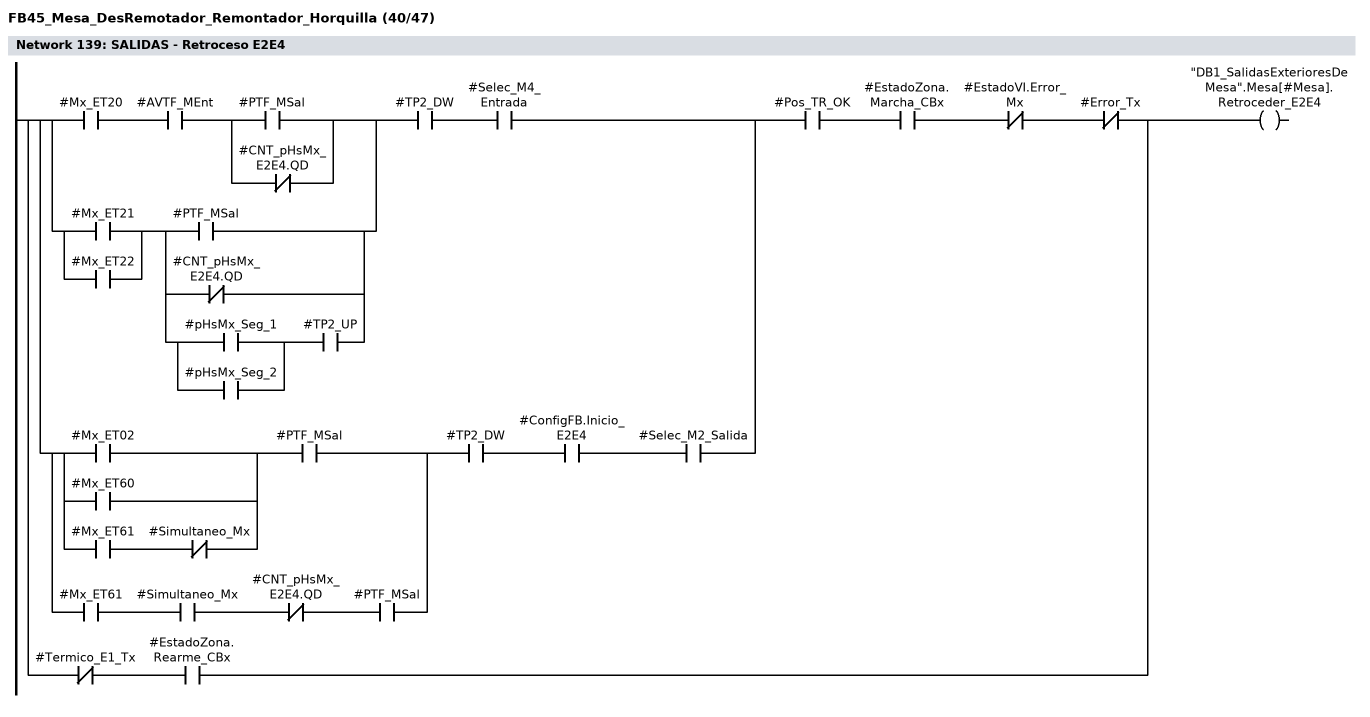
   RUNG wire#powerrail
      Contact( #Mx_ET20 )
      Contact( #AVTF_MEnt )
      wire#w1
      Contact( #PTF_MSal )
      wire#w2
      Contact( #TP2_DW )
      Contact( #Selec_M4_Entrada )
      wire#w5
      Contact( #Pos_TR_OK )
      Contact( #EstadoZona.Marcha_CBx )
      I_Contact( #EstadoVI.Error_Mx )
      I_Contact( #Error_Tx )
      wire#w8
      Coil( "DB1_SalidasExterioresDeMesa".Mesa[#Mesa].Retroceder_E2E4 )
   END_RUNG
   RUNG wire#w1
      I_Contact( #CNT_pHsMx_E2E4.QD )
   END_RUNG wire#w2
   RUNG wire#powerrail
      Contact( #Mx_ET21 )
      wire#w3
      Contact( #PTF_MSal )
   END_RUNG wire#w2
   RUNG wire#powerrail
      Contact( #Mx_ET22 )
   END_RUNG wire#w3
   RUNG wire#w3
      I_Contact( #CNT_pHsMx_E2E4.QD )
   END_RUNG wire#w2
   RUNG wire#w3
      Contact( #pHsMx_Seg_1 )
      wire#w4
      Contact( #TP2_UP )
   END_RUNG wire#w2
   RUNG wire#w3
      Contact( #pHsMx_Seg_2 )
   END_RUNG wire#w4
   RUNG wire#powerrail
      Contact( #Mx_ET02 )
      wire#w6
      Contact( #PTF_MSal )
      wire#w7
      Contact( #TP2_DW )
      Contact( #ConfigFB.Inicio_E2E4 )
      Contact( #Selec_M2_Salida )
   END_RUNG wire#w5
   RUNG wire#powerrail
      Contact( #Mx_ET60 )
   END_RUNG wire#w6
   RUNG wire#powerrail
      Contact( #Mx_ET61 )
      I_Contact( #Simultaneo_Mx )
   END_RUNG wire#w6
   RUNG wire#powerrail
      Contact( #Mx_ET61 )
      Contact( #Simultaneo_Mx )
      I_Contact( #CNT_pHsMx_E2E4.QD )
      Contact( #PTF_MSal )
   END_RUNG wire#w7
   RUNG wire#powerrail
      I_Contact( #Termico_E1_Tx )
      Contact( #EstadoZona.Rearme_CBx )
   END_RUNG wire#w8
   // the same network as SCL:
   "DB1_SalidasExterioresDeMesa".Mesa[#Mesa].Retroceder_E2E4 := (((((#Mx_ET20 AND #AVTF_MEnt AND (#PTF_MSal OR NOT #CNT_pHsMx_E2E4.QD)) OR ((#Mx_ET21 OR #Mx_ET22) AND (#PTF_MSal OR NOT #CNT_pHsMx_E2E4.QD OR ((#pHsMx_Seg_1 OR #pHsMx_Seg_2) AND #TP2_UP)))) AND #TP2_DW AND #Selec_M4_Entrada) OR ((((#Mx_ET02 OR #Mx_ET60 OR (#Mx_ET61 AND NOT #Simultaneo_Mx)) AND #PTF_MSal) OR (#Mx_ET61 AND #Simultaneo_Mx AND NOT #CNT_pHsMx_E2E4.QD AND #PTF_MSal)) AND #TP2_DW AND #ConfigFB.Inicio_E2E4 AND #Selec_M2_Salida)) AND #Pos_TR_OK AND #EstadoZona.Marcha_CBx AND NOT #EstadoVI.Error_Mx AND NOT #Error_Tx) OR (NOT #Termico_E1_Tx AND #EstadoZona.Rearme_CBx);
END_REGION

REGION Network 140: SALIDAS - Parar E2E4
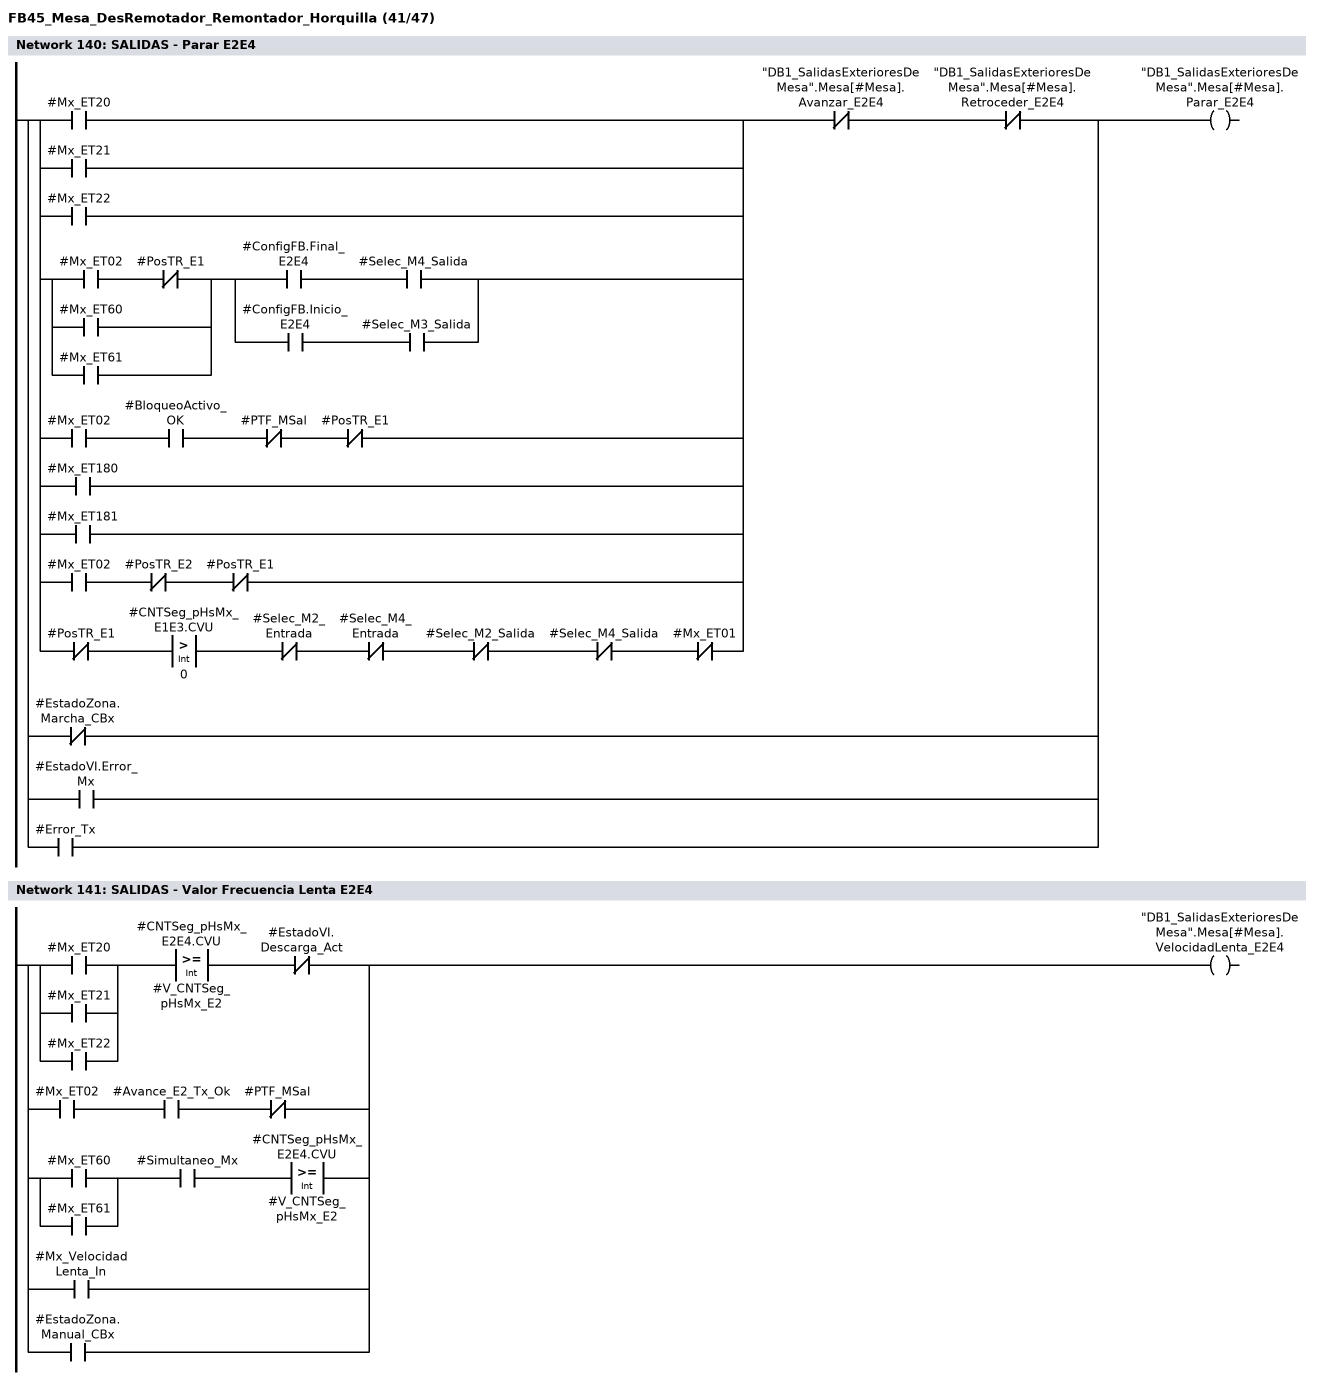
   RUNG wire#powerrail
      Contact( #Mx_ET20 )
      wire#w1
      I_Contact( "DB1_SalidasExterioresDeMesa".Mesa[#Mesa].Avanzar_E2E4 )
      I_Contact( "DB1_SalidasExterioresDeMesa".Mesa[#Mesa].Retroceder_E2E4 )
      wire#w3
      Coil( "DB1_SalidasExterioresDeMesa".Mesa[#Mesa].Parar_E2E4 )
   END_RUNG
   RUNG wire#powerrail
      Contact( #Mx_ET21 )
   END_RUNG wire#w1
   RUNG wire#powerrail
      Contact( #Mx_ET22 )
   END_RUNG wire#w1
   RUNG wire#powerrail
      Contact( #Mx_ET02 )
      I_Contact( #PosTR_E1 )
      wire#w2
      Contact( #ConfigFB.Final_E2E4 )
      Contact( #Selec_M4_Salida )
   END_RUNG wire#w1
   RUNG wire#powerrail
      Contact( #Mx_ET60 )
   END_RUNG wire#w2
   RUNG wire#powerrail
      Contact( #Mx_ET61 )
   END_RUNG wire#w2
   RUNG wire#w2
      Contact( #ConfigFB.Inicio_E2E4 )
      Contact( #Selec_M3_Salida )
   END_RUNG wire#w1
   RUNG wire#powerrail
      Contact( #Mx_ET02 )
      Contact( #BloqueoActivo_OK )
      I_Contact( #PTF_MSal )
      I_Contact( #PosTR_E1 )
   END_RUNG wire#w1
   RUNG wire#powerrail
      Contact( #Mx_ET180 )
   END_RUNG wire#w1
   RUNG wire#powerrail
      Contact( #Mx_ET181 )
   END_RUNG wire#w1
   RUNG wire#powerrail
      Contact( #Mx_ET02 )
      I_Contact( #PosTR_E2 )
      I_Contact( #PosTR_E1 )
   END_RUNG wire#w1
   RUNG wire#powerrail
      I_Contact( #PosTR_E1 )
      { S7_Templates := "SrcType := Int" } GT_Contact(in1 := #CNTSeg_pHsMx_E1E3.CVU, in2 := 0)
      I_Contact( #Selec_M2_Entrada )
      I_Contact( #Selec_M4_Entrada )
      I_Contact( #Selec_M2_Salida )
      I_Contact( #Selec_M4_Salida )
      I_Contact( #Mx_ET01 )
   END_RUNG wire#w1
   RUNG wire#powerrail
      I_Contact( #EstadoZona.Marcha_CBx )
   END_RUNG wire#w3
   RUNG wire#powerrail
      Contact( #EstadoVI.Error_Mx )
   END_RUNG wire#w3
   RUNG wire#powerrail
      Contact( #Error_Tx )
   END_RUNG wire#w3
   // the same network as SCL:
   "DB1_SalidasExterioresDeMesa".Mesa[#Mesa].Parar_E2E4 := ((#Mx_ET20 OR #Mx_ET21 OR #Mx_ET22 OR (((#Mx_ET02 AND NOT #PosTR_E1) OR #Mx_ET60 OR #Mx_ET61) AND ((#ConfigFB.Final_E2E4 AND #Selec_M4_Salida) OR (#ConfigFB.Inicio_E2E4 AND #Selec_M3_Salida))) OR (#Mx_ET02 AND #BloqueoActivo_OK AND NOT #PTF_MSal AND NOT #PosTR_E1) OR #Mx_ET180 OR #Mx_ET181 OR (#Mx_ET02 AND NOT #PosTR_E2 AND NOT #PosTR_E1) OR (NOT #PosTR_E1 AND (#CNTSeg_pHsMx_E1E3.CVU > 0) AND NOT #Selec_M2_Entrada AND NOT #Selec_M4_Entrada AND NOT #Selec_M2_Salida AND NOT #Selec_M4_Salida AND NOT #Mx_ET01)) AND NOT "DB1_SalidasExterioresDeMesa".Mesa[#Mesa].Avanzar_E2E4 AND NOT "DB1_SalidasExterioresDeMesa".Mesa[#Mesa].Retroceder_E2E4) OR NOT #EstadoZona.Marcha_CBx OR #EstadoVI.Error_Mx OR #Error_Tx;
END_REGION

REGION Network 141: SALIDAS - Valor Frecuencia Lenta E2E4
   RUNG wire#powerrail
      Contact( #Mx_ET20 )
      wire#w1
      { S7_Templates := "SrcType := Int" } GE_Contact(in1 := #CNTSeg_pHsMx_E2E4.CVU, in2 := #V_CNTSeg_pHsMx_E2)
      I_Contact( #EstadoVI.Descarga_Act )
      wire#w2
      Coil( "DB1_SalidasExterioresDeMesa".Mesa[#Mesa].VelocidadLenta_E2E4 )
   END_RUNG
   RUNG wire#powerrail
      Contact( #Mx_ET21 )
   END_RUNG wire#w1
   RUNG wire#powerrail
      Contact( #Mx_ET22 )
   END_RUNG wire#w1
   RUNG wire#powerrail
      Contact( #Mx_ET02 )
      Contact( #Avance_E2_Tx_Ok )
      I_Contact( #PTF_MSal )
   END_RUNG wire#w2
   RUNG wire#powerrail
      Contact( #Mx_ET60 )
      wire#w3
      Contact( #Simultaneo_Mx )
      { S7_Templates := "SrcType := Int" } GE_Contact(in1 := #CNTSeg_pHsMx_E2E4.CVU, in2 := #V_CNTSeg_pHsMx_E2)
   END_RUNG wire#w2
   RUNG wire#powerrail
      Contact( #Mx_ET61 )
   END_RUNG wire#w3
   RUNG wire#powerrail
      Contact( #Mx_VelocidadLenta_In )
   END_RUNG wire#w2
   RUNG wire#powerrail
      Contact( #EstadoZona.Manual_CBx )
   END_RUNG wire#w2
   // the same network as SCL:
   "DB1_SalidasExterioresDeMesa".Mesa[#Mesa].VelocidadLenta_E2E4 := ((#Mx_ET20 OR #Mx_ET21 OR #Mx_ET22) AND (#CNTSeg_pHsMx_E2E4.CVU >= #V_CNTSeg_pHsMx_E2) AND NOT #EstadoVI.Descarga_Act) OR (#Mx_ET02 AND #Avance_E2_Tx_Ok AND NOT #PTF_MSal) OR ((#Mx_ET60 OR #Mx_ET61) AND #Simultaneo_Mx AND (#CNTSeg_pHsMx_E2E4.CVU >= #V_CNTSeg_pHsMx_E2)) OR #Mx_VelocidadLenta_In OR #EstadoZona.Manual_CBx;
END_REGION

REGION Network 142: SALIDAS - Ir a posicion E1E3
   // DANI: 2021/06/28. BAJAR EL TOPE DE CADENAS SI HAY S2 O S4 EN ETAPA2 Y TR POS RODILLOS
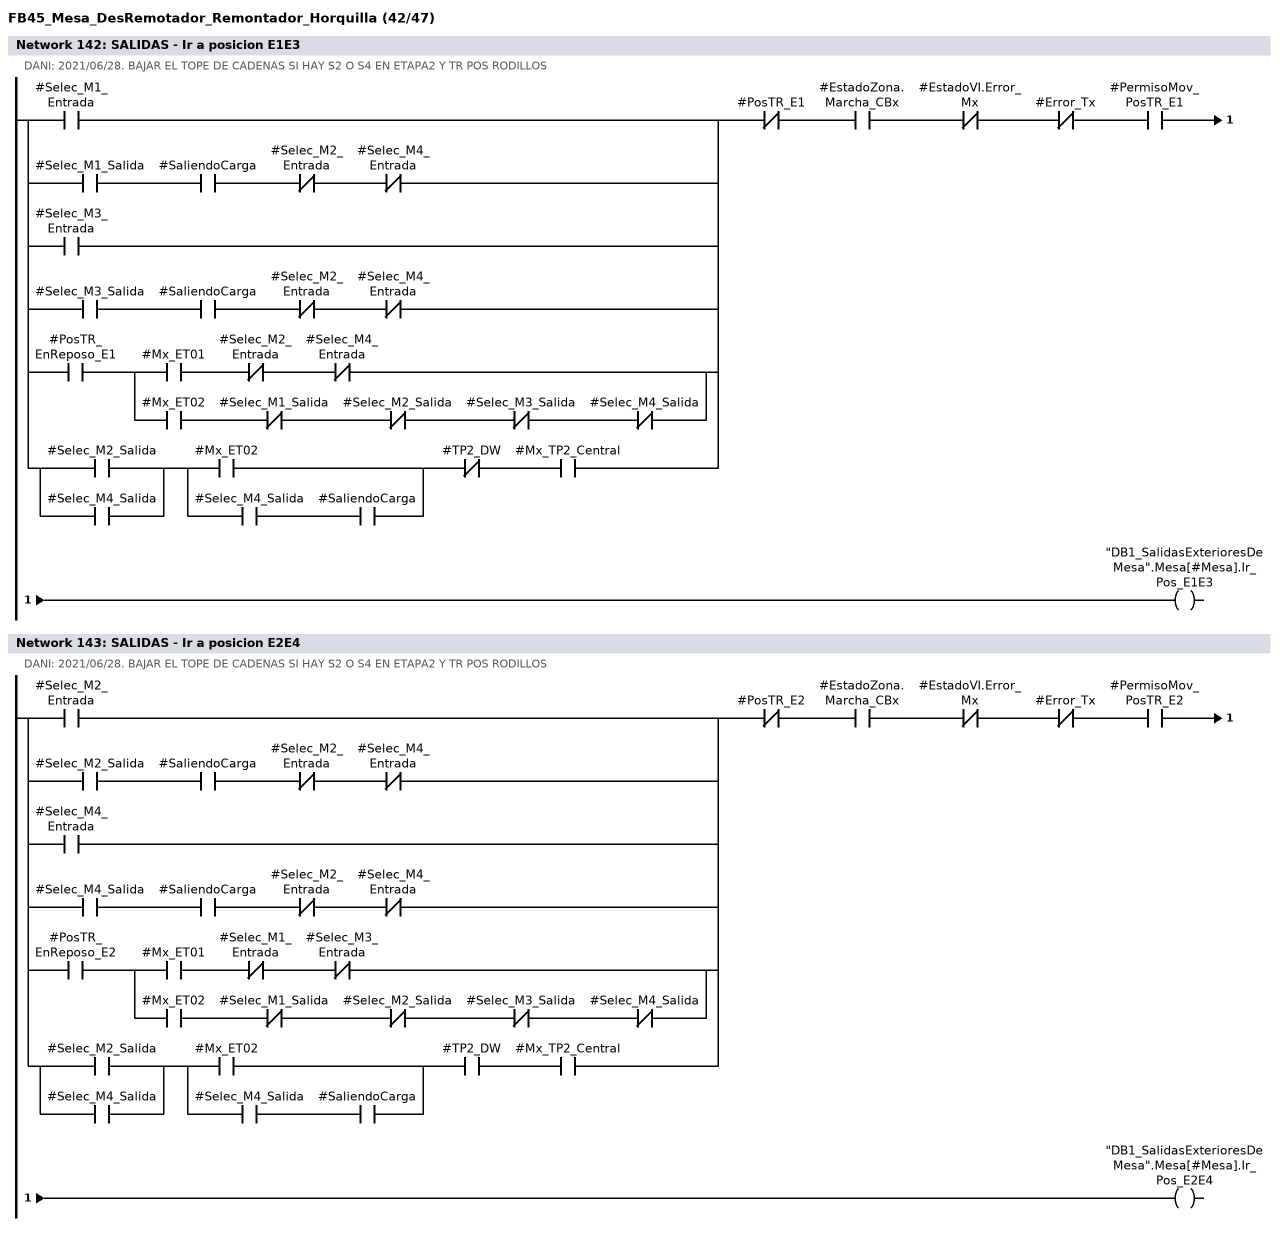
   RUNG wire#powerrail
      Contact( #Selec_M1_Entrada )
      wire#w1
      I_Contact( #PosTR_E1 )
      Contact( #EstadoZona.Marcha_CBx )
      I_Contact( #EstadoVI.Error_Mx )
      I_Contact( #Error_Tx )
      Contact( #PermisoMov_PosTR_E1 )
      Coil( "DB1_SalidasExterioresDeMesa".Mesa[#Mesa].Ir_Pos_E1E3 )
   END_RUNG
   RUNG wire#powerrail
      Contact( #Selec_M1_Salida )
      Contact( #SaliendoCarga )
      I_Contact( #Selec_M2_Entrada )
      I_Contact( #Selec_M4_Entrada )
   END_RUNG wire#w1
   RUNG wire#powerrail
      Contact( #Selec_M3_Entrada )
   END_RUNG wire#w1
   RUNG wire#powerrail
      Contact( #Selec_M3_Salida )
      Contact( #SaliendoCarga )
      I_Contact( #Selec_M2_Entrada )
      I_Contact( #Selec_M4_Entrada )
   END_RUNG wire#w1
   RUNG wire#powerrail
      Contact( #PosTR_EnReposo_E1 )
      wire#w2
      Contact( #Mx_ET01 )
      I_Contact( #Selec_M2_Entrada )
      I_Contact( #Selec_M4_Entrada )
   END_RUNG wire#w1
   RUNG wire#w2
      Contact( #Mx_ET02 )
      I_Contact( #Selec_M1_Salida )
      I_Contact( #Selec_M2_Salida )
      I_Contact( #Selec_M3_Salida )
      I_Contact( #Selec_M4_Salida )
   END_RUNG wire#w1
   RUNG wire#powerrail
      Contact( #Selec_M2_Salida )
      wire#w3
      Contact( #Mx_ET02 )
      wire#w4
      I_Contact( #TP2_DW )
      Contact( #Mx_TP2_Central )
   END_RUNG wire#w1
   RUNG wire#powerrail
      Contact( #Selec_M4_Salida )
   END_RUNG wire#w3
   RUNG wire#w3
      Contact( #Selec_M4_Salida )
      Contact( #SaliendoCarga )
   END_RUNG wire#w4
   // the same network as SCL:
   "DB1_SalidasExterioresDeMesa".Mesa[#Mesa].Ir_Pos_E1E3 := (#Selec_M1_Entrada OR (#Selec_M1_Salida AND #SaliendoCarga AND NOT #Selec_M2_Entrada AND NOT #Selec_M4_Entrada) OR #Selec_M3_Entrada OR (#Selec_M3_Salida AND #SaliendoCarga AND NOT #Selec_M2_Entrada AND NOT #Selec_M4_Entrada) OR (#PosTR_EnReposo_E1 AND ((#Mx_ET01 AND NOT #Selec_M2_Entrada AND NOT #Selec_M4_Entrada) OR (#Mx_ET02 AND NOT #Selec_M1_Salida AND NOT #Selec_M2_Salida AND NOT #Selec_M3_Salida AND NOT #Selec_M4_Salida))) OR ((#Selec_M2_Salida OR #Selec_M4_Salida) AND (#Mx_ET02 OR (#Selec_M4_Salida AND #SaliendoCarga)) AND NOT #TP2_DW AND #Mx_TP2_Central)) AND NOT #PosTR_E1 AND #EstadoZona.Marcha_CBx AND NOT #EstadoVI.Error_Mx AND NOT #Error_Tx AND #PermisoMov_PosTR_E1;
END_REGION

REGION Network 143: SALIDAS - Ir a posicion E2E4
   // DANI: 2021/06/28. BAJAR EL TOPE DE CADENAS SI HAY S2 O S4 EN ETAPA2 Y TR POS RODILLOS
   RUNG wire#powerrail
      Contact( #Selec_M2_Entrada )
      wire#w1
      I_Contact( #PosTR_E2 )
      Contact( #EstadoZona.Marcha_CBx )
      I_Contact( #EstadoVI.Error_Mx )
      I_Contact( #Error_Tx )
      Contact( #PermisoMov_PosTR_E2 )
      Coil( "DB1_SalidasExterioresDeMesa".Mesa[#Mesa].Ir_Pos_E2E4 )
   END_RUNG
   RUNG wire#powerrail
      Contact( #Selec_M2_Salida )
      Contact( #SaliendoCarga )
      I_Contact( #Selec_M2_Entrada )
      I_Contact( #Selec_M4_Entrada )
   END_RUNG wire#w1
   RUNG wire#powerrail
      Contact( #Selec_M4_Entrada )
   END_RUNG wire#w1
   RUNG wire#powerrail
      Contact( #Selec_M4_Salida )
      Contact( #SaliendoCarga )
      I_Contact( #Selec_M2_Entrada )
      I_Contact( #Selec_M4_Entrada )
   END_RUNG wire#w1
   RUNG wire#powerrail
      Contact( #PosTR_EnReposo_E2 )
      wire#w2
      Contact( #Mx_ET01 )
      I_Contact( #Selec_M1_Entrada )
      I_Contact( #Selec_M3_Entrada )
   END_RUNG wire#w1
   RUNG wire#w2
      Contact( #Mx_ET02 )
      I_Contact( #Selec_M1_Salida )
      I_Contact( #Selec_M2_Salida )
      I_Contact( #Selec_M3_Salida )
      I_Contact( #Selec_M4_Salida )
   END_RUNG wire#w1
   RUNG wire#powerrail
      Contact( #Selec_M2_Salida )
      wire#w3
      Contact( #Mx_ET02 )
      wire#w4
      Contact( #TP2_DW )
      Contact( #Mx_TP2_Central )
   END_RUNG wire#w1
   RUNG wire#powerrail
      Contact( #Selec_M4_Salida )
   END_RUNG wire#w3
   RUNG wire#w3
      Contact( #Selec_M4_Salida )
      Contact( #SaliendoCarga )
   END_RUNG wire#w4
   // the same network as SCL:
   "DB1_SalidasExterioresDeMesa".Mesa[#Mesa].Ir_Pos_E2E4 := (#Selec_M2_Entrada OR (#Selec_M2_Salida AND #SaliendoCarga AND NOT #Selec_M2_Entrada AND NOT #Selec_M4_Entrada) OR #Selec_M4_Entrada OR (#Selec_M4_Salida AND #SaliendoCarga AND NOT #Selec_M2_Entrada AND NOT #Selec_M4_Entrada) OR (#PosTR_EnReposo_E2 AND ((#Mx_ET01 AND NOT #Selec_M1_Entrada AND NOT #Selec_M3_Entrada) OR (#Mx_ET02 AND NOT #Selec_M1_Salida AND NOT #Selec_M2_Salida AND NOT #Selec_M3_Salida AND NOT #Selec_M4_Salida))) OR ((#Selec_M2_Salida OR #Selec_M4_Salida) AND (#Mx_ET02 OR (#Selec_M4_Salida AND #SaliendoCarga)) AND #TP2_DW AND #Mx_TP2_Central)) AND NOT #PosTR_E2 AND #EstadoZona.Marcha_CBx AND NOT #EstadoVI.Error_Mx AND NOT #Error_Tx AND #PermisoMov_PosTR_E2;
END_REGION

REGION Network 144: SALIDAS - Bajar TP1
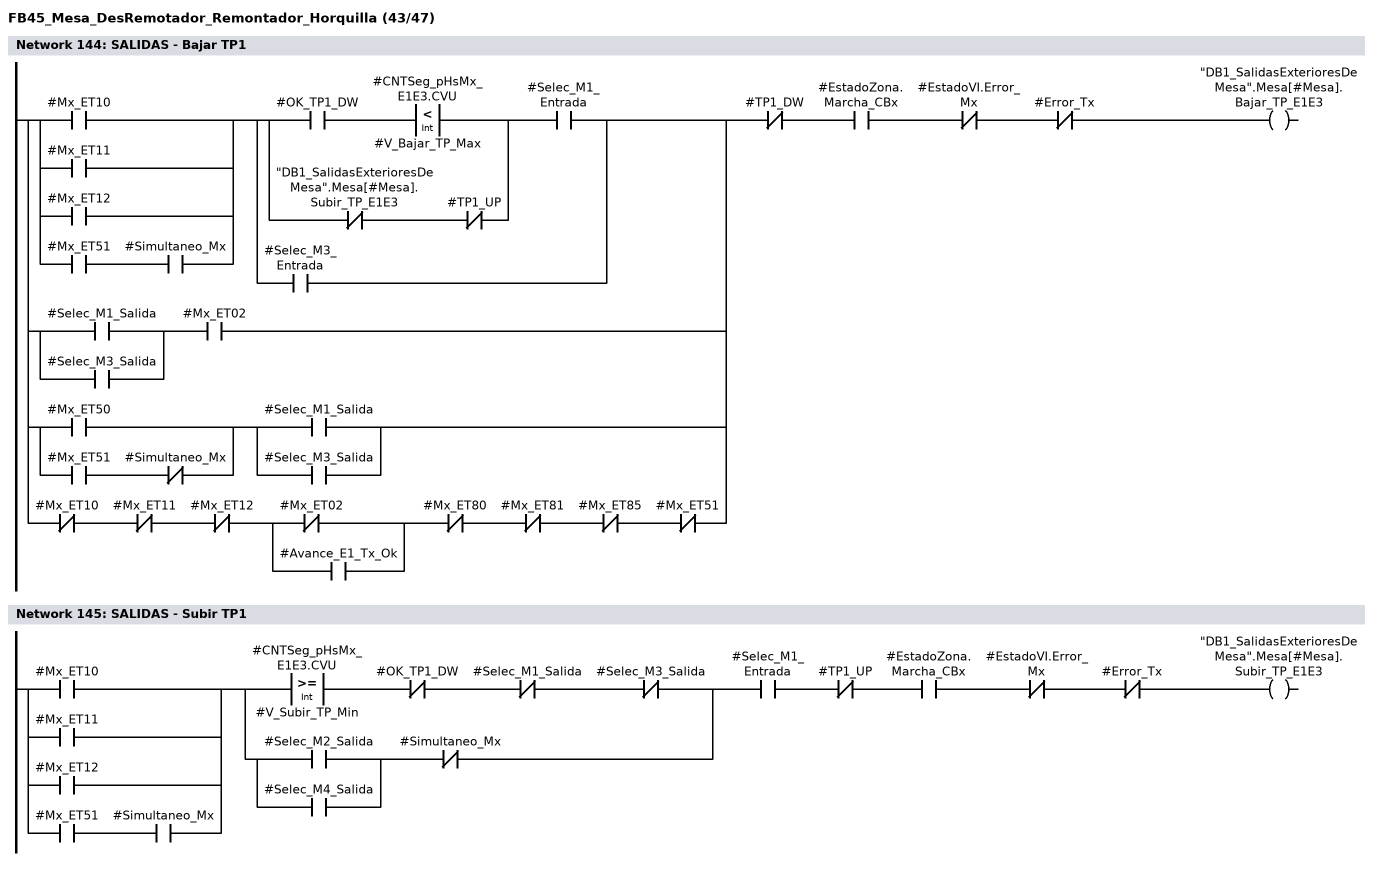
   RUNG wire#powerrail
      Contact( #Mx_ET10 )
      wire#w1
      Contact( #OK_TP1_DW )
      { S7_Templates := "SrcType := Int" } LT_Contact(in1 := #CNTSeg_pHsMx_E1E3.CVU, in2 := #V_Bajar_TP_Max)
      wire#w2
      Contact( #Selec_M1_Entrada )
      wire#w3
      I_Contact( #TP1_DW )
      Contact( #EstadoZona.Marcha_CBx )
      I_Contact( #EstadoVI.Error_Mx )
      I_Contact( #Error_Tx )
      Coil( "DB1_SalidasExterioresDeMesa".Mesa[#Mesa].Bajar_TP_E1E3 )
   END_RUNG
   RUNG wire#powerrail
      Contact( #Mx_ET11 )
   END_RUNG wire#w1
   RUNG wire#powerrail
      Contact( #Mx_ET12 )
   END_RUNG wire#w1
   RUNG wire#powerrail
      Contact( #Mx_ET51 )
      Contact( #Simultaneo_Mx )
   END_RUNG wire#w1
   RUNG wire#w1
      I_Contact( "DB1_SalidasExterioresDeMesa".Mesa[#Mesa].Subir_TP_E1E3 )
      I_Contact( #TP1_UP )
   END_RUNG wire#w2
   RUNG wire#w1
      Contact( #Selec_M3_Entrada )
   END_RUNG wire#w3
   RUNG wire#powerrail
      Contact( #Selec_M1_Salida )
      wire#w4
      Contact( #Mx_ET02 )
   END_RUNG wire#w3
   RUNG wire#powerrail
      Contact( #Selec_M3_Salida )
   END_RUNG wire#w4
   RUNG wire#powerrail
      Contact( #Mx_ET50 )
      wire#w5
      Contact( #Selec_M1_Salida )
   END_RUNG wire#w3
   RUNG wire#powerrail
      Contact( #Mx_ET51 )
      I_Contact( #Simultaneo_Mx )
   END_RUNG wire#w5
   RUNG wire#w5
      Contact( #Selec_M3_Salida )
   END_RUNG wire#w3
   RUNG wire#powerrail
      I_Contact( #Mx_ET10 )
      I_Contact( #Mx_ET11 )
      I_Contact( #Mx_ET12 )
      wire#w6
      I_Contact( #Mx_ET02 )
      wire#w7
      I_Contact( #Mx_ET80 )
      I_Contact( #Mx_ET81 )
      I_Contact( #Mx_ET85 )
      I_Contact( #Mx_ET51 )
   END_RUNG wire#w3
   RUNG wire#w6
      Contact( #Avance_E1_Tx_Ok )
   END_RUNG wire#w7
   // the same network as SCL:
   "DB1_SalidasExterioresDeMesa".Mesa[#Mesa].Bajar_TP_E1E3 := (((#Mx_ET10 OR #Mx_ET11 OR #Mx_ET12 OR (#Mx_ET51 AND #Simultaneo_Mx)) AND ((((#OK_TP1_DW AND (#CNTSeg_pHsMx_E1E3.CVU < #V_Bajar_TP_Max)) OR (NOT "DB1_SalidasExterioresDeMesa".Mesa[#Mesa].Subir_TP_E1E3 AND NOT #TP1_UP)) AND #Selec_M1_Entrada) OR #Selec_M3_Entrada)) OR ((#Selec_M1_Salida OR #Selec_M3_Salida) AND #Mx_ET02) OR ((#Mx_ET50 OR (#Mx_ET51 AND NOT #Simultaneo_Mx)) AND (#Selec_M1_Salida OR #Selec_M3_Salida)) OR (NOT #Mx_ET10 AND NOT #Mx_ET11 AND NOT #Mx_ET12 AND (NOT #Mx_ET02 OR #Avance_E1_Tx_Ok) AND NOT #Mx_ET80 AND NOT #Mx_ET81 AND NOT #Mx_ET85 AND NOT #Mx_ET51)) AND NOT #TP1_DW AND #EstadoZona.Marcha_CBx AND NOT #EstadoVI.Error_Mx AND NOT #Error_Tx;
END_REGION

REGION Network 145: SALIDAS - Subir TP1
   RUNG wire#powerrail
      Contact( #Mx_ET10 )
      wire#w1
      { S7_Templates := "SrcType := Int" } GE_Contact(in1 := #CNTSeg_pHsMx_E1E3.CVU, in2 := #V_Subir_TP_Min)
      I_Contact( #OK_TP1_DW )
      I_Contact( #Selec_M1_Salida )
      I_Contact( #Selec_M3_Salida )
      wire#w2
      Contact( #Selec_M1_Entrada )
      I_Contact( #TP1_UP )
      Contact( #EstadoZona.Marcha_CBx )
      I_Contact( #EstadoVI.Error_Mx )
      I_Contact( #Error_Tx )
      Coil( "DB1_SalidasExterioresDeMesa".Mesa[#Mesa].Subir_TP_E1E3 )
   END_RUNG
   RUNG wire#powerrail
      Contact( #Mx_ET11 )
   END_RUNG wire#w1
   RUNG wire#powerrail
      Contact( #Mx_ET12 )
   END_RUNG wire#w1
   RUNG wire#powerrail
      Contact( #Mx_ET51 )
      Contact( #Simultaneo_Mx )
   END_RUNG wire#w1
   RUNG wire#w1
      Contact( #Selec_M2_Salida )
      wire#w3
      I_Contact( #Simultaneo_Mx )
   END_RUNG wire#w2
   RUNG wire#w1
      Contact( #Selec_M4_Salida )
   END_RUNG wire#w3
   // the same network as SCL:
   "DB1_SalidasExterioresDeMesa".Mesa[#Mesa].Subir_TP_E1E3 := (#Mx_ET10 OR #Mx_ET11 OR #Mx_ET12 OR (#Mx_ET51 AND #Simultaneo_Mx)) AND (((#CNTSeg_pHsMx_E1E3.CVU >= #V_Subir_TP_Min) AND NOT #OK_TP1_DW AND NOT #Selec_M1_Salida AND NOT #Selec_M3_Salida) OR ((#Selec_M2_Salida OR #Selec_M4_Salida) AND NOT #Simultaneo_Mx)) AND #Selec_M1_Entrada AND NOT #TP1_UP AND #EstadoZona.Marcha_CBx AND NOT #EstadoVI.Error_Mx AND NOT #Error_Tx;
END_REGION

REGION Network 146: SALIDAS - Bajar TP2
   // DANI: 2021/06/28. BAJAR EL TOPE DE CADENAS SI HAY S2 O S4 EN ETAPA2 Y TR POS RODILLOS
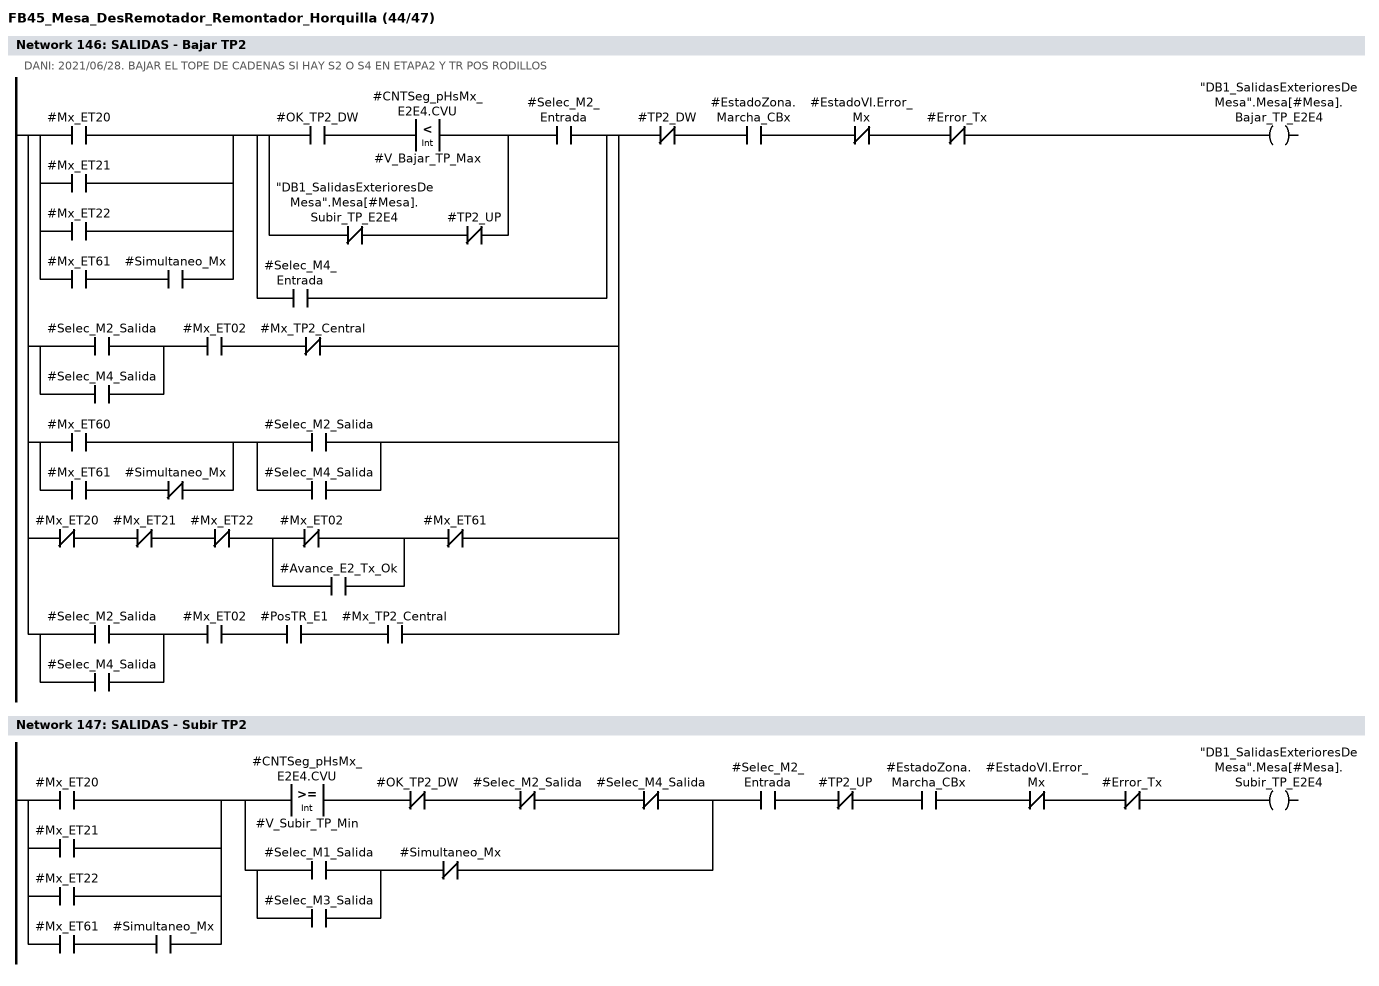
   RUNG wire#powerrail
      Contact( #Mx_ET20 )
      wire#w1
      Contact( #OK_TP2_DW )
      { S7_Templates := "SrcType := Int" } LT_Contact(in1 := #CNTSeg_pHsMx_E2E4.CVU, in2 := #V_Bajar_TP_Max)
      wire#w2
      Contact( #Selec_M2_Entrada )
      wire#w3
      I_Contact( #TP2_DW )
      Contact( #EstadoZona.Marcha_CBx )
      I_Contact( #EstadoVI.Error_Mx )
      I_Contact( #Error_Tx )
      Coil( "DB1_SalidasExterioresDeMesa".Mesa[#Mesa].Bajar_TP_E2E4 )
   END_RUNG
   RUNG wire#powerrail
      Contact( #Mx_ET21 )
   END_RUNG wire#w1
   RUNG wire#powerrail
      Contact( #Mx_ET22 )
   END_RUNG wire#w1
   RUNG wire#powerrail
      Contact( #Mx_ET61 )
      Contact( #Simultaneo_Mx )
   END_RUNG wire#w1
   RUNG wire#w1
      I_Contact( "DB1_SalidasExterioresDeMesa".Mesa[#Mesa].Subir_TP_E2E4 )
      I_Contact( #TP2_UP )
   END_RUNG wire#w2
   RUNG wire#w1
      Contact( #Selec_M4_Entrada )
   END_RUNG wire#w3
   RUNG wire#powerrail
      Contact( #Selec_M2_Salida )
      wire#w4
      Contact( #Mx_ET02 )
      I_Contact( #Mx_TP2_Central )
   END_RUNG wire#w3
   RUNG wire#powerrail
      Contact( #Selec_M4_Salida )
   END_RUNG wire#w4
   RUNG wire#powerrail
      Contact( #Mx_ET60 )
      wire#w5
      Contact( #Selec_M2_Salida )
   END_RUNG wire#w3
   RUNG wire#powerrail
      Contact( #Mx_ET61 )
      I_Contact( #Simultaneo_Mx )
   END_RUNG wire#w5
   RUNG wire#w5
      Contact( #Selec_M4_Salida )
   END_RUNG wire#w3
   RUNG wire#powerrail
      I_Contact( #Mx_ET20 )
      I_Contact( #Mx_ET21 )
      I_Contact( #Mx_ET22 )
      wire#w6
      I_Contact( #Mx_ET02 )
      wire#w7
      I_Contact( #Mx_ET61 )
   END_RUNG wire#w3
   RUNG wire#w6
      Contact( #Avance_E2_Tx_Ok )
   END_RUNG wire#w7
   RUNG wire#powerrail
      Contact( #Selec_M2_Salida )
      wire#w8
      Contact( #Mx_ET02 )
      Contact( #PosTR_E1 )
      Contact( #Mx_TP2_Central )
   END_RUNG wire#w3
   RUNG wire#powerrail
      Contact( #Selec_M4_Salida )
   END_RUNG wire#w8
   // the same network as SCL:
   "DB1_SalidasExterioresDeMesa".Mesa[#Mesa].Bajar_TP_E2E4 := (((#Mx_ET20 OR #Mx_ET21 OR #Mx_ET22 OR (#Mx_ET61 AND #Simultaneo_Mx)) AND ((((#OK_TP2_DW AND (#CNTSeg_pHsMx_E2E4.CVU < #V_Bajar_TP_Max)) OR (NOT "DB1_SalidasExterioresDeMesa".Mesa[#Mesa].Subir_TP_E2E4 AND NOT #TP2_UP)) AND #Selec_M2_Entrada) OR #Selec_M4_Entrada)) OR ((#Selec_M2_Salida OR #Selec_M4_Salida) AND #Mx_ET02 AND NOT #Mx_TP2_Central) OR ((#Mx_ET60 OR (#Mx_ET61 AND NOT #Simultaneo_Mx)) AND (#Selec_M2_Salida OR #Selec_M4_Salida)) OR (NOT #Mx_ET20 AND NOT #Mx_ET21 AND NOT #Mx_ET22 AND (NOT #Mx_ET02 OR #Avance_E2_Tx_Ok) AND NOT #Mx_ET61) OR ((#Selec_M2_Salida OR #Selec_M4_Salida) AND #Mx_ET02 AND #PosTR_E1 AND #Mx_TP2_Central)) AND NOT #TP2_DW AND #EstadoZona.Marcha_CBx AND NOT #EstadoVI.Error_Mx AND NOT #Error_Tx;
END_REGION

REGION Network 147: SALIDAS - Subir TP2
   RUNG wire#powerrail
      Contact( #Mx_ET20 )
      wire#w1
      { S7_Templates := "SrcType := Int" } GE_Contact(in1 := #CNTSeg_pHsMx_E2E4.CVU, in2 := #V_Subir_TP_Min)
      I_Contact( #OK_TP2_DW )
      I_Contact( #Selec_M2_Salida )
      I_Contact( #Selec_M4_Salida )
      wire#w2
      Contact( #Selec_M2_Entrada )
      I_Contact( #TP2_UP )
      Contact( #EstadoZona.Marcha_CBx )
      I_Contact( #EstadoVI.Error_Mx )
      I_Contact( #Error_Tx )
      Coil( "DB1_SalidasExterioresDeMesa".Mesa[#Mesa].Subir_TP_E2E4 )
   END_RUNG
   RUNG wire#powerrail
      Contact( #Mx_ET21 )
   END_RUNG wire#w1
   RUNG wire#powerrail
      Contact( #Mx_ET22 )
   END_RUNG wire#w1
   RUNG wire#powerrail
      Contact( #Mx_ET61 )
      Contact( #Simultaneo_Mx )
   END_RUNG wire#w1
   RUNG wire#w1
      Contact( #Selec_M1_Salida )
      wire#w3
      I_Contact( #Simultaneo_Mx )
   END_RUNG wire#w2
   RUNG wire#w1
      Contact( #Selec_M3_Salida )
   END_RUNG wire#w3
   // the same network as SCL:
   "DB1_SalidasExterioresDeMesa".Mesa[#Mesa].Subir_TP_E2E4 := (#Mx_ET20 OR #Mx_ET21 OR #Mx_ET22 OR (#Mx_ET61 AND #Simultaneo_Mx)) AND (((#CNTSeg_pHsMx_E2E4.CVU >= #V_Subir_TP_Min) AND NOT #OK_TP2_DW AND NOT #Selec_M2_Salida AND NOT #Selec_M4_Salida) OR ((#Selec_M1_Salida OR #Selec_M3_Salida) AND NOT #Simultaneo_Mx)) AND #Selec_M2_Entrada AND NOT #TP2_UP AND #EstadoZona.Marcha_CBx AND NOT #EstadoVI.Error_Mx AND NOT #Error_Tx;
END_REGION

REGION Network 148: ESTADOS DE LA MESA
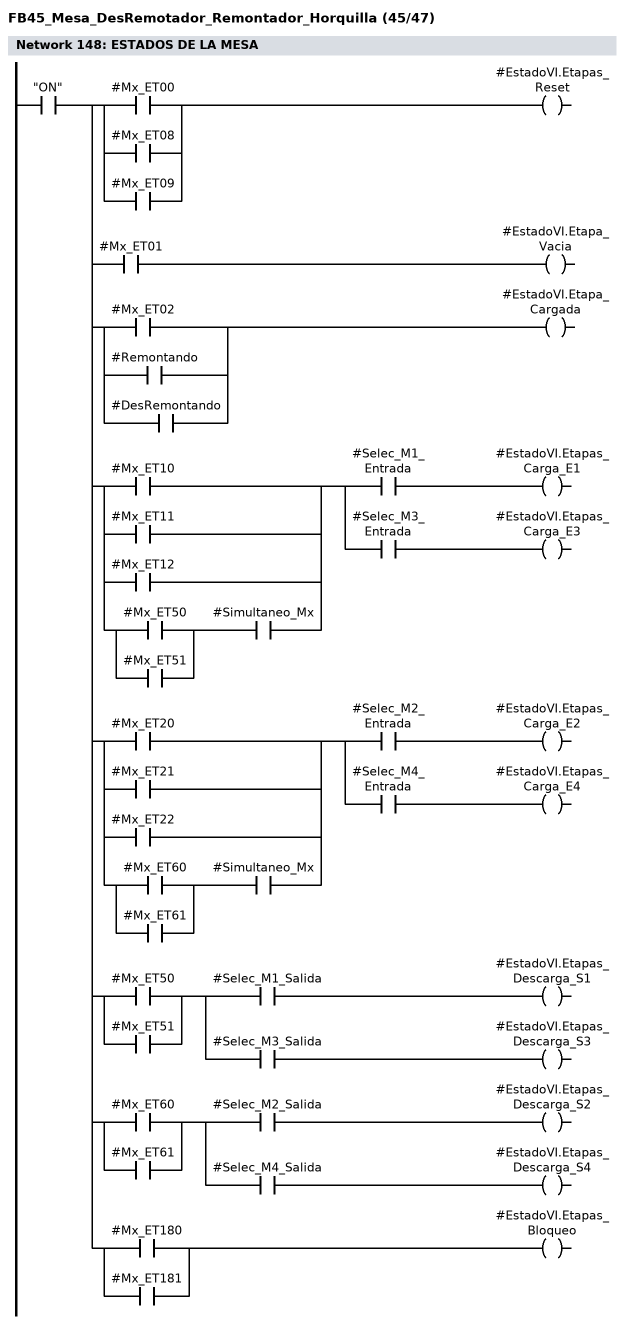
   RUNG wire#powerrail
      Contact( "ON" )
      wire#w1
      Contact( #Mx_ET00 )
      wire#w2
      Coil( #EstadoVI.Etapas_Reset )
   END_RUNG
   RUNG wire#w1
      Contact( #Mx_ET08 )
   END_RUNG wire#w2
   RUNG wire#w1
      Contact( #Mx_ET09 )
   END_RUNG wire#w2
   RUNG wire#w1
      Contact( #Mx_ET01 )
      Coil( #EstadoVI.Etapa_Vacia )
   END_RUNG
   RUNG wire#w1
      Contact( #Mx_ET02 )
      wire#w3
      Coil( #EstadoVI.Etapa_Cargada )
   END_RUNG
   RUNG wire#w1
      Contact( #Remontando )
   END_RUNG wire#w3
   RUNG wire#w1
      Contact( #DesRemontando )
   END_RUNG wire#w3
   RUNG wire#w1
      Contact( #Mx_ET10 )
      wire#w4
      Contact( #Selec_M1_Entrada )
      Coil( #EstadoVI.Etapas_Carga_E1 )
   END_RUNG
   RUNG wire#w1
      Contact( #Mx_ET11 )
   END_RUNG wire#w4
   RUNG wire#w1
      Contact( #Mx_ET12 )
   END_RUNG wire#w4
   RUNG wire#w1
      Contact( #Mx_ET50 )
      wire#w5
      Contact( #Simultaneo_Mx )
   END_RUNG wire#w4
   RUNG wire#w1
      Contact( #Mx_ET51 )
   END_RUNG wire#w5
   RUNG wire#w4
      Contact( #Selec_M3_Entrada )
      Coil( #EstadoVI.Etapas_Carga_E3 )
   END_RUNG
   RUNG wire#w1
      Contact( #Mx_ET20 )
      wire#w6
      Contact( #Selec_M2_Entrada )
      Coil( #EstadoVI.Etapas_Carga_E2 )
   END_RUNG
   RUNG wire#w1
      Contact( #Mx_ET21 )
   END_RUNG wire#w6
   RUNG wire#w1
      Contact( #Mx_ET22 )
   END_RUNG wire#w6
   RUNG wire#w1
      Contact( #Mx_ET60 )
      wire#w7
      Contact( #Simultaneo_Mx )
   END_RUNG wire#w6
   RUNG wire#w1
      Contact( #Mx_ET61 )
   END_RUNG wire#w7
   RUNG wire#w6
      Contact( #Selec_M4_Entrada )
      Coil( #EstadoVI.Etapas_Carga_E4 )
   END_RUNG
   RUNG wire#w1
      Contact( #Mx_ET50 )
      wire#w8
      Contact( #Selec_M1_Salida )
      Coil( #EstadoVI.Etapas_Descarga_S1 )
   END_RUNG
   RUNG wire#w1
      Contact( #Mx_ET51 )
   END_RUNG wire#w8
   RUNG wire#w8
      Contact( #Selec_M3_Salida )
      Coil( #EstadoVI.Etapas_Descarga_S3 )
   END_RUNG
   RUNG wire#w1
      Contact( #Mx_ET60 )
      wire#w9
      Contact( #Selec_M2_Salida )
      Coil( #EstadoVI.Etapas_Descarga_S2 )
   END_RUNG
   RUNG wire#w1
      Contact( #Mx_ET61 )
   END_RUNG wire#w9
   RUNG wire#w9
      Contact( #Selec_M4_Salida )
      Coil( #EstadoVI.Etapas_Descarga_S4 )
   END_RUNG
   RUNG wire#w1
      Contact( #Mx_ET180 )
      wire#w10
      Coil( #EstadoVI.Etapas_Bloqueo )
   END_RUNG
   RUNG wire#w1
      Contact( #Mx_ET181 )
   END_RUNG wire#w10
   // the same network as SCL:
   #EstadoVI.Etapas_Reset := "ON" AND (#Mx_ET00 OR #Mx_ET08 OR #Mx_ET09);
   #EstadoVI.Etapa_Vacia := "ON" AND #Mx_ET01;
   #EstadoVI.Etapa_Cargada := "ON" AND (#Mx_ET02 OR #Remontando OR #DesRemontando);
   #_w1 := "ON" AND (#Mx_ET10 OR #Mx_ET11 OR #Mx_ET12 OR ((#Mx_ET50 OR #Mx_ET51) AND #Simultaneo_Mx));
   #EstadoVI.Etapas_Carga_E1 := #_w1 AND #Selec_M1_Entrada;
   #EstadoVI.Etapas_Carga_E3 := #_w1 AND #Selec_M3_Entrada;
   #_w2 := "ON" AND (#Mx_ET20 OR #Mx_ET21 OR #Mx_ET22 OR ((#Mx_ET60 OR #Mx_ET61) AND #Simultaneo_Mx));
   #EstadoVI.Etapas_Carga_E2 := #_w2 AND #Selec_M2_Entrada;
   #EstadoVI.Etapas_Carga_E4 := #_w2 AND #Selec_M4_Entrada;
   #_w3 := "ON" AND (#Mx_ET50 OR #Mx_ET51);
   #EstadoVI.Etapas_Descarga_S1 := #_w3 AND #Selec_M1_Salida;
   #EstadoVI.Etapas_Descarga_S3 := #_w3 AND #Selec_M3_Salida;
   #_w4 := "ON" AND (#Mx_ET60 OR #Mx_ET61);
   #EstadoVI.Etapas_Descarga_S2 := #_w4 AND #Selec_M2_Salida;
   #EstadoVI.Etapas_Descarga_S4 := #_w4 AND #Selec_M4_Salida;
   #EstadoVI.Etapas_Bloqueo := "ON" AND (#Mx_ET180 OR #Mx_ET181);
END_REGION

REGION Network 149: ESTADO ENTRADAS DE LA MESA
   // MODIF: TRANSFER UP, TRANSFER_DW, TOPE_UP_2, TOPE_DW_2
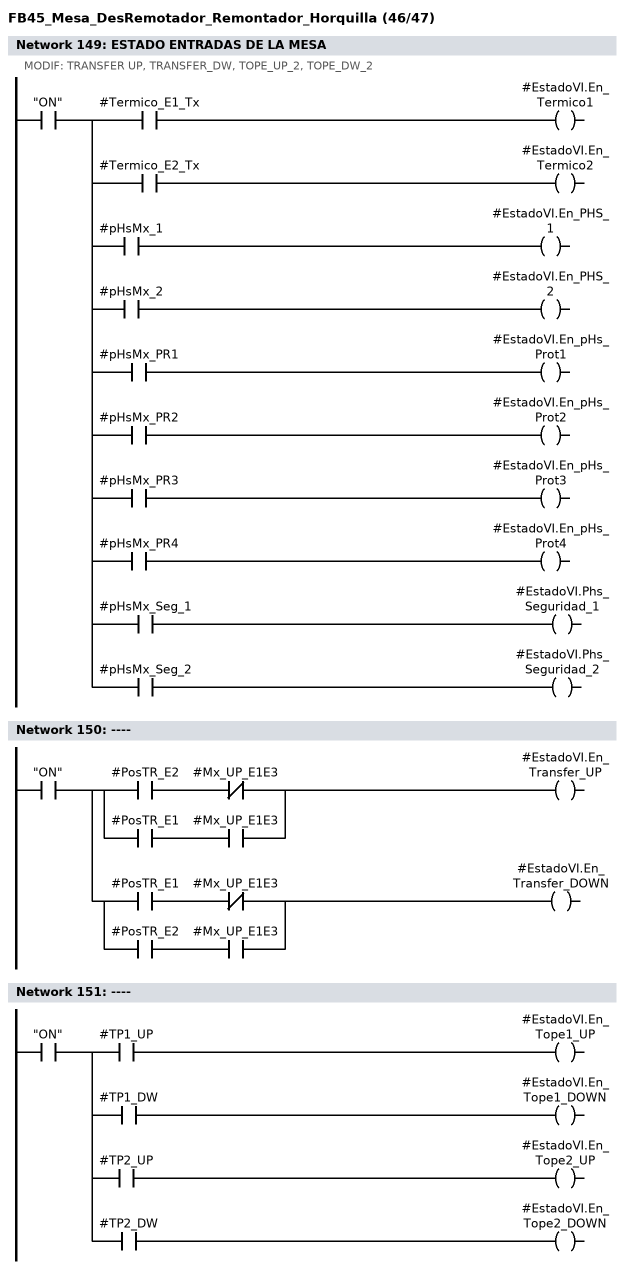
   RUNG wire#powerrail
      Contact( "ON" )
      wire#w1
      Contact( #Termico_E1_Tx )
      Coil( #EstadoVI.En_Termico1 )
   END_RUNG
   RUNG wire#w1
      Contact( #Termico_E2_Tx )
      Coil( #EstadoVI.En_Termico2 )
   END_RUNG
   RUNG wire#w1
      Contact( #pHsMx_1 )
      Coil( #EstadoVI.En_PHS_1 )
   END_RUNG
   RUNG wire#w1
      Contact( #pHsMx_2 )
      Coil( #EstadoVI.En_PHS_2 )
   END_RUNG
   RUNG wire#w1
      Contact( #pHsMx_PR1 )
      Coil( #EstadoVI.En_pHs_Prot1 )
   END_RUNG
   RUNG wire#w1
      Contact( #pHsMx_PR2 )
      Coil( #EstadoVI.En_pHs_Prot2 )
   END_RUNG
   RUNG wire#w1
      Contact( #pHsMx_PR3 )
      Coil( #EstadoVI.En_pHs_Prot3 )
   END_RUNG
   RUNG wire#w1
      Contact( #pHsMx_PR4 )
      Coil( #EstadoVI.En_pHs_Prot4 )
   END_RUNG
   RUNG wire#w1
      Contact( #pHsMx_Seg_1 )
      Coil( #EstadoVI.Phs_Seguridad_1 )
   END_RUNG
   RUNG wire#w1
      Contact( #pHsMx_Seg_2 )
      Coil( #EstadoVI.Phs_Seguridad_2 )
   END_RUNG
   // the same network as SCL:
   #EstadoVI.En_Termico1 := "ON" AND #Termico_E1_Tx;
   #EstadoVI.En_Termico2 := "ON" AND #Termico_E2_Tx;
   #EstadoVI.En_PHS_1 := "ON" AND #pHsMx_1;
   #EstadoVI.En_PHS_2 := "ON" AND #pHsMx_2;
   #EstadoVI.En_pHs_Prot1 := "ON" AND #pHsMx_PR1;
   #EstadoVI.En_pHs_Prot2 := "ON" AND #pHsMx_PR2;
   #EstadoVI.En_pHs_Prot3 := "ON" AND #pHsMx_PR3;
   #EstadoVI.En_pHs_Prot4 := "ON" AND #pHsMx_PR4;
   #EstadoVI.Phs_Seguridad_1 := "ON" AND #pHsMx_Seg_1;
   #EstadoVI.Phs_Seguridad_2 := "ON" AND #pHsMx_Seg_2;
END_REGION

REGION Network 150: ----
   RUNG wire#powerrail
      Contact( "ON" )
      wire#w1
      Contact( #PosTR_E2 )
      I_Contact( #Mx_UP_E1E3 )
      wire#w2
      Coil( #EstadoVI.En_Transfer_UP )
   END_RUNG
   RUNG wire#w1
      Contact( #PosTR_E1 )
      Contact( #Mx_UP_E1E3 )
   END_RUNG wire#w2
   RUNG wire#w1
      Contact( #PosTR_E1 )
      I_Contact( #Mx_UP_E1E3 )
      wire#w3
      Coil( #EstadoVI.En_Transfer_DOWN )
   END_RUNG
   RUNG wire#w1
      Contact( #PosTR_E2 )
      Contact( #Mx_UP_E1E3 )
   END_RUNG wire#w3
   // the same network as SCL:
   #EstadoVI.En_Transfer_UP := "ON" AND ((#PosTR_E2 AND NOT #Mx_UP_E1E3) OR (#PosTR_E1 AND #Mx_UP_E1E3));
   #EstadoVI.En_Transfer_DOWN := "ON" AND ((#PosTR_E1 AND NOT #Mx_UP_E1E3) OR (#PosTR_E2 AND #Mx_UP_E1E3));
END_REGION

REGION Network 151: ----
   RUNG wire#powerrail
      Contact( "ON" )
      wire#w1
      Contact( #TP1_UP )
      Coil( #EstadoVI.En_Tope1_UP )
   END_RUNG
   RUNG wire#w1
      Contact( #TP1_DW )
      Coil( #EstadoVI.En_Tope1_DOWN )
   END_RUNG
   RUNG wire#w1
      Contact( #TP2_UP )
      Coil( #EstadoVI.En_Tope2_UP )
   END_RUNG
   RUNG wire#w1
      Contact( #TP2_DW )
      Coil( #EstadoVI.En_Tope2_DOWN )
   END_RUNG
   // the same network as SCL:
   #EstadoVI.En_Tope1_UP := "ON" AND #TP1_UP;
   #EstadoVI.En_Tope1_DOWN := "ON" AND #TP1_DW;
   #EstadoVI.En_Tope2_UP := "ON" AND #TP2_UP;
   #EstadoVI.En_Tope2_DOWN := "ON" AND #TP2_DW;
END_REGION

REGION Network 152: SALIDAS DE LA MESA
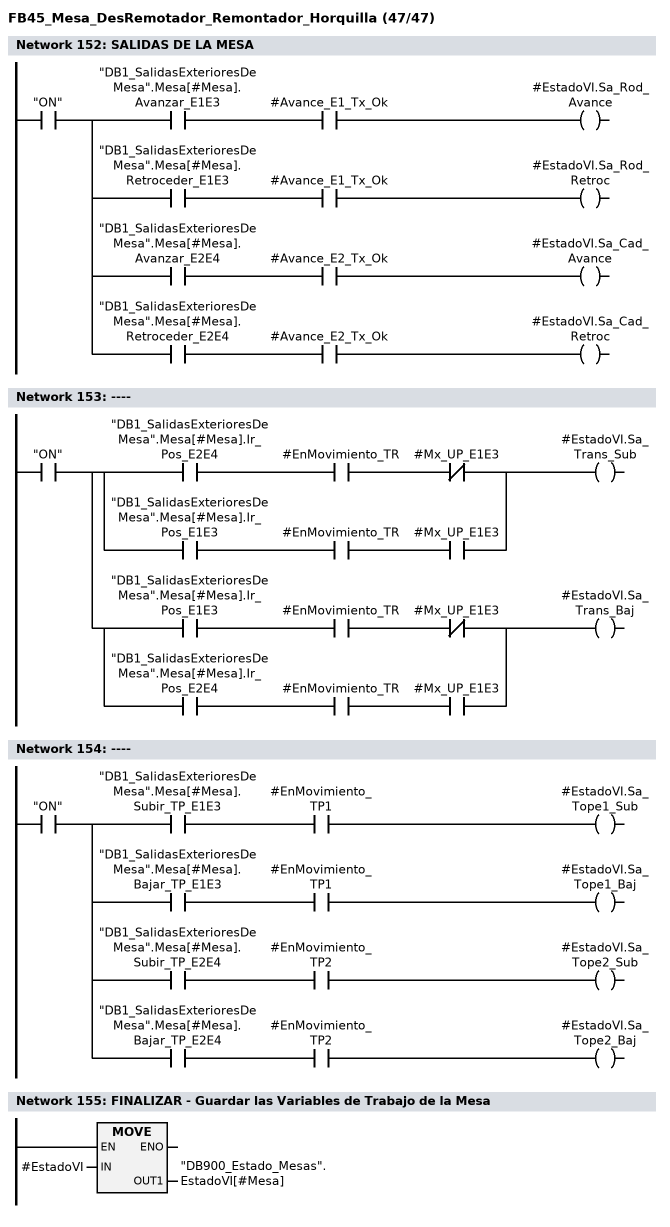
   RUNG wire#powerrail
      Contact( "ON" )
      wire#w1
      Contact( "DB1_SalidasExterioresDeMesa".Mesa[#Mesa].Avanzar_E1E3 )
      Contact( #Avance_E1_Tx_Ok )
      Coil( #EstadoVI.Sa_Rod_Avance )
   END_RUNG
   RUNG wire#w1
      Contact( "DB1_SalidasExterioresDeMesa".Mesa[#Mesa].Retroceder_E1E3 )
      Contact( #Avance_E1_Tx_Ok )
      Coil( #EstadoVI.Sa_Rod_Retroc )
   END_RUNG
   RUNG wire#w1
      Contact( "DB1_SalidasExterioresDeMesa".Mesa[#Mesa].Avanzar_E2E4 )
      Contact( #Avance_E2_Tx_Ok )
      Coil( #EstadoVI.Sa_Cad_Avance )
   END_RUNG
   RUNG wire#w1
      Contact( "DB1_SalidasExterioresDeMesa".Mesa[#Mesa].Retroceder_E2E4 )
      Contact( #Avance_E2_Tx_Ok )
      Coil( #EstadoVI.Sa_Cad_Retroc )
   END_RUNG
   // the same network as SCL:
   #EstadoVI.Sa_Rod_Avance := "ON" AND "DB1_SalidasExterioresDeMesa".Mesa[#Mesa].Avanzar_E1E3 AND #Avance_E1_Tx_Ok;
   #EstadoVI.Sa_Rod_Retroc := "ON" AND "DB1_SalidasExterioresDeMesa".Mesa[#Mesa].Retroceder_E1E3 AND #Avance_E1_Tx_Ok;
   #EstadoVI.Sa_Cad_Avance := "ON" AND "DB1_SalidasExterioresDeMesa".Mesa[#Mesa].Avanzar_E2E4 AND #Avance_E2_Tx_Ok;
   #EstadoVI.Sa_Cad_Retroc := "ON" AND "DB1_SalidasExterioresDeMesa".Mesa[#Mesa].Retroceder_E2E4 AND #Avance_E2_Tx_Ok;
END_REGION

REGION Network 153: ----
   RUNG wire#powerrail
      Contact( "ON" )
      wire#w1
      Contact( "DB1_SalidasExterioresDeMesa".Mesa[#Mesa].Ir_Pos_E2E4 )
      Contact( #EnMovimiento_TR )
      I_Contact( #Mx_UP_E1E3 )
      wire#w2
      Coil( #EstadoVI.Sa_Trans_Sub )
   END_RUNG
   RUNG wire#w1
      Contact( "DB1_SalidasExterioresDeMesa".Mesa[#Mesa].Ir_Pos_E1E3 )
      Contact( #EnMovimiento_TR )
      Contact( #Mx_UP_E1E3 )
   END_RUNG wire#w2
   RUNG wire#w1
      Contact( "DB1_SalidasExterioresDeMesa".Mesa[#Mesa].Ir_Pos_E1E3 )
      Contact( #EnMovimiento_TR )
      I_Contact( #Mx_UP_E1E3 )
      wire#w3
      Coil( #EstadoVI.Sa_Trans_Baj )
   END_RUNG
   RUNG wire#w1
      Contact( "DB1_SalidasExterioresDeMesa".Mesa[#Mesa].Ir_Pos_E2E4 )
      Contact( #EnMovimiento_TR )
      Contact( #Mx_UP_E1E3 )
   END_RUNG wire#w3
   // the same network as SCL:
   #EstadoVI.Sa_Trans_Sub := "ON" AND (("DB1_SalidasExterioresDeMesa".Mesa[#Mesa].Ir_Pos_E2E4 AND #EnMovimiento_TR AND NOT #Mx_UP_E1E3) OR ("DB1_SalidasExterioresDeMesa".Mesa[#Mesa].Ir_Pos_E1E3 AND #EnMovimiento_TR AND #Mx_UP_E1E3));
   #EstadoVI.Sa_Trans_Baj := "ON" AND (("DB1_SalidasExterioresDeMesa".Mesa[#Mesa].Ir_Pos_E1E3 AND #EnMovimiento_TR AND NOT #Mx_UP_E1E3) OR ("DB1_SalidasExterioresDeMesa".Mesa[#Mesa].Ir_Pos_E2E4 AND #EnMovimiento_TR AND #Mx_UP_E1E3));
END_REGION

REGION Network 154: ----
   RUNG wire#powerrail
      Contact( "ON" )
      wire#w1
      Contact( "DB1_SalidasExterioresDeMesa".Mesa[#Mesa].Subir_TP_E1E3 )
      Contact( #EnMovimiento_TP1 )
      Coil( #EstadoVI.Sa_Tope1_Sub )
   END_RUNG
   RUNG wire#w1
      Contact( "DB1_SalidasExterioresDeMesa".Mesa[#Mesa].Bajar_TP_E1E3 )
      Contact( #EnMovimiento_TP1 )
      Coil( #EstadoVI.Sa_Tope1_Baj )
   END_RUNG
   RUNG wire#w1
      Contact( "DB1_SalidasExterioresDeMesa".Mesa[#Mesa].Subir_TP_E2E4 )
      Contact( #EnMovimiento_TP2 )
      Coil( #EstadoVI.Sa_Tope2_Sub )
   END_RUNG
   RUNG wire#w1
      Contact( "DB1_SalidasExterioresDeMesa".Mesa[#Mesa].Bajar_TP_E2E4 )
      Contact( #EnMovimiento_TP2 )
      Coil( #EstadoVI.Sa_Tope2_Baj )
   END_RUNG
   // the same network as SCL:
   #EstadoVI.Sa_Tope1_Sub := "ON" AND "DB1_SalidasExterioresDeMesa".Mesa[#Mesa].Subir_TP_E1E3 AND #EnMovimiento_TP1;
   #EstadoVI.Sa_Tope1_Baj := "ON" AND "DB1_SalidasExterioresDeMesa".Mesa[#Mesa].Bajar_TP_E1E3 AND #EnMovimiento_TP1;
   #EstadoVI.Sa_Tope2_Sub := "ON" AND "DB1_SalidasExterioresDeMesa".Mesa[#Mesa].Subir_TP_E2E4 AND #EnMovimiento_TP2;
   #EstadoVI.Sa_Tope2_Baj := "ON" AND "DB1_SalidasExterioresDeMesa".Mesa[#Mesa].Bajar_TP_E2E4 AND #EnMovimiento_TP2;
END_REGION

REGION Network 155: FINALIZAR - Guardar las Variables de Trabajo de la Mesa
   RUNG wire#powerrail
      Move(in := #EstadoVI, out1 => "DB900_Estado_Mesas".EstadoVI[#Mesa])
   END_RUNG
   // the same network as SCL:
   "DB900_Estado_Mesas".EstadoVI[#Mesa] := #EstadoVI;
END_REGION
END_FUNCTION_BLOCK

FUNCTION_BLOCK "FB461_CRTL_TR_TP_E1E2_S34_Pres"   // FB461, LAD
TITLE = Control del Ramal de Salidas
{ S7_Optimized_Access := 'FALSE' }
AUTHOR : TLigero
NAME : 20180827
VERSION : 3.3
// stored: AutoNumber false, SetENOAutomatically false
   VAR_INPUT
      Mesa : UInt;   // Número de mesa
      En_Tension : Bool;
      pHsMx : Bool;   // pHs de presencia de la Mesa
      TP1_Up : Bool;   // TP1 Arriba. E1 >> S3. si no hay tope poner ON
      TP1_Down : Bool;   // TP1 Abajo. E1 >> S3. si no hay tope poner ON
      TP2_Up : Bool;   // TP1 Arriba. E2 >> S4. si no hay tope poner ON
      TP2_Down : Bool;   // TP1 Abajo. E2 >> S4. si no hay tope poner ON
      PosTR_E1 : Bool;   // Posicion del TR en E1E3
      PosTR_E2 : Bool;   // Posicion del TR en E2E4
      Termico_13 : Bool;   // Proteccion del Tx en E1E3
      Termico_24 : Bool;   // Proteccion del Tx en E2E4
      Avance_13 : Bool;   // Avance del Tx en E1E3
      Avance_24 : Bool;   // Avance del Tx en E2E4
      PTF_Sal_M3 : Bool;   // S3 >> Mesa Siguiente PTF
      NXT_Avance_S3 : Bool;   // S3 >> Mesa Siguiente avanzando
      PTF_Sal_M4 : Bool;   // S4 >> Mesa Siguiente PTF
      NXT_Avance_S4 : Bool;   // S4 >> Mesa Siguiente avanzando
      F_EnvMens_Mx : Bool;   // Fin de Envio de Mensaje
      Mx_Bloq_Activo_S4 : Bool;   // Bloqueo Activo de la Mesa
      Mx_FlujoPrin_S4 : Bool;   // El flujo principal es Saliendo por S4
      AVTF_Ent_M1 : Bool;   // E1 >> Mesa Anterior AVTF
      AVTF_Ent_M2 : Bool;   // E2 >> Mesa Anterior AVTF
      Num_Cruce : UInt;   // Número de cruce.
      DB_FIFO_Cruce : UInt := 213;   // DB de la FIFO de ordenes del cruce
      Long_FIFO_Cruce : UInt := 1;   // Longitut de la FIFO de ordenes del cruce
      ValorOrden_S4 : Word := 16#81;   // Con que orden entra por S4
      MesaS3 : UInt;   // Número de mesa por S3
      MesaS4 : UInt;   // Número de mesa por S4
      V_CNT_pHsMx_E1 : UDInt := 500;   // Valor de presencia por E1 en ms
      V_CNT_pHsMx_E2 : UDInt := 500;   // Valor de presencia por E2 en ms
      V_CNT_ApHsMx_S3 : UDInt := 500;   // Valor de Ausencia por S3 en ms
      V_CNT_ApHsMx_S4 : UDInt := 500;   // Valor de Ausencia por S4 en ms
      V_TOut_Tx_Mx : UDInt := 3000;   // TimeOut de Atasco en ms
      V_Vaciado : UDInt := 3000;   // Valor de vaciado en ms
      V_Paro : UDInt := 5000;   // tiempo que avanza el transportador sin aviso hasta que se para (ms)
      V_TOut_TP : UDInt;   // TimeOut de Tope en ms
      V_TOut_TR : UDInt;   // TimeOut de Transfer en ms
   END_VAR
   VAR_OUTPUT
      P_EnvMens_PMx : Bool;   // Permiso de Enviar Mensaje de Presencia
      Etiqueta_Jdt : UDInt;   // Etiqueta que ha sido leida
      Orden_Ejecutada_Jdt : UInt;   // Orden que se ha ejecutado
      PTF_Ent_M1 : Bool;   // E1 >> Mesa Anterior PTF
      PTF_Ent_M2 : Bool;   // E2 >> Mesa Anterior PTF
      AVTF_Sal_M3 : Bool;   // S3 >> Mesa Siguiente AVTF
      NXT_Descarga_Act_S3 : Bool;   // S3 >> Mesa Siguiente descarga activa
      AVTF_Sal_M4 : Bool;   // S4 >> Mesa Siguiente AVTF
      NXT_Descarga_Act_S4 : Bool;   // S4 >> Mesa Siguiente descarga activa
   END_VAR
   VAR
      T1_ET00 : Bool;
      T1_ET01 : Bool;
      T1_ET02 : Bool;
      T1_ET03 : Bool;
      T1_ET10 : Bool;
      T1_ET11 : Bool;
      T1_ET20 : Bool;
      T1_ET21 : Bool;
      T1_ET50 : Bool;
      T1_ET60 : Bool;
      T1_ET61 : Bool;
      T1_ET70 : Bool;
      T1_ET110 : Bool;
      T1_ET111 : Bool;
      T1_ET112 : Bool;
      Simul_Mx : Bool;
      maux_fp_disparo_e1 : Bool;
      maux_fp_disparo_e2 : Bool;
      FIFO_OK : Bool;
      TRANS_OK : Bool;
      O_Bloqueo : Bool;
      Ultima_entra_de_E2 : Bool;
      Ultima_entra_de_E1 : Bool;
      Err_Detec_PHS : Bool;
      FN_ET02 : Bool;
      TIM_Vaciado_Q : Bool;
      TMP_Paro_Q : Bool;
      TMP_Presencia_E1 : UDInt;
      TMP_Aus_S4 : UDInt;
      TMP_Aus_S3 : UDInt;
      CNT_pHs_E2 : UDInt;
      TIM_Vaciado : UDInt;
      TMP_Paro : UDInt;
      TMP_tout_Tope_S3 : UDInt;
      TMP_tout_Tope_S4 : UDInt;
      TMP_tout_transfer : UDInt;
      TMP_Err_Tout : UDInt;
      TMP_En_Tension : UDInt;
      Datos_Scanner { S7_SetPoint := 'True'} : "ROUT_Orden_Fifo_Scanner";
   END_VAR
   VAR_TEMP
      EstadoZona : "EstadoZona";   // Estado de Zona de la Mesa
      EstadoVI : "EstadosMesa";   // Estado del Vehiculo Inteliguente de la Mesa
      ConfigFB : "UDT_ConfigFB";   // Configuracion de la FB de la Mesa
      MA_SubirTP : Bool;
      O_Sal_S3 : Bool;
      O_Sal_S4 : Bool;
      O_Vaciar : Bool;
      Moti_ERRO : Bool;
      Moti_NENC : Bool;
      Moti_NORM : Bool;
      Moti_INIC : Bool;
      Parar_E1 : Bool;
      tmp_Aus_S4_Q : Bool;
      tmp_pHs_E2_Q : Bool;
      tmp_pHs_E1_Q : Bool;
      tmp_pHs_S3_Q : Bool;
      TMP_Err_Tout_Q : Bool;
      timeout_tope_s3 : Bool;
      timeout_tope_s4 : Bool;
      timeout_transfer : Bool;
      ok_tension : Bool;
      Aux_W_Moti : Word;
      Libre : UInt;
      INT_ORDEN : UInt;
      Aux_W_Orden : Word;
      I_Ord_Filtrada : UInt;
      I_V_Ord_S4 : UInt;
   END_VAR
   VAR_TEMP   // added for the SCL form of the ladder/FBD networks
      _w1 : Bool;
      _w2 : Bool;
      _w3 : Bool;
      _w4 : Bool;
      _w5 : Bool;
      _w6 : Bool;
   END_VAR
BEGIN

REGION Network 1: INICIALIZAR - Recoger las Variables de Estado de la Mesa
   // Se recoge - Estado_CBx
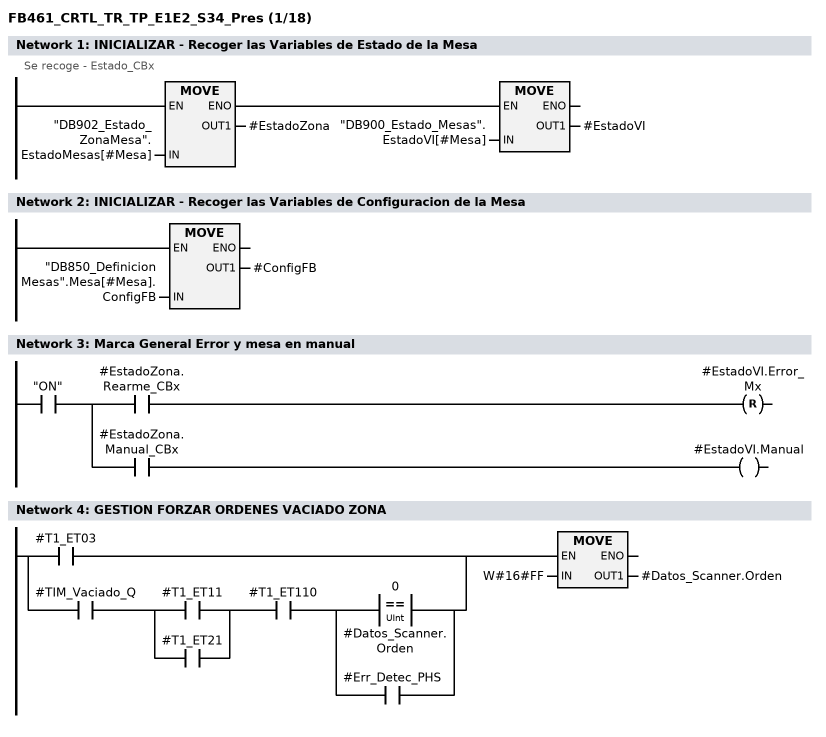
   RUNG wire#powerrail
      Move(in := "DB902_Estado_ZonaMesa".EstadoMesas[#Mesa], out1 => #EstadoZona)
      Move(in := "DB900_Estado_Mesas".EstadoVI[#Mesa], out1 => #EstadoVI)
   END_RUNG
   // the same network as SCL:
   #EstadoZona := "DB902_Estado_ZonaMesa".EstadoMesas[#Mesa];
   #EstadoVI := "DB900_Estado_Mesas".EstadoVI[#Mesa];
END_REGION

REGION Network 2: INICIALIZAR - Recoger las Variables de Configuracion de la Mesa
   RUNG wire#powerrail
      Move(in := "DB850_DefinicionMesas".Mesa[#Mesa].ConfigFB, out1 => #ConfigFB)
   END_RUNG
   // the same network as SCL:
   #ConfigFB := "DB850_DefinicionMesas".Mesa[#Mesa].ConfigFB;
END_REGION

REGION Network 3: Marca General Error y mesa en manual
   RUNG wire#powerrail
      Contact( "ON" )
      wire#w1
      Contact( #EstadoZona.Rearme_CBx )
      R_Coil( #EstadoVI.Error_Mx )
   END_RUNG
   RUNG wire#w1
      Contact( #EstadoZona.Manual_CBx )
      Coil( #EstadoVI.Manual )
   END_RUNG
   // the same network as SCL:
   IF "ON" AND #EstadoZona.Rearme_CBx THEN #EstadoVI.Error_Mx := FALSE; END_IF;
   #EstadoVI.Manual := "ON" AND #EstadoZona.Manual_CBx;
END_REGION

REGION Network 4: GESTION FORZAR ORDENES VACIADO ZONA
   RUNG wire#powerrail
      Contact( #T1_ET03 )
      wire#w1
      { S7_GenerateENO := "TRUE" } Move(in := W#16#FF, out1 => #Datos_Scanner.Orden)
   END_RUNG
   RUNG wire#powerrail
      Contact( #TIM_Vaciado_Q )
      wire#w2
      Contact( #T1_ET11 )
      wire#w3
      Contact( #T1_ET110 )
      wire#w4
      { S7_Templates := "SrcType := UInt" } EQ_Contact(in1 := 0, in2 := #Datos_Scanner.Orden)
   END_RUNG wire#w1
   RUNG wire#w2
      Contact( #T1_ET21 )
   END_RUNG wire#w3
   RUNG wire#w4
      Contact( #Err_Detec_PHS )
   END_RUNG wire#w1
   // the same network as SCL:
   IF #T1_ET03 OR (#TIM_Vaciado_Q AND (#T1_ET11 OR #T1_ET21) AND #T1_ET110 AND ((0 = #Datos_Scanner.Orden) OR #Err_Detec_PHS)) THEN
       #Datos_Scanner.Orden := W#16#FF;
   END_IF;
END_REGION

REGION Network 5: Extraccion de orden
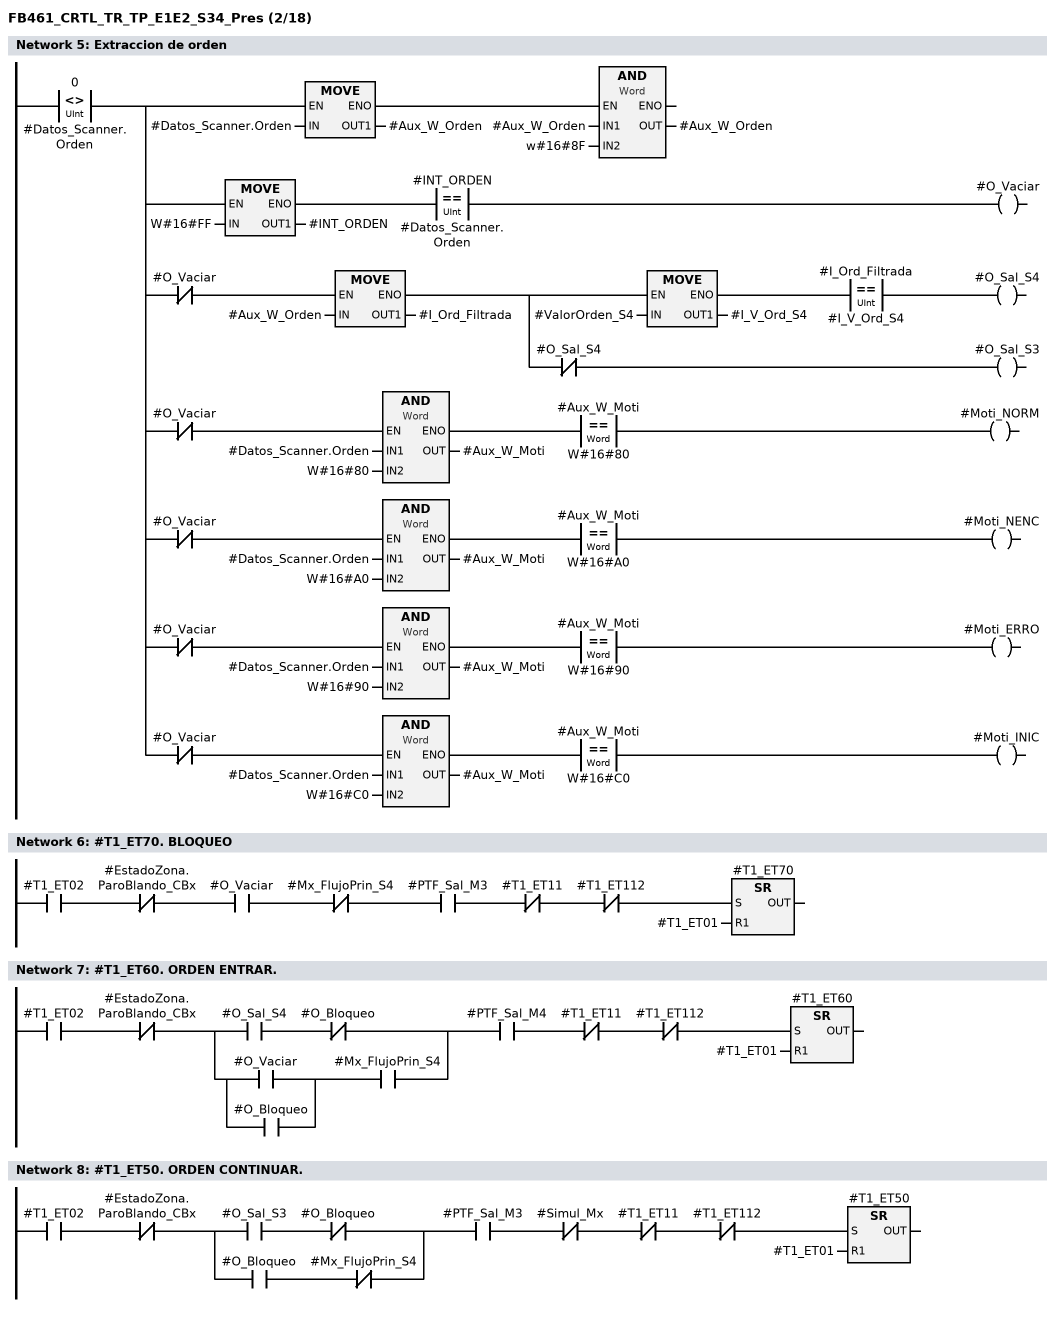
   RUNG wire#powerrail
      { S7_Templates := "SrcType := UInt" } NE_Contact(in1 := 0, in2 := #Datos_Scanner.Orden)
      wire#w1
      { S7_GenerateENO := "TRUE" } Move(in := #Datos_Scanner.Orden, out1 => #Aux_W_Orden)
      { S7_Templates := "SrcType := Word"; S7_GenerateENO := "TRUE" } And(in1 := #Aux_W_Orden, in2 := w#16#8F, out => #Aux_W_Orden)
   END_RUNG
   RUNG wire#w1
      { S7_GenerateENO := "TRUE" } Move(in := W#16#FF, out1 => #INT_ORDEN)
      { S7_Templates := "SrcType := UInt" } EQ_Contact(in1 := #INT_ORDEN, in2 := #Datos_Scanner.Orden)
      Coil( #O_Vaciar )
   END_RUNG
   RUNG wire#w1
      I_Contact( #O_Vaciar )
      { S7_GenerateENO := "TRUE" } Move(in := #Aux_W_Orden, out1 => #I_Ord_Filtrada)
      wire#w2
      { S7_GenerateENO := "TRUE" } Move(in := #ValorOrden_S4, out1 => #I_V_Ord_S4)
      { S7_Templates := "SrcType := UInt" } EQ_Contact(in1 := #I_Ord_Filtrada, in2 := #I_V_Ord_S4)
      Coil( #O_Sal_S4 )
   END_RUNG
   RUNG wire#w2
      I_Contact( #O_Sal_S4 )
      Coil( #O_Sal_S3 )
   END_RUNG
   RUNG wire#w1
      I_Contact( #O_Vaciar )
      { S7_Templates := "SrcType := Word"; S7_GenerateENO := "TRUE" } And(in1 := #Datos_Scanner.Orden, in2 := W#16#80, out => #Aux_W_Moti)
      { S7_Templates := "SrcType := Word" } EQ_Contact(in1 := #Aux_W_Moti, in2 := W#16#80)
      Coil( #Moti_NORM )
   END_RUNG
   RUNG wire#w1
      I_Contact( #O_Vaciar )
      { S7_Templates := "SrcType := Word"; S7_GenerateENO := "TRUE" } And(in1 := #Datos_Scanner.Orden, in2 := W#16#A0, out => #Aux_W_Moti)
      { S7_Templates := "SrcType := Word" } EQ_Contact(in1 := #Aux_W_Moti, in2 := W#16#A0)
      Coil( #Moti_NENC )
   END_RUNG
   RUNG wire#w1
      I_Contact( #O_Vaciar )
      { S7_Templates := "SrcType := Word"; S7_GenerateENO := "TRUE" } And(in1 := #Datos_Scanner.Orden, in2 := W#16#90, out => #Aux_W_Moti)
      { S7_Templates := "SrcType := Word" } EQ_Contact(in1 := #Aux_W_Moti, in2 := W#16#90)
      Coil( #Moti_ERRO )
   END_RUNG
   RUNG wire#w1
      I_Contact( #O_Vaciar )
      { S7_Templates := "SrcType := Word"; S7_GenerateENO := "TRUE" } And(in1 := #Datos_Scanner.Orden, in2 := W#16#C0, out => #Aux_W_Moti)
      { S7_Templates := "SrcType := Word" } EQ_Contact(in1 := #Aux_W_Moti, in2 := W#16#C0)
      Coil( #Moti_INIC )
   END_RUNG
   // the same network as SCL:
   // ENO of a box is taken as its EN; it also drops when the box reports an error
   #_w1 := 0 <> #Datos_Scanner.Orden;
   IF #_w1 THEN
       #Aux_W_Orden := #Datos_Scanner.Orden;
       #Aux_W_Orden := #Aux_W_Orden AND w#16#8F;
       #INT_ORDEN := W#16#FF;
   END_IF;
   #O_Vaciar := #_w1 AND (#INT_ORDEN = #Datos_Scanner.Orden);
   #_w2 := #_w1 AND NOT #O_Vaciar;
   IF #_w2 THEN
       #I_Ord_Filtrada := #Aux_W_Orden;
       #I_V_Ord_S4 := #ValorOrden_S4;
   END_IF;
   #O_Sal_S4 := #_w2 AND (#I_Ord_Filtrada = #I_V_Ord_S4);
   #O_Sal_S3 := #_w2 AND NOT #O_Sal_S4;
   #_w3 := #_w1 AND NOT #O_Vaciar;
   IF #_w3 THEN #Aux_W_Moti := #Datos_Scanner.Orden AND W#16#80; END_IF;
   #Moti_NORM := #_w3 AND (#Aux_W_Moti = W#16#80);
   #_w4 := #_w1 AND NOT #O_Vaciar;
   IF #_w4 THEN #Aux_W_Moti := #Datos_Scanner.Orden AND W#16#A0; END_IF;
   #Moti_NENC := #_w4 AND (#Aux_W_Moti = W#16#A0);
   #_w5 := #_w1 AND NOT #O_Vaciar;
   IF #_w5 THEN #Aux_W_Moti := #Datos_Scanner.Orden AND W#16#90; END_IF;
   #Moti_ERRO := #_w5 AND (#Aux_W_Moti = W#16#90);
   #_w6 := #_w1 AND NOT #O_Vaciar;
   IF #_w6 THEN #Aux_W_Moti := #Datos_Scanner.Orden AND W#16#C0; END_IF;
   #Moti_INIC := #_w6 AND (#Aux_W_Moti = W#16#C0);
END_REGION

REGION Network 6: #T1_ET70. BLOQUEO
   RUNG wire#powerrail
      Contact( #T1_ET02 )
      I_Contact( #EstadoZona.ParoBlando_CBx )
      Contact( #O_Vaciar )
      I_Contact( #Mx_FlujoPrin_S4 )
      Contact( #PTF_Sal_M3 )
      I_Contact( #T1_ET11 )
      I_Contact( #T1_ET112 )
      S_SR(operand := #T1_ET70, r1 := #T1_ET01)
   END_RUNG
   // the same network as SCL:
   IF #T1_ET02 AND NOT #EstadoZona.ParoBlando_CBx AND #O_Vaciar AND NOT #Mx_FlujoPrin_S4 AND #PTF_Sal_M3 AND NOT #T1_ET11 AND NOT #T1_ET112 THEN
       #T1_ET70 := TRUE;   // SR flip-flop
   END_IF;
   IF #T1_ET01 THEN #T1_ET70 := FALSE; END_IF;
END_REGION

REGION Network 7: #T1_ET60. ORDEN ENTRAR.
   RUNG wire#powerrail
      Contact( #T1_ET02 )
      I_Contact( #EstadoZona.ParoBlando_CBx )
      wire#w1
      Contact( #O_Sal_S4 )
      I_Contact( #O_Bloqueo )
      wire#w2
      Contact( #PTF_Sal_M4 )
      I_Contact( #T1_ET11 )
      I_Contact( #T1_ET112 )
      S_SR(operand := #T1_ET60, r1 := #T1_ET01)
   END_RUNG
   RUNG wire#w1
      Contact( #O_Vaciar )
      wire#w3
      Contact( #Mx_FlujoPrin_S4 )
   END_RUNG wire#w2
   RUNG wire#w1
      Contact( #O_Bloqueo )
   END_RUNG wire#w3
   // the same network as SCL:
   IF #T1_ET02 AND NOT #EstadoZona.ParoBlando_CBx AND ((#O_Sal_S4 AND NOT #O_Bloqueo) OR ((#O_Vaciar OR #O_Bloqueo) AND #Mx_FlujoPrin_S4)) AND #PTF_Sal_M4 AND NOT #T1_ET11 AND NOT #T1_ET112 THEN
       #T1_ET60 := TRUE;   // SR flip-flop
   END_IF;
   IF #T1_ET01 THEN #T1_ET60 := FALSE; END_IF;
END_REGION

REGION Network 8: #T1_ET50. ORDEN CONTINUAR.
   RUNG wire#powerrail
      Contact( #T1_ET02 )
      I_Contact( #EstadoZona.ParoBlando_CBx )
      wire#w1
      Contact( #O_Sal_S3 )
      I_Contact( #O_Bloqueo )
      wire#w2
      Contact( #PTF_Sal_M3 )
      I_Contact( #Simul_Mx )
      I_Contact( #T1_ET11 )
      I_Contact( #T1_ET112 )
      S_SR(operand := #T1_ET50, r1 := #T1_ET01)
   END_RUNG
   RUNG wire#w1
      Contact( #O_Bloqueo )
      I_Contact( #Mx_FlujoPrin_S4 )
   END_RUNG wire#w2
   // the same network as SCL:
   IF #T1_ET02 AND NOT #EstadoZona.ParoBlando_CBx AND ((#O_Sal_S3 AND NOT #O_Bloqueo) OR (#O_Bloqueo AND NOT #Mx_FlujoPrin_S4)) AND #PTF_Sal_M3 AND NOT #Simul_Mx AND NOT #T1_ET11 AND NOT #T1_ET112 THEN
       #T1_ET50 := TRUE;   // SR flip-flop
   END_IF;
   IF #T1_ET01 THEN #T1_ET50 := FALSE; END_IF;
END_REGION

REGION Network 9: #T1_ET02. ESTADO REPOSO CARGADA.
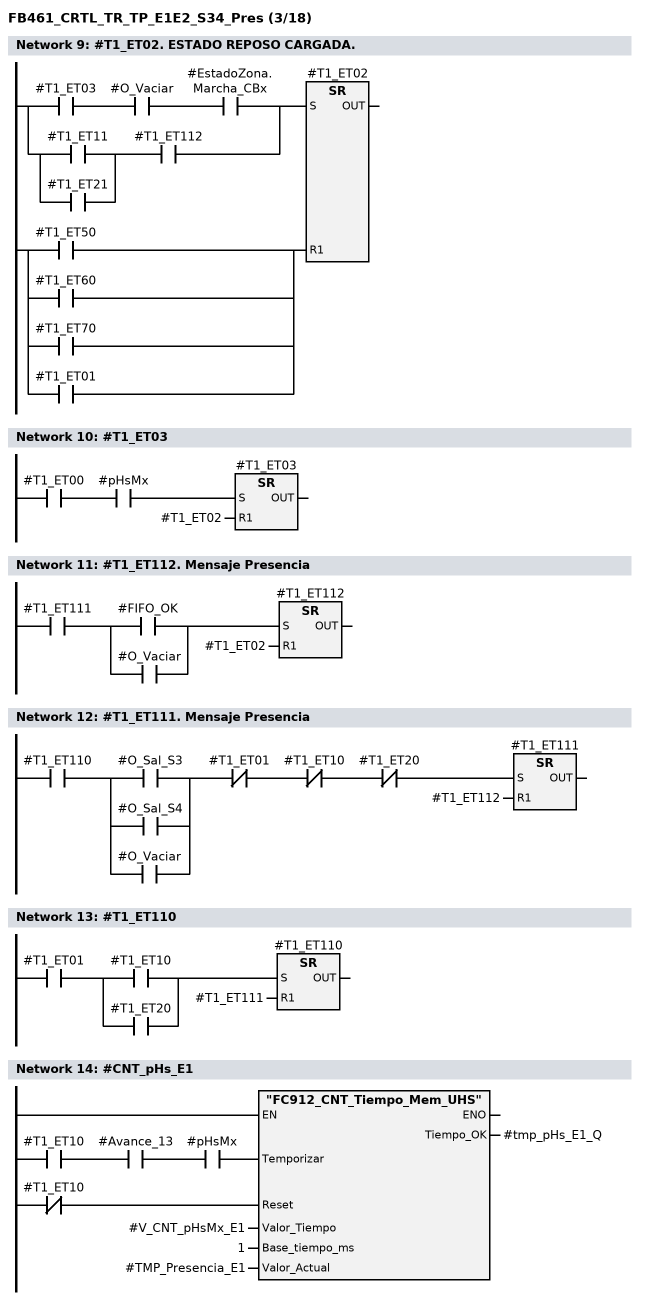
   RUNG wire#powerrail
      Contact( #T1_ET03 )
      Contact( #O_Vaciar )
      Contact( #EstadoZona.Marcha_CBx )
      wire#w1
      S_SR(operand := #T1_ET02, r1 := wire#w3)
   END_RUNG
   RUNG wire#powerrail
      Contact( #T1_ET11 )
      wire#w2
      Contact( #T1_ET112 )
   END_RUNG wire#w1
   RUNG wire#powerrail
      Contact( #T1_ET21 )
   END_RUNG wire#w2
   RUNG wire#powerrail
      Contact( #T1_ET50 )
   END_RUNG wire#w3
   RUNG wire#powerrail
      Contact( #T1_ET60 )
   END_RUNG wire#w3
   RUNG wire#powerrail
      Contact( #T1_ET70 )
   END_RUNG wire#w3
   RUNG wire#powerrail
      Contact( #T1_ET01 )
   END_RUNG wire#w3
   // the same network as SCL:
   IF (#T1_ET03 AND #O_Vaciar AND #EstadoZona.Marcha_CBx) OR ((#T1_ET11 OR #T1_ET21) AND #T1_ET112) THEN
       #T1_ET02 := TRUE;   // SR flip-flop
   END_IF;
   IF #T1_ET50 OR #T1_ET60 OR #T1_ET70 OR #T1_ET01 THEN #T1_ET02 := FALSE; END_IF;
END_REGION

REGION Network 10: #T1_ET03
   RUNG wire#powerrail
      Contact( #T1_ET00 )
      Contact( #pHsMx )
      S_SR(operand := #T1_ET03, r1 := #T1_ET02)
   END_RUNG
   // the same network as SCL:
   IF #T1_ET00 AND #pHsMx THEN
       #T1_ET03 := TRUE;   // SR flip-flop
   END_IF;
   IF #T1_ET02 THEN #T1_ET03 := FALSE; END_IF;
END_REGION

REGION Network 11: #T1_ET112. Mensaje Presencia
   RUNG wire#powerrail
      Contact( #T1_ET111 )
      wire#w1
      Contact( #FIFO_OK )
      wire#w2
      S_SR(operand := #T1_ET112, r1 := #T1_ET02)
   END_RUNG
   RUNG wire#w1
      Contact( #O_Vaciar )
   END_RUNG wire#w2
   // the same network as SCL:
   IF #T1_ET111 AND (#FIFO_OK OR #O_Vaciar) THEN
       #T1_ET112 := TRUE;   // SR flip-flop
   END_IF;
   IF #T1_ET02 THEN #T1_ET112 := FALSE; END_IF;
END_REGION

REGION Network 12: #T1_ET111. Mensaje Presencia
   RUNG wire#powerrail
      Contact( #T1_ET110 )
      wire#w1
      Contact( #O_Sal_S3 )
      wire#w2
      I_Contact( #T1_ET01 )
      I_Contact( #T1_ET10 )
      I_Contact( #T1_ET20 )
      S_SR(operand := #T1_ET111, r1 := #T1_ET112)
   END_RUNG
   RUNG wire#w1
      Contact( #O_Sal_S4 )
   END_RUNG wire#w2
   RUNG wire#w1
      Contact( #O_Vaciar )
   END_RUNG wire#w2
   // the same network as SCL:
   IF #T1_ET110 AND (#O_Sal_S3 OR #O_Sal_S4 OR #O_Vaciar) AND NOT #T1_ET01 AND NOT #T1_ET10 AND NOT #T1_ET20 THEN
       #T1_ET111 := TRUE;   // SR flip-flop
   END_IF;
   IF #T1_ET112 THEN #T1_ET111 := FALSE; END_IF;
END_REGION

REGION Network 13: #T1_ET110
   RUNG wire#powerrail
      Contact( #T1_ET01 )
      wire#w1
      Contact( #T1_ET10 )
      wire#w2
      S_SR(operand := #T1_ET110, r1 := #T1_ET111)
   END_RUNG
   RUNG wire#w1
      Contact( #T1_ET20 )
   END_RUNG wire#w2
   // the same network as SCL:
   IF #T1_ET01 AND (#T1_ET10 OR #T1_ET20) THEN
       #T1_ET110 := TRUE;   // SR flip-flop
   END_IF;
   IF #T1_ET111 THEN #T1_ET110 := FALSE; END_IF;
END_REGION

REGION Network 14: #CNT_pHs_E1
   RUNG wire#powerrail
      "FC912_CNT_Tiempo_Mem_UHS"(Temporizar := wire#w1, Reset := wire#w2, Valor_Tiempo := #V_CNT_pHsMx_E1, Base_tiempo_ms := 1, Valor_Actual := #TMP_Presencia_E1, Tiempo_OK => #tmp_pHs_E1_Q)
   END_RUNG
   RUNG wire#powerrail
      Contact( #T1_ET10 )
      Contact( #Avance_13 )
      Contact( #pHsMx )
   END_RUNG wire#w1
   RUNG wire#powerrail
      I_Contact( #T1_ET10 )
   END_RUNG wire#w2
   // the same network as SCL:
   "FC912_CNT_Tiempo_Mem_UHS"(Temporizar := #T1_ET10 AND #Avance_13 AND #pHsMx,
                           Reset := NOT #T1_ET10,
                           Valor_Tiempo := #V_CNT_pHsMx_E1,
                           Base_tiempo_ms := 1,
                           Valor_Actual := #TMP_Presencia_E1,
                           Tiempo_OK => #tmp_pHs_E1_Q);
END_REGION

REGION Network 15: #CNT_pHs_E2
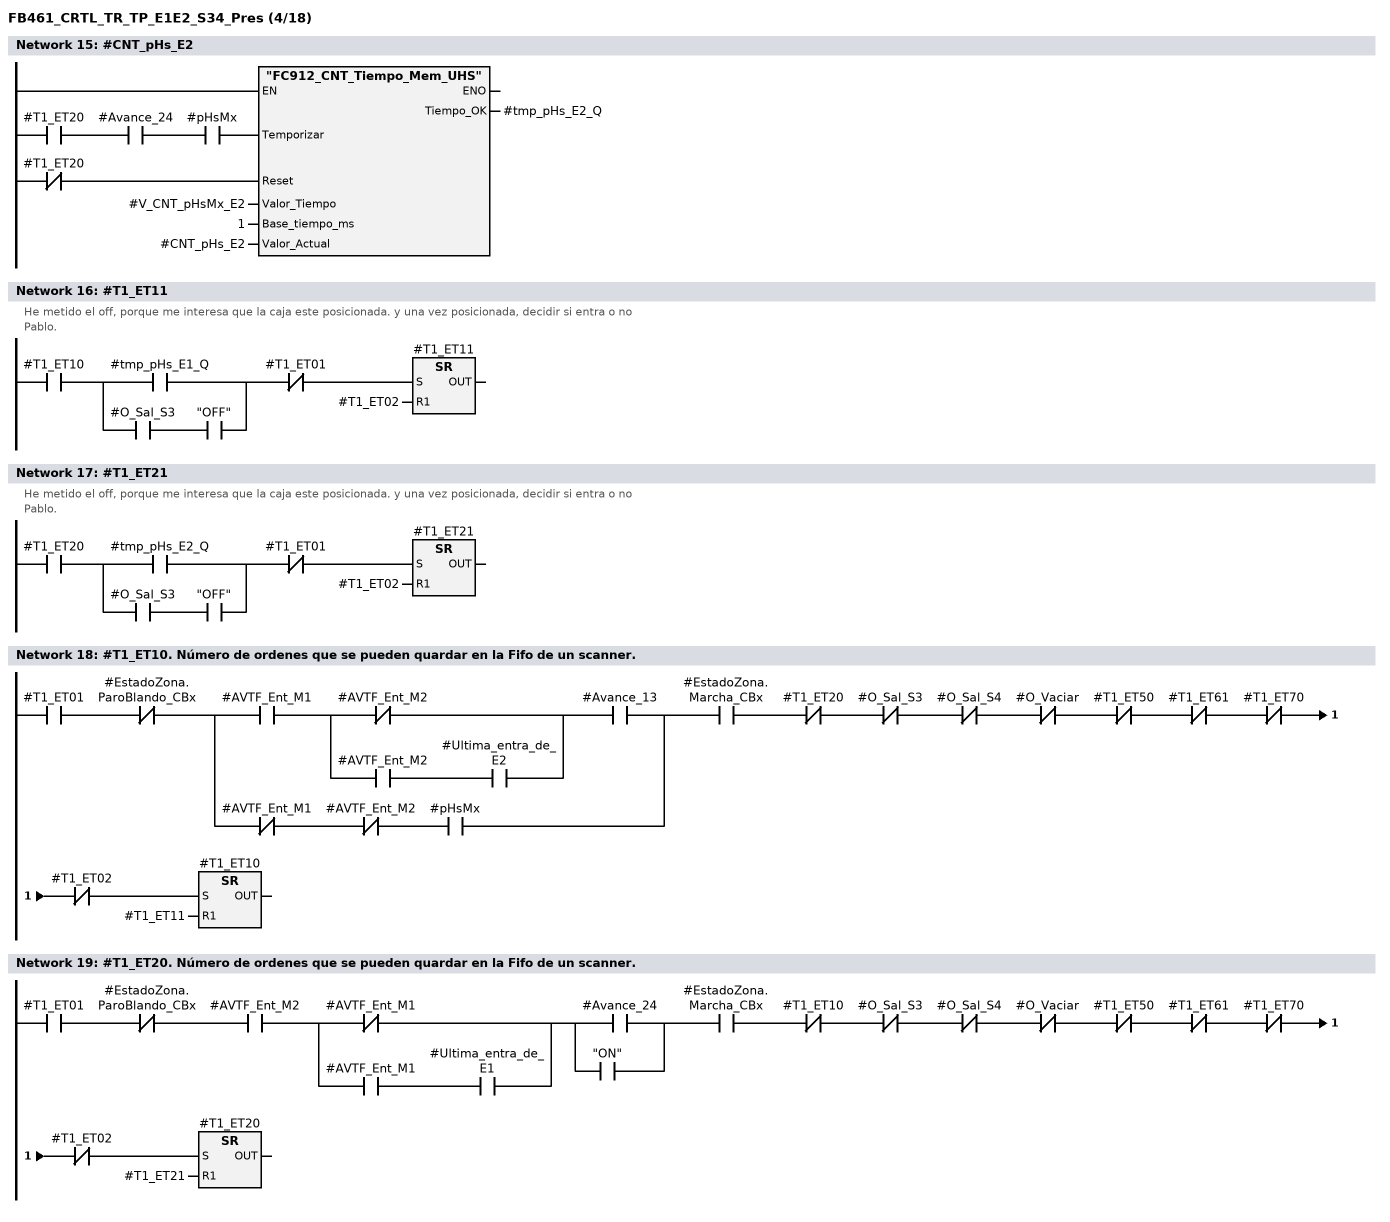
   RUNG wire#powerrail
      "FC912_CNT_Tiempo_Mem_UHS"(Temporizar := wire#w1, Reset := wire#w2, Valor_Tiempo := #V_CNT_pHsMx_E2, Base_tiempo_ms := 1, Valor_Actual := #CNT_pHs_E2, Tiempo_OK => #tmp_pHs_E2_Q)
   END_RUNG
   RUNG wire#powerrail
      Contact( #T1_ET20 )
      Contact( #Avance_24 )
      Contact( #pHsMx )
   END_RUNG wire#w1
   RUNG wire#powerrail
      I_Contact( #T1_ET20 )
   END_RUNG wire#w2
   // the same network as SCL:
   "FC912_CNT_Tiempo_Mem_UHS"(Temporizar := #T1_ET20 AND #Avance_24 AND #pHsMx,
                           Reset := NOT #T1_ET20,
                           Valor_Tiempo := #V_CNT_pHsMx_E2,
                           Base_tiempo_ms := 1,
                           Valor_Actual := #CNT_pHs_E2,
                           Tiempo_OK => #tmp_pHs_E2_Q);
END_REGION

REGION Network 16: #T1_ET11
   // He metido el off, porque me interesa que la caja este posicionada. y una vez posicionada, decidir si entra o no
   // Pablo.
   RUNG wire#powerrail
      Contact( #T1_ET10 )
      wire#w1
      Contact( #tmp_pHs_E1_Q )
      wire#w2
      I_Contact( #T1_ET01 )
      S_SR(operand := #T1_ET11, r1 := #T1_ET02)
   END_RUNG
   RUNG wire#w1
      Contact( #O_Sal_S3 )
      Contact( "OFF" )
   END_RUNG wire#w2
   // the same network as SCL:
   IF #T1_ET10 AND (#tmp_pHs_E1_Q OR (#O_Sal_S3 AND "OFF")) AND NOT #T1_ET01 THEN
       #T1_ET11 := TRUE;   // SR flip-flop
   END_IF;
   IF #T1_ET02 THEN #T1_ET11 := FALSE; END_IF;
END_REGION

REGION Network 17: #T1_ET21
   // He metido el off, porque me interesa que la caja este posicionada. y una vez posicionada, decidir si entra o no
   // Pablo.
   RUNG wire#powerrail
      Contact( #T1_ET20 )
      wire#w1
      Contact( #tmp_pHs_E2_Q )
      wire#w2
      I_Contact( #T1_ET01 )
      S_SR(operand := #T1_ET21, r1 := #T1_ET02)
   END_RUNG
   RUNG wire#w1
      Contact( #O_Sal_S3 )
      Contact( "OFF" )
   END_RUNG wire#w2
   // the same network as SCL:
   IF #T1_ET20 AND (#tmp_pHs_E2_Q OR (#O_Sal_S3 AND "OFF")) AND NOT #T1_ET01 THEN
       #T1_ET21 := TRUE;   // SR flip-flop
   END_IF;
   IF #T1_ET02 THEN #T1_ET21 := FALSE; END_IF;
END_REGION

REGION Network 18: #T1_ET10. Número de ordenes que se pueden quardar en la Fifo de un scanner.
   RUNG wire#powerrail
      Contact( #T1_ET01 )
      I_Contact( #EstadoZona.ParoBlando_CBx )
      wire#w1
      Contact( #AVTF_Ent_M1 )
      wire#w2
      I_Contact( #AVTF_Ent_M2 )
      wire#w3
      Contact( #Avance_13 )
      wire#w4
      Contact( #EstadoZona.Marcha_CBx )
      I_Contact( #T1_ET20 )
      I_Contact( #O_Sal_S3 )
      I_Contact( #O_Sal_S4 )
      I_Contact( #O_Vaciar )
      I_Contact( #T1_ET50 )
      I_Contact( #T1_ET61 )
      I_Contact( #T1_ET70 )
      I_Contact( #T1_ET02 )
      S_SR(operand := #T1_ET10, r1 := #T1_ET11)
   END_RUNG
   RUNG wire#w2
      Contact( #AVTF_Ent_M2 )
      Contact( #Ultima_entra_de_E2 )
   END_RUNG wire#w3
   RUNG wire#w1
      I_Contact( #AVTF_Ent_M1 )
      I_Contact( #AVTF_Ent_M2 )
      Contact( #pHsMx )
   END_RUNG wire#w4
   // the same network as SCL:
   IF #T1_ET01 AND NOT #EstadoZona.ParoBlando_CBx AND ((#AVTF_Ent_M1 AND (NOT #AVTF_Ent_M2 OR (#AVTF_Ent_M2 AND #Ultima_entra_de_E2)) AND #Avance_13) OR (NOT #AVTF_Ent_M1 AND NOT #AVTF_Ent_M2 AND #pHsMx)) AND #EstadoZona.Marcha_CBx AND NOT #T1_ET20 AND NOT #O_Sal_S3 AND NOT #O_Sal_S4 AND NOT #O_Vaciar AND NOT #T1_ET50 AND NOT #T1_ET61 AND NOT #T1_ET70 AND NOT #T1_ET02 THEN
       #T1_ET10 := TRUE;   // SR flip-flop
   END_IF;
   IF #T1_ET11 THEN #T1_ET10 := FALSE; END_IF;
END_REGION

REGION Network 19: #T1_ET20. Número de ordenes que se pueden quardar en la Fifo de un scanner.
   RUNG wire#powerrail
      Contact( #T1_ET01 )
      I_Contact( #EstadoZona.ParoBlando_CBx )
      Contact( #AVTF_Ent_M2 )
      wire#w1
      I_Contact( #AVTF_Ent_M1 )
      wire#w2
      Contact( #Avance_24 )
      wire#w3
      Contact( #EstadoZona.Marcha_CBx )
      I_Contact( #T1_ET10 )
      I_Contact( #O_Sal_S3 )
      I_Contact( #O_Sal_S4 )
      I_Contact( #O_Vaciar )
      I_Contact( #T1_ET50 )
      I_Contact( #T1_ET61 )
      I_Contact( #T1_ET70 )
      I_Contact( #T1_ET02 )
      S_SR(operand := #T1_ET20, r1 := #T1_ET21)
   END_RUNG
   RUNG wire#w1
      Contact( #AVTF_Ent_M1 )
      Contact( #Ultima_entra_de_E1 )
   END_RUNG wire#w2
   RUNG wire#w2
      Contact( "ON" )
   END_RUNG wire#w3
   // the same network as SCL:
   IF #T1_ET01 AND NOT #EstadoZona.ParoBlando_CBx AND #AVTF_Ent_M2 AND (NOT #AVTF_Ent_M1 OR (#AVTF_Ent_M1 AND #Ultima_entra_de_E1)) AND (#Avance_24 OR "ON") AND #EstadoZona.Marcha_CBx AND NOT #T1_ET10 AND NOT #O_Sal_S3 AND NOT #O_Sal_S4 AND NOT #O_Vaciar AND NOT #T1_ET50 AND NOT #T1_ET61 AND NOT #T1_ET70 AND NOT #T1_ET02 THEN
       #T1_ET20 := TRUE;   // SR flip-flop
   END_IF;
   IF #T1_ET21 THEN #T1_ET20 := FALSE; END_IF;
END_REGION

REGION Network 20: #CNT_Aus_S4
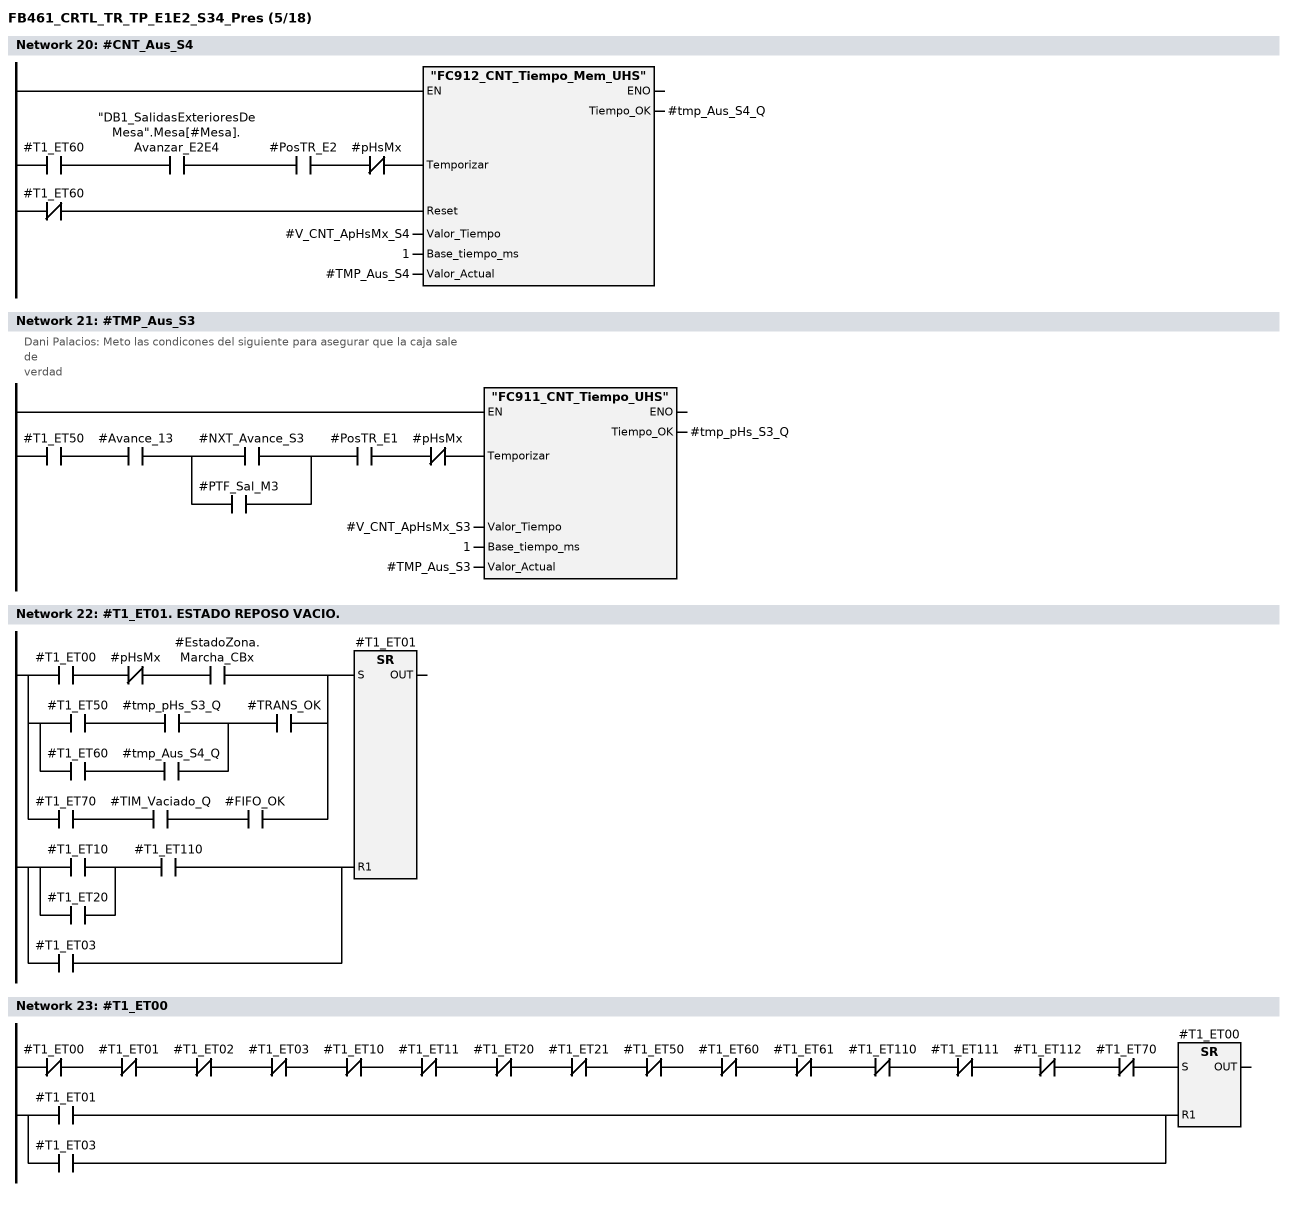
   RUNG wire#powerrail
      "FC912_CNT_Tiempo_Mem_UHS"(Temporizar := wire#w1, Reset := wire#w2, Valor_Tiempo := #V_CNT_ApHsMx_S4, Base_tiempo_ms := 1, Valor_Actual := #TMP_Aus_S4, Tiempo_OK => #tmp_Aus_S4_Q)
   END_RUNG
   RUNG wire#powerrail
      Contact( #T1_ET60 )
      Contact( "DB1_SalidasExterioresDeMesa".Mesa[#Mesa].Avanzar_E2E4 )
      Contact( #PosTR_E2 )
      I_Contact( #pHsMx )
   END_RUNG wire#w1
   RUNG wire#powerrail
      I_Contact( #T1_ET60 )
   END_RUNG wire#w2
   // the same network as SCL:
   "FC912_CNT_Tiempo_Mem_UHS"(Temporizar := #T1_ET60 AND "DB1_SalidasExterioresDeMesa".Mesa[#Mesa].Avanzar_E2E4 AND #PosTR_E2 AND NOT #pHsMx,
                           Reset := NOT #T1_ET60,
                           Valor_Tiempo := #V_CNT_ApHsMx_S4,
                           Base_tiempo_ms := 1,
                           Valor_Actual := #TMP_Aus_S4,
                           Tiempo_OK => #tmp_Aus_S4_Q);
END_REGION

REGION Network 21: #TMP_Aus_S3
   // Dani Palacios: Meto las condicones del siguiente para asegurar que la caja sale 
   // de 
   // verdad
   RUNG wire#powerrail
      "FC911_CNT_Tiempo_UHS"(Temporizar := wire#w3, Valor_Tiempo := #V_CNT_ApHsMx_S3, Base_tiempo_ms := 1, Valor_Actual := #TMP_Aus_S3, Tiempo_OK => #tmp_pHs_S3_Q)
   END_RUNG
   RUNG wire#powerrail
      Contact( #T1_ET50 )
      Contact( #Avance_13 )
      wire#w1
      Contact( #NXT_Avance_S3 )
      wire#w2
      Contact( #PosTR_E1 )
      I_Contact( #pHsMx )
   END_RUNG wire#w3
   RUNG wire#w1
      Contact( #PTF_Sal_M3 )
   END_RUNG wire#w2
   // the same network as SCL:
   "FC911_CNT_Tiempo_UHS"(Temporizar := #T1_ET50 AND #Avance_13 AND (#NXT_Avance_S3 OR #PTF_Sal_M3) AND #PosTR_E1 AND NOT #pHsMx,
                          Valor_Tiempo := #V_CNT_ApHsMx_S3,
                          Base_tiempo_ms := 1,
                          Valor_Actual := #TMP_Aus_S3,
                          Tiempo_OK => #tmp_pHs_S3_Q);
END_REGION

REGION Network 22: #T1_ET01. ESTADO REPOSO VACIO.
   RUNG wire#powerrail
      Contact( #T1_ET00 )
      I_Contact( #pHsMx )
      Contact( #EstadoZona.Marcha_CBx )
      wire#w1
      S_SR(operand := #T1_ET01, r1 := wire#w4)
   END_RUNG
   RUNG wire#powerrail
      Contact( #T1_ET50 )
      Contact( #tmp_pHs_S3_Q )
      wire#w2
      Contact( #TRANS_OK )
   END_RUNG wire#w1
   RUNG wire#powerrail
      Contact( #T1_ET60 )
      Contact( #tmp_Aus_S4_Q )
   END_RUNG wire#w2
   RUNG wire#powerrail
      Contact( #T1_ET70 )
      Contact( #TIM_Vaciado_Q )
      Contact( #FIFO_OK )
   END_RUNG wire#w1
   RUNG wire#powerrail
      Contact( #T1_ET10 )
      wire#w3
      Contact( #T1_ET110 )
   END_RUNG wire#w4
   RUNG wire#powerrail
      Contact( #T1_ET20 )
   END_RUNG wire#w3
   RUNG wire#powerrail
      Contact( #T1_ET03 )
   END_RUNG wire#w4
   // the same network as SCL:
   IF (#T1_ET00 AND NOT #pHsMx AND #EstadoZona.Marcha_CBx) OR (((#T1_ET50 AND #tmp_pHs_S3_Q) OR (#T1_ET60 AND #tmp_Aus_S4_Q)) AND #TRANS_OK) OR (#T1_ET70 AND #TIM_Vaciado_Q AND #FIFO_OK) THEN
       #T1_ET01 := TRUE;   // SR flip-flop
   END_IF;
   IF ((#T1_ET10 OR #T1_ET20) AND #T1_ET110) OR #T1_ET03 THEN #T1_ET01 := FALSE; END_IF;
END_REGION

REGION Network 23: #T1_ET00
   RUNG wire#powerrail
      I_Contact( #T1_ET00 )
      I_Contact( #T1_ET01 )
      I_Contact( #T1_ET02 )
      I_Contact( #T1_ET03 )
      I_Contact( #T1_ET10 )
      I_Contact( #T1_ET11 )
      I_Contact( #T1_ET20 )
      I_Contact( #T1_ET21 )
      I_Contact( #T1_ET50 )
      I_Contact( #T1_ET60 )
      I_Contact( #T1_ET61 )
      I_Contact( #T1_ET110 )
      I_Contact( #T1_ET111 )
      I_Contact( #T1_ET112 )
      I_Contact( #T1_ET70 )
      S_SR(operand := #T1_ET00, r1 := wire#w1)
   END_RUNG
   RUNG wire#powerrail
      Contact( #T1_ET01 )
   END_RUNG wire#w1
   RUNG wire#powerrail
      Contact( #T1_ET03 )
   END_RUNG wire#w1
   // the same network as SCL:
   IF NOT #T1_ET00 AND NOT #T1_ET01 AND NOT #T1_ET02 AND NOT #T1_ET03 AND NOT #T1_ET10 AND NOT #T1_ET11 AND NOT #T1_ET20 AND NOT #T1_ET21 AND NOT #T1_ET50 AND NOT #T1_ET60 AND NOT #T1_ET61 AND NOT #T1_ET110 AND NOT #T1_ET111 AND NOT #T1_ET112 AND NOT #T1_ET70 THEN
       #T1_ET00 := TRUE;   // SR flip-flop
   END_IF;
   IF #T1_ET01 OR #T1_ET03 THEN #T1_ET00 := FALSE; END_IF;
END_REGION

REGION Network 24: timeout tope S3
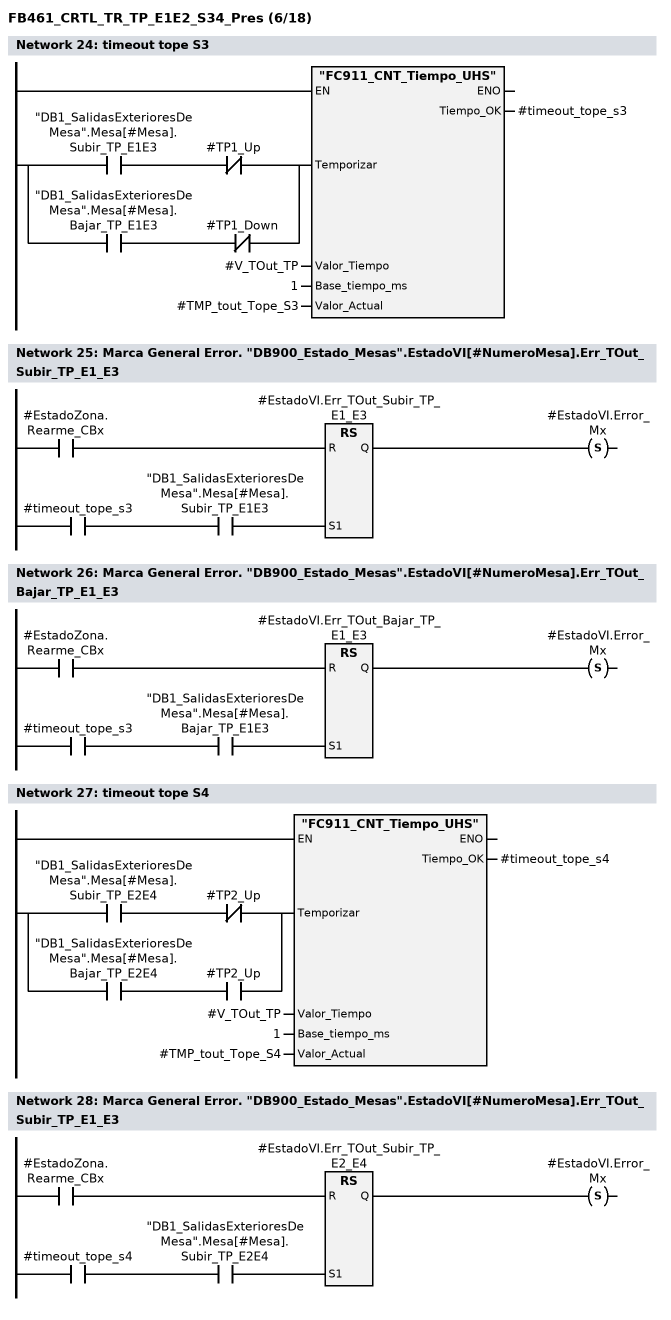
   RUNG wire#powerrail
      "FC911_CNT_Tiempo_UHS"(Temporizar := wire#w1, Valor_Tiempo := #V_TOut_TP, Base_tiempo_ms := 1, Valor_Actual := #TMP_tout_Tope_S3, Tiempo_OK => #timeout_tope_s3)
   END_RUNG
   RUNG wire#powerrail
      Contact( "DB1_SalidasExterioresDeMesa".Mesa[#Mesa].Subir_TP_E1E3 )
      I_Contact( #TP1_Up )
   END_RUNG wire#w1
   RUNG wire#powerrail
      Contact( "DB1_SalidasExterioresDeMesa".Mesa[#Mesa].Bajar_TP_E1E3 )
      I_Contact( #TP1_Down )
   END_RUNG wire#w1
   // the same network as SCL:
   "FC911_CNT_Tiempo_UHS"(Temporizar := ("DB1_SalidasExterioresDeMesa".Mesa[#Mesa].Subir_TP_E1E3 AND NOT #TP1_Up) OR ("DB1_SalidasExterioresDeMesa".Mesa[#Mesa].Bajar_TP_E1E3 AND NOT #TP1_Down),
                          Valor_Tiempo := #V_TOut_TP,
                          Base_tiempo_ms := 1,
                          Valor_Actual := #TMP_tout_Tope_S3,
                          Tiempo_OK => #timeout_tope_s3);
END_REGION

REGION Network 25: Marca General Error. "DB900_Estado_Mesas".EstadoVI[#NumeroMesa].Err_TOut_Subir_TP_E1_E3
   RUNG wire#powerrail
      Contact( #EstadoZona.Rearme_CBx )
      S_RS(operand := #EstadoVI.Err_TOut_Subir_TP_E1_E3, s1 := wire#w1)
      S_Coil( #EstadoVI.Error_Mx )
   END_RUNG
   RUNG wire#powerrail
      Contact( #timeout_tope_s3 )
      Contact( "DB1_SalidasExterioresDeMesa".Mesa[#Mesa].Subir_TP_E1E3 )
   END_RUNG wire#w1
   // the same network as SCL:
   IF #EstadoZona.Rearme_CBx THEN
       #EstadoVI.Err_TOut_Subir_TP_E1_E3 := FALSE;   // RS flip-flop
   END_IF;
   IF #timeout_tope_s3 AND "DB1_SalidasExterioresDeMesa".Mesa[#Mesa].Subir_TP_E1E3 THEN
       #EstadoVI.Err_TOut_Subir_TP_E1_E3 := TRUE;
   END_IF;
   IF #EstadoVI.Err_TOut_Subir_TP_E1_E3 THEN #EstadoVI.Error_Mx := TRUE; END_IF;
END_REGION

REGION Network 26: Marca General Error. "DB900_Estado_Mesas".EstadoVI[#NumeroMesa].Err_TOut_Bajar_TP_E1_E3
   RUNG wire#powerrail
      Contact( #EstadoZona.Rearme_CBx )
      S_RS(operand := #EstadoVI.Err_TOut_Bajar_TP_E1_E3, s1 := wire#w1)
      S_Coil( #EstadoVI.Error_Mx )
   END_RUNG
   RUNG wire#powerrail
      Contact( #timeout_tope_s3 )
      Contact( "DB1_SalidasExterioresDeMesa".Mesa[#Mesa].Bajar_TP_E1E3 )
   END_RUNG wire#w1
   // the same network as SCL:
   IF #EstadoZona.Rearme_CBx THEN
       #EstadoVI.Err_TOut_Bajar_TP_E1_E3 := FALSE;   // RS flip-flop
   END_IF;
   IF #timeout_tope_s3 AND "DB1_SalidasExterioresDeMesa".Mesa[#Mesa].Bajar_TP_E1E3 THEN
       #EstadoVI.Err_TOut_Bajar_TP_E1_E3 := TRUE;
   END_IF;
   IF #EstadoVI.Err_TOut_Bajar_TP_E1_E3 THEN #EstadoVI.Error_Mx := TRUE; END_IF;
END_REGION

REGION Network 27: timeout tope S4
   RUNG wire#powerrail
      "FC911_CNT_Tiempo_UHS"(Temporizar := wire#w1, Valor_Tiempo := #V_TOut_TP, Base_tiempo_ms := 1, Valor_Actual := #TMP_tout_Tope_S4, Tiempo_OK => #timeout_tope_s4)
   END_RUNG
   RUNG wire#powerrail
      Contact( "DB1_SalidasExterioresDeMesa".Mesa[#Mesa].Subir_TP_E2E4 )
      I_Contact( #TP2_Up )
   END_RUNG wire#w1
   RUNG wire#powerrail
      Contact( "DB1_SalidasExterioresDeMesa".Mesa[#Mesa].Bajar_TP_E2E4 )
      Contact( #TP2_Up )
   END_RUNG wire#w1
   // the same network as SCL:
   "FC911_CNT_Tiempo_UHS"(Temporizar := ("DB1_SalidasExterioresDeMesa".Mesa[#Mesa].Subir_TP_E2E4 AND NOT #TP2_Up) OR ("DB1_SalidasExterioresDeMesa".Mesa[#Mesa].Bajar_TP_E2E4 AND #TP2_Up),
                          Valor_Tiempo := #V_TOut_TP,
                          Base_tiempo_ms := 1,
                          Valor_Actual := #TMP_tout_Tope_S4,
                          Tiempo_OK => #timeout_tope_s4);
END_REGION

REGION Network 28: Marca General Error. "DB900_Estado_Mesas".EstadoVI[#NumeroMesa].Err_TOut_Subir_TP_E1_E3
   RUNG wire#powerrail
      Contact( #EstadoZona.Rearme_CBx )
      S_RS(operand := #EstadoVI.Err_TOut_Subir_TP_E2_E4, s1 := wire#w1)
      S_Coil( #EstadoVI.Error_Mx )
   END_RUNG
   RUNG wire#powerrail
      Contact( #timeout_tope_s4 )
      Contact( "DB1_SalidasExterioresDeMesa".Mesa[#Mesa].Subir_TP_E2E4 )
   END_RUNG wire#w1
   // the same network as SCL:
   IF #EstadoZona.Rearme_CBx THEN
       #EstadoVI.Err_TOut_Subir_TP_E2_E4 := FALSE;   // RS flip-flop
   END_IF;
   IF #timeout_tope_s4 AND "DB1_SalidasExterioresDeMesa".Mesa[#Mesa].Subir_TP_E2E4 THEN
       #EstadoVI.Err_TOut_Subir_TP_E2_E4 := TRUE;
   END_IF;
   IF #EstadoVI.Err_TOut_Subir_TP_E2_E4 THEN #EstadoVI.Error_Mx := TRUE; END_IF;
END_REGION

REGION Network 29: Marca General Error. "DB900_Estado_Mesas".EstadoVI[#NumeroMesa].Err_TOut_Bajar_TP_E1_E3
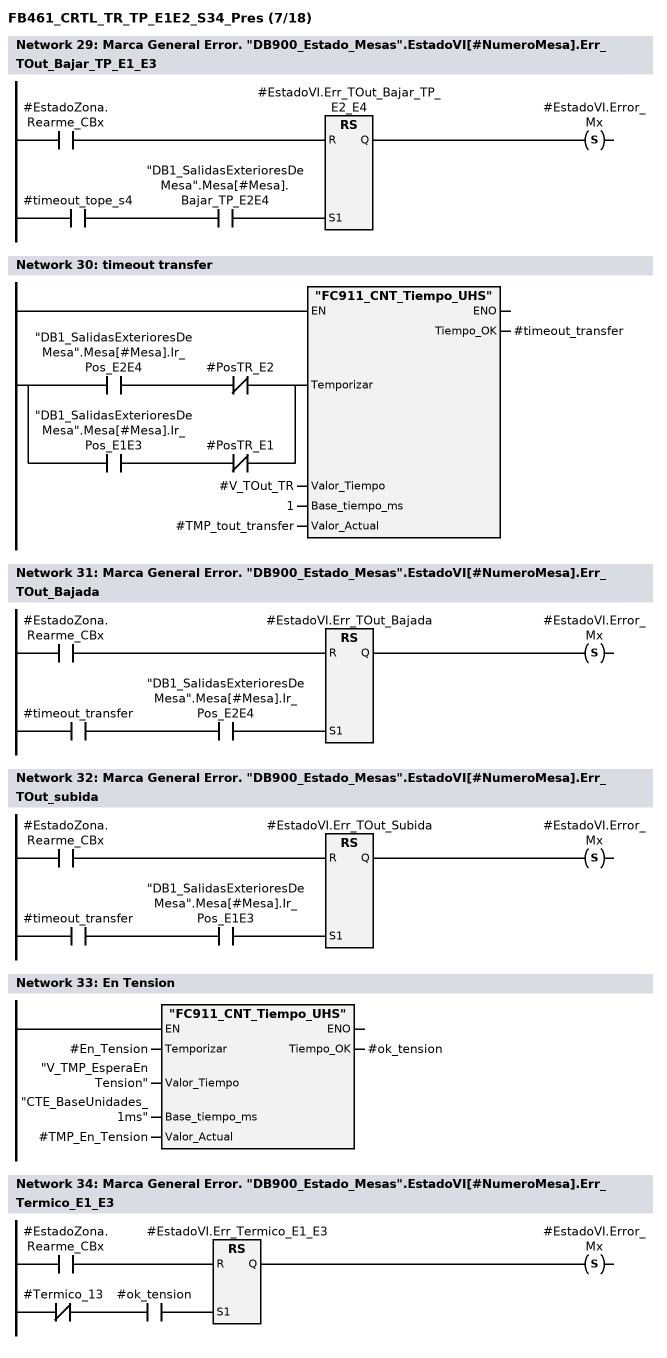
   RUNG wire#powerrail
      Contact( #EstadoZona.Rearme_CBx )
      S_RS(operand := #EstadoVI.Err_TOut_Bajar_TP_E2_E4, s1 := wire#w1)
      S_Coil( #EstadoVI.Error_Mx )
   END_RUNG
   RUNG wire#powerrail
      Contact( #timeout_tope_s4 )
      Contact( "DB1_SalidasExterioresDeMesa".Mesa[#Mesa].Bajar_TP_E2E4 )
   END_RUNG wire#w1
   // the same network as SCL:
   IF #EstadoZona.Rearme_CBx THEN
       #EstadoVI.Err_TOut_Bajar_TP_E2_E4 := FALSE;   // RS flip-flop
   END_IF;
   IF #timeout_tope_s4 AND "DB1_SalidasExterioresDeMesa".Mesa[#Mesa].Bajar_TP_E2E4 THEN
       #EstadoVI.Err_TOut_Bajar_TP_E2_E4 := TRUE;
   END_IF;
   IF #EstadoVI.Err_TOut_Bajar_TP_E2_E4 THEN #EstadoVI.Error_Mx := TRUE; END_IF;
END_REGION

REGION Network 30: timeout transfer
   RUNG wire#powerrail
      "FC911_CNT_Tiempo_UHS"(Temporizar := wire#w1, Valor_Tiempo := #V_TOut_TR, Base_tiempo_ms := 1, Valor_Actual := #TMP_tout_transfer, Tiempo_OK => #timeout_transfer)
   END_RUNG
   RUNG wire#powerrail
      Contact( "DB1_SalidasExterioresDeMesa".Mesa[#Mesa].Ir_Pos_E2E4 )
      I_Contact( #PosTR_E2 )
   END_RUNG wire#w1
   RUNG wire#powerrail
      Contact( "DB1_SalidasExterioresDeMesa".Mesa[#Mesa].Ir_Pos_E1E3 )
      I_Contact( #PosTR_E1 )
   END_RUNG wire#w1
   // the same network as SCL:
   "FC911_CNT_Tiempo_UHS"(Temporizar := ("DB1_SalidasExterioresDeMesa".Mesa[#Mesa].Ir_Pos_E2E4 AND NOT #PosTR_E2) OR ("DB1_SalidasExterioresDeMesa".Mesa[#Mesa].Ir_Pos_E1E3 AND NOT #PosTR_E1),
                          Valor_Tiempo := #V_TOut_TR,
                          Base_tiempo_ms := 1,
                          Valor_Actual := #TMP_tout_transfer,
                          Tiempo_OK => #timeout_transfer);
END_REGION

REGION Network 31: Marca General Error. "DB900_Estado_Mesas".EstadoVI[#NumeroMesa].Err_TOut_Bajada
   RUNG wire#powerrail
      Contact( #EstadoZona.Rearme_CBx )
      S_RS(operand := #EstadoVI.Err_TOut_Bajada, s1 := wire#w1)
      S_Coil( #EstadoVI.Error_Mx )
   END_RUNG
   RUNG wire#powerrail
      Contact( #timeout_transfer )
      Contact( "DB1_SalidasExterioresDeMesa".Mesa[#Mesa].Ir_Pos_E2E4 )
   END_RUNG wire#w1
   // the same network as SCL:
   IF #EstadoZona.Rearme_CBx THEN
       #EstadoVI.Err_TOut_Bajada := FALSE;   // RS flip-flop
   END_IF;
   IF #timeout_transfer AND "DB1_SalidasExterioresDeMesa".Mesa[#Mesa].Ir_Pos_E2E4 THEN
       #EstadoVI.Err_TOut_Bajada := TRUE;
   END_IF;
   IF #EstadoVI.Err_TOut_Bajada THEN #EstadoVI.Error_Mx := TRUE; END_IF;
END_REGION

REGION Network 32: Marca General Error. "DB900_Estado_Mesas".EstadoVI[#NumeroMesa].Err_TOut_subida
   RUNG wire#powerrail
      Contact( #EstadoZona.Rearme_CBx )
      S_RS(operand := #EstadoVI.Err_TOut_Subida, s1 := wire#w1)
      S_Coil( #EstadoVI.Error_Mx )
   END_RUNG
   RUNG wire#powerrail
      Contact( #timeout_transfer )
      Contact( "DB1_SalidasExterioresDeMesa".Mesa[#Mesa].Ir_Pos_E1E3 )
   END_RUNG wire#w1
   // the same network as SCL:
   IF #EstadoZona.Rearme_CBx THEN
       #EstadoVI.Err_TOut_Subida := FALSE;   // RS flip-flop
   END_IF;
   IF #timeout_transfer AND "DB1_SalidasExterioresDeMesa".Mesa[#Mesa].Ir_Pos_E1E3 THEN
       #EstadoVI.Err_TOut_Subida := TRUE;
   END_IF;
   IF #EstadoVI.Err_TOut_Subida THEN #EstadoVI.Error_Mx := TRUE; END_IF;
END_REGION

REGION Network 33: En Tension
   RUNG wire#powerrail
      "FC911_CNT_Tiempo_UHS"(Temporizar := #En_Tension, Valor_Tiempo := "V_TMP_EsperaEnTension", Base_tiempo_ms := "CTE_BaseUnidades_1ms", Valor_Actual := #TMP_En_Tension, Tiempo_OK => #ok_tension)
   END_RUNG
   // the same network as SCL:
   "FC911_CNT_Tiempo_UHS"(Temporizar := #En_Tension,
                          Valor_Tiempo := "V_TMP_EsperaEnTension",
                          Base_tiempo_ms := "CTE_BaseUnidades_1ms",
                          Valor_Actual := #TMP_En_Tension,
                          Tiempo_OK => #ok_tension);
END_REGION

REGION Network 34: Marca General Error. "DB900_Estado_Mesas".EstadoVI[#NumeroMesa].Err_Termico_E1_E3
   RUNG wire#powerrail
      Contact( #EstadoZona.Rearme_CBx )
      S_RS(operand := #EstadoVI.Err_Termico_E1_E3, s1 := wire#w1)
      S_Coil( #EstadoVI.Error_Mx )
   END_RUNG
   RUNG wire#powerrail
      I_Contact( #Termico_13 )
      Contact( #ok_tension )
   END_RUNG wire#w1
   // the same network as SCL:
   IF #EstadoZona.Rearme_CBx THEN
       #EstadoVI.Err_Termico_E1_E3 := FALSE;   // RS flip-flop
   END_IF;
   IF NOT #Termico_13 AND #ok_tension THEN #EstadoVI.Err_Termico_E1_E3 := TRUE; END_IF;
   IF #EstadoVI.Err_Termico_E1_E3 THEN #EstadoVI.Error_Mx := TRUE; END_IF;
END_REGION

REGION Network 35: Marca General Error. "DB900_Estado_Mesas".EstadoVI[#NumeroMesa].Err_Termico_E2_E4
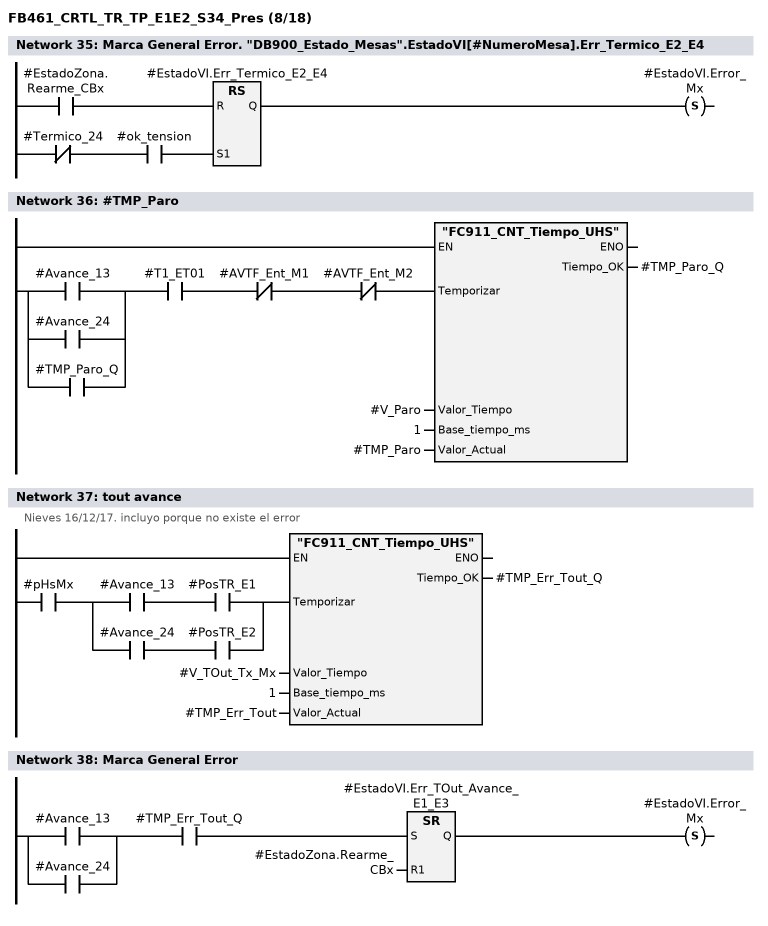
   RUNG wire#powerrail
      Contact( #EstadoZona.Rearme_CBx )
      S_RS(operand := #EstadoVI.Err_Termico_E2_E4, s1 := wire#w1)
      S_Coil( #EstadoVI.Error_Mx )
   END_RUNG
   RUNG wire#powerrail
      I_Contact( #Termico_24 )
      Contact( #ok_tension )
   END_RUNG wire#w1
   // the same network as SCL:
   IF #EstadoZona.Rearme_CBx THEN
       #EstadoVI.Err_Termico_E2_E4 := FALSE;   // RS flip-flop
   END_IF;
   IF NOT #Termico_24 AND #ok_tension THEN #EstadoVI.Err_Termico_E2_E4 := TRUE; END_IF;
   IF #EstadoVI.Err_Termico_E2_E4 THEN #EstadoVI.Error_Mx := TRUE; END_IF;
END_REGION

REGION Network 36: #TMP_Paro
   RUNG wire#powerrail
      "FC911_CNT_Tiempo_UHS"(Temporizar := wire#w2, Valor_Tiempo := #V_Paro, Base_tiempo_ms := 1, Valor_Actual := #TMP_Paro, Tiempo_OK => #TMP_Paro_Q)
   END_RUNG
   RUNG wire#powerrail
      Contact( #Avance_13 )
      wire#w1
      Contact( #T1_ET01 )
      I_Contact( #AVTF_Ent_M1 )
      I_Contact( #AVTF_Ent_M2 )
   END_RUNG wire#w2
   RUNG wire#powerrail
      Contact( #Avance_24 )
   END_RUNG wire#w1
   RUNG wire#powerrail
      Contact( #TMP_Paro_Q )
   END_RUNG wire#w1
   // the same network as SCL:
   "FC911_CNT_Tiempo_UHS"(Temporizar := (#Avance_13 OR #Avance_24 OR #TMP_Paro_Q) AND #T1_ET01 AND NOT #AVTF_Ent_M1 AND NOT #AVTF_Ent_M2,
                          Valor_Tiempo := #V_Paro,
                          Base_tiempo_ms := 1,
                          Valor_Actual := #TMP_Paro,
                          Tiempo_OK => #TMP_Paro_Q);
END_REGION

REGION Network 37: tout avance
   // Nieves 16/12/17. incluyo porque no existe el error
   RUNG wire#powerrail
      "FC911_CNT_Tiempo_UHS"(Temporizar := wire#w2, Valor_Tiempo := #V_TOut_Tx_Mx, Base_tiempo_ms := 1, Valor_Actual := #TMP_Err_Tout, Tiempo_OK => #TMP_Err_Tout_Q)
   END_RUNG
   RUNG wire#powerrail
      Contact( #pHsMx )
      wire#w1
      Contact( #Avance_13 )
      Contact( #PosTR_E1 )
   END_RUNG wire#w2
   RUNG wire#w1
      Contact( #Avance_24 )
      Contact( #PosTR_E2 )
   END_RUNG wire#w2
   // the same network as SCL:
   "FC911_CNT_Tiempo_UHS"(Temporizar := #pHsMx AND ((#Avance_13 AND #PosTR_E1) OR (#Avance_24 AND #PosTR_E2)),
                          Valor_Tiempo := #V_TOut_Tx_Mx,
                          Base_tiempo_ms := 1,
                          Valor_Actual := #TMP_Err_Tout,
                          Tiempo_OK => #TMP_Err_Tout_Q);
END_REGION

REGION Network 38: Marca General Error
   RUNG wire#powerrail
      Contact( #Avance_13 )
      wire#w1
      Contact( #TMP_Err_Tout_Q )
      S_SR(operand := #EstadoVI.Err_TOut_Avance_E1_E3, r1 := #EstadoZona.Rearme_CBx)
      S_Coil( #EstadoVI.Error_Mx )
   END_RUNG
   RUNG wire#powerrail
      Contact( #Avance_24 )
   END_RUNG wire#w1
   // the same network as SCL:
   IF (#Avance_13 OR #Avance_24) AND #TMP_Err_Tout_Q THEN
       #EstadoVI.Err_TOut_Avance_E1_E3 := TRUE;   // SR flip-flop
   END_IF;
   IF #EstadoZona.Rearme_CBx THEN #EstadoVI.Err_TOut_Avance_E1_E3 := FALSE; END_IF;
   IF #EstadoVI.Err_TOut_Avance_E1_E3 THEN #EstadoVI.Error_Mx := TRUE; END_IF;
END_REGION

REGION Network 39: #TIM_Vacido
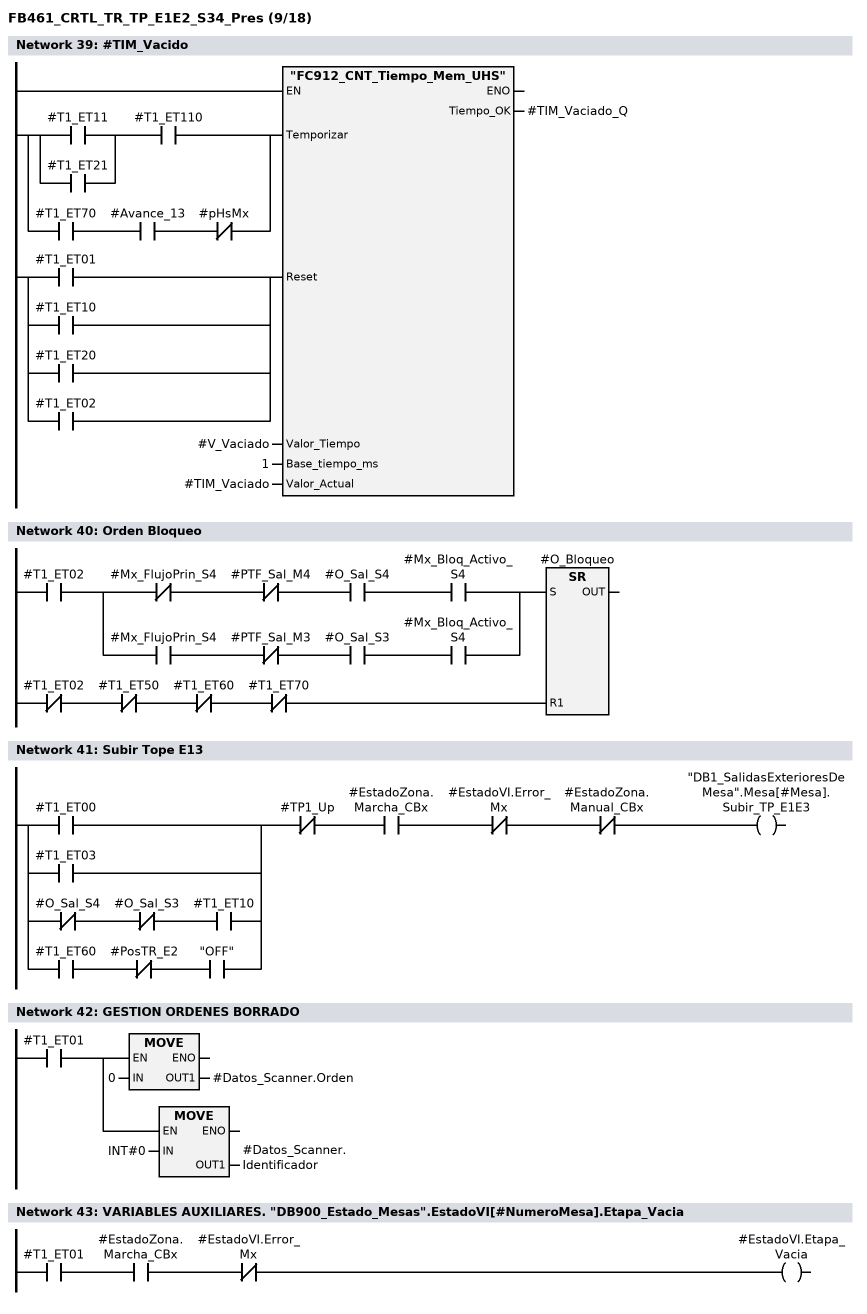
   RUNG wire#powerrail
      "FC912_CNT_Tiempo_Mem_UHS"(Temporizar := wire#w2, Reset := wire#w3, Valor_Tiempo := #V_Vaciado, Base_tiempo_ms := 1, Valor_Actual := #TIM_Vaciado, Tiempo_OK => #TIM_Vaciado_Q)
   END_RUNG
   RUNG wire#powerrail
      Contact( #T1_ET11 )
      wire#w1
      Contact( #T1_ET110 )
   END_RUNG wire#w2
   RUNG wire#powerrail
      Contact( #T1_ET21 )
   END_RUNG wire#w1
   RUNG wire#powerrail
      Contact( #T1_ET70 )
      Contact( #Avance_13 )
      I_Contact( #pHsMx )
   END_RUNG wire#w2
   RUNG wire#powerrail
      Contact( #T1_ET01 )
   END_RUNG wire#w3
   RUNG wire#powerrail
      Contact( #T1_ET10 )
   END_RUNG wire#w3
   RUNG wire#powerrail
      Contact( #T1_ET20 )
   END_RUNG wire#w3
   RUNG wire#powerrail
      Contact( #T1_ET02 )
   END_RUNG wire#w3
   // the same network as SCL:
   "FC912_CNT_Tiempo_Mem_UHS"(Temporizar := ((#T1_ET11 OR #T1_ET21) AND #T1_ET110) OR (#T1_ET70 AND #Avance_13 AND NOT #pHsMx),
                           Reset := #T1_ET01 OR #T1_ET10 OR #T1_ET20 OR #T1_ET02,
                           Valor_Tiempo := #V_Vaciado,
                           Base_tiempo_ms := 1,
                           Valor_Actual := #TIM_Vaciado,
                           Tiempo_OK => #TIM_Vaciado_Q);
END_REGION

REGION Network 40: Orden Bloqueo
   RUNG wire#powerrail
      Contact( #T1_ET02 )
      wire#w1
      I_Contact( #Mx_FlujoPrin_S4 )
      I_Contact( #PTF_Sal_M4 )
      Contact( #O_Sal_S4 )
      Contact( #Mx_Bloq_Activo_S4 )
      wire#w2
      S_SR(operand := #O_Bloqueo, r1 := wire#w3)
   END_RUNG
   RUNG wire#w1
      Contact( #Mx_FlujoPrin_S4 )
      I_Contact( #PTF_Sal_M3 )
      Contact( #O_Sal_S3 )
      Contact( #Mx_Bloq_Activo_S4 )
   END_RUNG wire#w2
   RUNG wire#powerrail
      I_Contact( #T1_ET02 )
      I_Contact( #T1_ET50 )
      I_Contact( #T1_ET60 )
      I_Contact( #T1_ET70 )
   END_RUNG wire#w3
   // the same network as SCL:
   IF #T1_ET02 AND ((NOT #Mx_FlujoPrin_S4 AND NOT #PTF_Sal_M4 AND #O_Sal_S4 AND #Mx_Bloq_Activo_S4) OR (#Mx_FlujoPrin_S4 AND NOT #PTF_Sal_M3 AND #O_Sal_S3 AND #Mx_Bloq_Activo_S4)) THEN
       #O_Bloqueo := TRUE;   // SR flip-flop
   END_IF;
   IF NOT #T1_ET02 AND NOT #T1_ET50 AND NOT #T1_ET60 AND NOT #T1_ET70 THEN #O_Bloqueo := FALSE; END_IF;
END_REGION

REGION Network 41: Subir Tope E13
   RUNG wire#powerrail
      Contact( #T1_ET00 )
      wire#w1
      I_Contact( #TP1_Up )
      Contact( #EstadoZona.Marcha_CBx )
      I_Contact( #EstadoVI.Error_Mx )
      I_Contact( #EstadoZona.Manual_CBx )
      Coil( "DB1_SalidasExterioresDeMesa".Mesa[#Mesa].Subir_TP_E1E3 )
   END_RUNG
   RUNG wire#powerrail
      Contact( #T1_ET03 )
   END_RUNG wire#w1
   RUNG wire#powerrail
      I_Contact( #O_Sal_S4 )
      I_Contact( #O_Sal_S3 )
      Contact( #T1_ET10 )
   END_RUNG wire#w1
   RUNG wire#powerrail
      Contact( #T1_ET60 )
      I_Contact( #PosTR_E2 )
      Contact( "OFF" )
   END_RUNG wire#w1
   // the same network as SCL:
   "DB1_SalidasExterioresDeMesa".Mesa[#Mesa].Subir_TP_E1E3 := (#T1_ET00 OR #T1_ET03 OR (NOT #O_Sal_S4 AND NOT #O_Sal_S3 AND #T1_ET10) OR (#T1_ET60 AND NOT #PosTR_E2 AND "OFF")) AND NOT #TP1_Up AND #EstadoZona.Marcha_CBx AND NOT #EstadoVI.Error_Mx AND NOT #EstadoZona.Manual_CBx;
END_REGION

REGION Network 42: GESTION ORDENES BORRADO
   RUNG wire#powerrail
      Contact( #T1_ET01 )
      wire#w1
      { S7_GenerateENO := "TRUE" } Move(in := 0, out1 => #Datos_Scanner.Orden)
   END_RUNG
   RUNG wire#w1
      { S7_GenerateENO := "TRUE" } Move(in := INT#0, out1 => #Datos_Scanner.Identificador)
   END_RUNG
   // the same network as SCL:
   IF #T1_ET01 THEN
       #Datos_Scanner.Orden := 0;
       #Datos_Scanner.Identificador := INT#0;
   END_IF;
END_REGION

REGION Network 43: VARIABLES AUXILIARES. "DB900_Estado_Mesas".EstadoVI[#NumeroMesa].Etapa_Vacia
   RUNG wire#powerrail
      Contact( #T1_ET01 )
      Contact( #EstadoZona.Marcha_CBx )
      I_Contact( #EstadoVI.Error_Mx )
      Coil( #EstadoVI.Etapa_Vacia )
   END_RUNG
   // the same network as SCL:
   #EstadoVI.Etapa_Vacia := #T1_ET01 AND #EstadoZona.Marcha_CBx AND NOT #EstadoVI.Error_Mx;
END_REGION

REGION Network 44: VARIABLES AUXILIARES. "DB900_Estado_Mesas".EstadoVI[#NumeroMesa].Etapas_Carga_E1
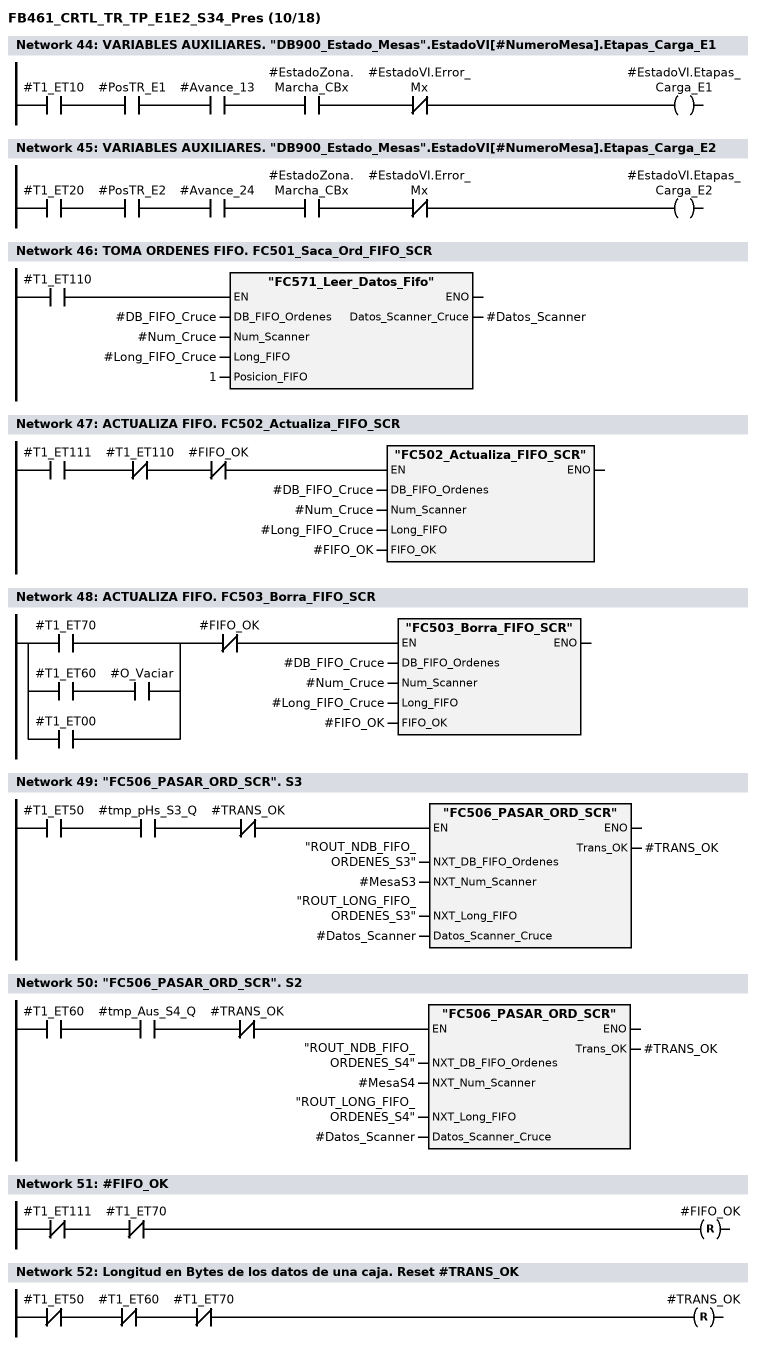
   RUNG wire#powerrail
      Contact( #T1_ET10 )
      Contact( #PosTR_E1 )
      Contact( #Avance_13 )
      Contact( #EstadoZona.Marcha_CBx )
      I_Contact( #EstadoVI.Error_Mx )
      Coil( #EstadoVI.Etapas_Carga_E1 )
   END_RUNG
   // the same network as SCL:
   #EstadoVI.Etapas_Carga_E1 := #T1_ET10 AND #PosTR_E1 AND #Avance_13 AND #EstadoZona.Marcha_CBx AND NOT #EstadoVI.Error_Mx;
END_REGION

REGION Network 45: VARIABLES AUXILIARES. "DB900_Estado_Mesas".EstadoVI[#NumeroMesa].Etapas_Carga_E2
   RUNG wire#powerrail
      Contact( #T1_ET20 )
      Contact( #PosTR_E2 )
      Contact( #Avance_24 )
      Contact( #EstadoZona.Marcha_CBx )
      I_Contact( #EstadoVI.Error_Mx )
      Coil( #EstadoVI.Etapas_Carga_E2 )
   END_RUNG
   // the same network as SCL:
   #EstadoVI.Etapas_Carga_E2 := #T1_ET20 AND #PosTR_E2 AND #Avance_24 AND #EstadoZona.Marcha_CBx AND NOT #EstadoVI.Error_Mx;
END_REGION

REGION Network 46: TOMA ORDENES FIFO. FC501_Saca_Ord_FIFO_SCR
   RUNG wire#powerrail
      Contact( #T1_ET110 )
      "FC571_Leer_Datos_Fifo"(DB_FIFO_Ordenes := #DB_FIFO_Cruce, Num_Scanner := #Num_Cruce, Long_FIFO := #Long_FIFO_Cruce, Posicion_FIFO := 1, Datos_Scanner_Cruce => #Datos_Scanner)
   END_RUNG
   // the same network as SCL:
   IF #T1_ET110 THEN
       "FC571_Leer_Datos_Fifo"(DB_FIFO_Ordenes := #DB_FIFO_Cruce,
                               Num_Scanner := #Num_Cruce,
                               Long_FIFO := #Long_FIFO_Cruce,
                               Posicion_FIFO := 1,
                               Datos_Scanner_Cruce => #Datos_Scanner);
   END_IF;
END_REGION

REGION Network 47: ACTUALIZA FIFO. FC502_Actualiza_FIFO_SCR
   RUNG wire#powerrail
      Contact( #T1_ET111 )
      I_Contact( #T1_ET110 )
      I_Contact( #FIFO_OK )
      "FC502_Actualiza_FIFO_SCR"(DB_FIFO_Ordenes := #DB_FIFO_Cruce, Num_Scanner := #Num_Cruce, Long_FIFO := #Long_FIFO_Cruce, FIFO_OK := #FIFO_OK)
   END_RUNG
   // the same network as SCL:
   IF #T1_ET111 AND NOT #T1_ET110 AND NOT #FIFO_OK THEN
       "FC502_Actualiza_FIFO_SCR"(DB_FIFO_Ordenes := #DB_FIFO_Cruce,
                               Num_Scanner := #Num_Cruce,
                               Long_FIFO := #Long_FIFO_Cruce,
                               FIFO_OK := #FIFO_OK);
   END_IF;
END_REGION

REGION Network 48: ACTUALIZA FIFO. FC503_Borra_FIFO_SCR
   RUNG wire#powerrail
      Contact( #T1_ET70 )
      wire#w1
      I_Contact( #FIFO_OK )
      "FC503_Borra_FIFO_SCR"(DB_FIFO_Ordenes := #DB_FIFO_Cruce, Num_Scanner := #Num_Cruce, Long_FIFO := #Long_FIFO_Cruce, FIFO_OK := #FIFO_OK)
   END_RUNG
   RUNG wire#powerrail
      Contact( #T1_ET60 )
      Contact( #O_Vaciar )
   END_RUNG wire#w1
   RUNG wire#powerrail
      Contact( #T1_ET00 )
   END_RUNG wire#w1
   // the same network as SCL:
   IF (#T1_ET70 OR (#T1_ET60 AND #O_Vaciar) OR #T1_ET00) AND NOT #FIFO_OK THEN
       "FC503_Borra_FIFO_SCR"(DB_FIFO_Ordenes := #DB_FIFO_Cruce,
                              Num_Scanner := #Num_Cruce,
                              Long_FIFO := #Long_FIFO_Cruce,
                              FIFO_OK := #FIFO_OK);
   END_IF;
END_REGION

REGION Network 49: "FC506_PASAR_ORD_SCR". S3
   RUNG wire#powerrail
      Contact( #T1_ET50 )
      Contact( #tmp_pHs_S3_Q )
      I_Contact( #TRANS_OK )
      "FC506_PASAR_ORD_SCR"(NXT_DB_FIFO_Ordenes := "ROUT_NDB_FIFO_ORDENES_S3", NXT_Num_Scanner := #MesaS3, NXT_Long_FIFO := "ROUT_LONG_FIFO_ORDENES_S3", Datos_Scanner_Cruce := #Datos_Scanner, Trans_OK => #TRANS_OK)
   END_RUNG
   // the same network as SCL:
   IF #T1_ET50 AND #tmp_pHs_S3_Q AND NOT #TRANS_OK THEN
       "FC506_PASAR_ORD_SCR"(NXT_DB_FIFO_Ordenes := "ROUT_NDB_FIFO_ORDENES_S3",
                             NXT_Num_Scanner := #MesaS3,
                             NXT_Long_FIFO := "ROUT_LONG_FIFO_ORDENES_S3",
                             Datos_Scanner_Cruce := #Datos_Scanner,
                             Trans_OK => #TRANS_OK);
   END_IF;
END_REGION

REGION Network 50: "FC506_PASAR_ORD_SCR". S2
   RUNG wire#powerrail
      Contact( #T1_ET60 )
      Contact( #tmp_Aus_S4_Q )
      I_Contact( #TRANS_OK )
      "FC506_PASAR_ORD_SCR"(NXT_DB_FIFO_Ordenes := "ROUT_NDB_FIFO_ORDENES_S4", NXT_Num_Scanner := #MesaS4, NXT_Long_FIFO := "ROUT_LONG_FIFO_ORDENES_S4", Datos_Scanner_Cruce := #Datos_Scanner, Trans_OK => #TRANS_OK)
   END_RUNG
   // the same network as SCL:
   IF #T1_ET60 AND #tmp_Aus_S4_Q AND NOT #TRANS_OK THEN
       "FC506_PASAR_ORD_SCR"(NXT_DB_FIFO_Ordenes := "ROUT_NDB_FIFO_ORDENES_S4",
                             NXT_Num_Scanner := #MesaS4,
                             NXT_Long_FIFO := "ROUT_LONG_FIFO_ORDENES_S4",
                             Datos_Scanner_Cruce := #Datos_Scanner,
                             Trans_OK => #TRANS_OK);
   END_IF;
END_REGION

REGION Network 51: #FIFO_OK
   RUNG wire#powerrail
      I_Contact( #T1_ET111 )
      I_Contact( #T1_ET70 )
      R_Coil( #FIFO_OK )
   END_RUNG
   // the same network as SCL:
   IF NOT #T1_ET111 AND NOT #T1_ET70 THEN #FIFO_OK := FALSE; END_IF;
END_REGION

REGION Network 52: Longitud en Bytes de los datos de una caja. Reset #TRANS_OK
   RUNG wire#powerrail
      I_Contact( #T1_ET50 )
      I_Contact( #T1_ET60 )
      I_Contact( #T1_ET70 )
      R_Coil( #TRANS_OK )
   END_RUNG
   // the same network as SCL:
   IF NOT #T1_ET50 AND NOT #T1_ET60 AND NOT #T1_ET70 THEN #TRANS_OK := FALSE; END_IF;
END_REGION

REGION Network 53: #PRV_CARGA_OK_E1
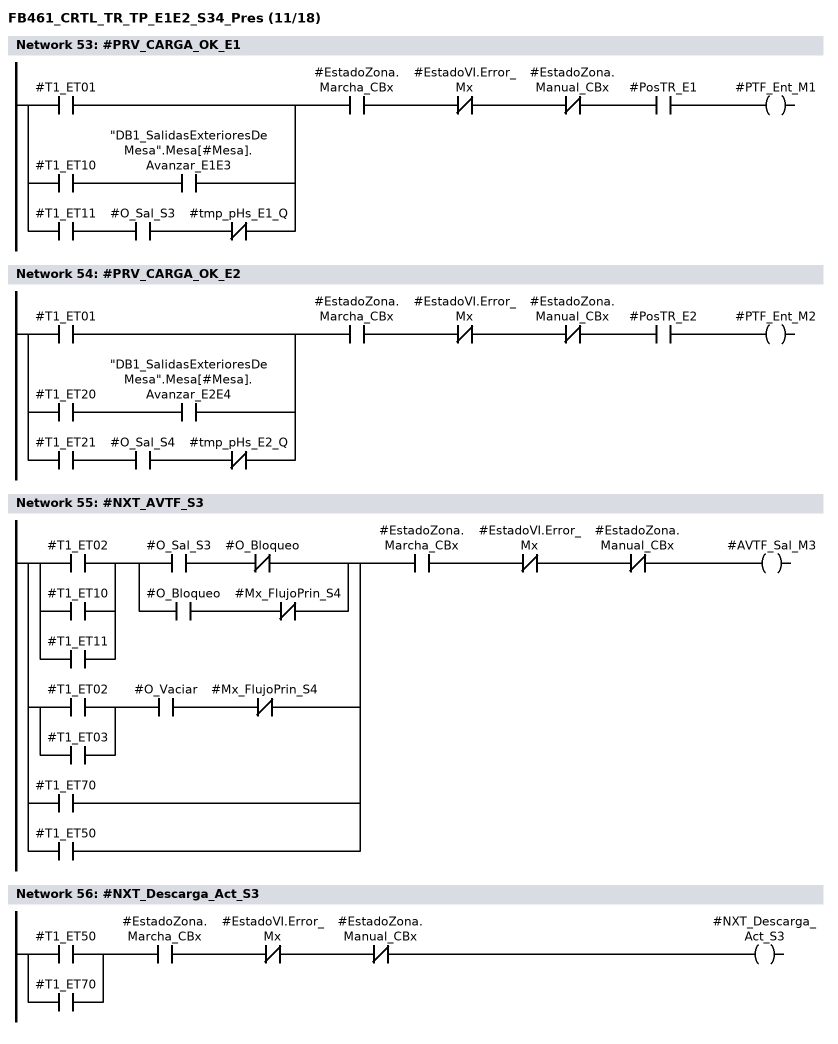
   RUNG wire#powerrail
      Contact( #T1_ET01 )
      wire#w1
      Contact( #EstadoZona.Marcha_CBx )
      I_Contact( #EstadoVI.Error_Mx )
      I_Contact( #EstadoZona.Manual_CBx )
      Contact( #PosTR_E1 )
      Coil( #PTF_Ent_M1 )
   END_RUNG
   RUNG wire#powerrail
      Contact( #T1_ET10 )
      Contact( "DB1_SalidasExterioresDeMesa".Mesa[#Mesa].Avanzar_E1E3 )
   END_RUNG wire#w1
   RUNG wire#powerrail
      Contact( #T1_ET11 )
      Contact( #O_Sal_S3 )
      I_Contact( #tmp_pHs_E1_Q )
   END_RUNG wire#w1
   // the same network as SCL:
   #PTF_Ent_M1 := (#T1_ET01 OR (#T1_ET10 AND "DB1_SalidasExterioresDeMesa".Mesa[#Mesa].Avanzar_E1E3) OR (#T1_ET11 AND #O_Sal_S3 AND NOT #tmp_pHs_E1_Q)) AND #EstadoZona.Marcha_CBx AND NOT #EstadoVI.Error_Mx AND NOT #EstadoZona.Manual_CBx AND #PosTR_E1;
END_REGION

REGION Network 54: #PRV_CARGA_OK_E2
   RUNG wire#powerrail
      Contact( #T1_ET01 )
      wire#w1
      Contact( #EstadoZona.Marcha_CBx )
      I_Contact( #EstadoVI.Error_Mx )
      I_Contact( #EstadoZona.Manual_CBx )
      Contact( #PosTR_E2 )
      Coil( #PTF_Ent_M2 )
   END_RUNG
   RUNG wire#powerrail
      Contact( #T1_ET20 )
      Contact( "DB1_SalidasExterioresDeMesa".Mesa[#Mesa].Avanzar_E2E4 )
   END_RUNG wire#w1
   RUNG wire#powerrail
      Contact( #T1_ET21 )
      Contact( #O_Sal_S4 )
      I_Contact( #tmp_pHs_E2_Q )
   END_RUNG wire#w1
   // the same network as SCL:
   #PTF_Ent_M2 := (#T1_ET01 OR (#T1_ET20 AND "DB1_SalidasExterioresDeMesa".Mesa[#Mesa].Avanzar_E2E4) OR (#T1_ET21 AND #O_Sal_S4 AND NOT #tmp_pHs_E2_Q)) AND #EstadoZona.Marcha_CBx AND NOT #EstadoVI.Error_Mx AND NOT #EstadoZona.Manual_CBx AND #PosTR_E2;
END_REGION

REGION Network 55: #NXT_AVTF_S3
   RUNG wire#powerrail
      Contact( #T1_ET02 )
      wire#w1
      Contact( #O_Sal_S3 )
      I_Contact( #O_Bloqueo )
      wire#w2
      Contact( #EstadoZona.Marcha_CBx )
      I_Contact( #EstadoVI.Error_Mx )
      I_Contact( #EstadoZona.Manual_CBx )
      Coil( #AVTF_Sal_M3 )
   END_RUNG
   RUNG wire#powerrail
      Contact( #T1_ET10 )
   END_RUNG wire#w1
   RUNG wire#powerrail
      Contact( #T1_ET11 )
   END_RUNG wire#w1
   RUNG wire#w1
      Contact( #O_Bloqueo )
      I_Contact( #Mx_FlujoPrin_S4 )
   END_RUNG wire#w2
   RUNG wire#powerrail
      Contact( #T1_ET02 )
      wire#w3
      Contact( #O_Vaciar )
      I_Contact( #Mx_FlujoPrin_S4 )
   END_RUNG wire#w2
   RUNG wire#powerrail
      Contact( #T1_ET03 )
   END_RUNG wire#w3
   RUNG wire#powerrail
      Contact( #T1_ET70 )
   END_RUNG wire#w2
   RUNG wire#powerrail
      Contact( #T1_ET50 )
   END_RUNG wire#w2
   // the same network as SCL:
   #AVTF_Sal_M3 := (((#T1_ET02 OR #T1_ET10 OR #T1_ET11) AND ((#O_Sal_S3 AND NOT #O_Bloqueo) OR (#O_Bloqueo AND NOT #Mx_FlujoPrin_S4))) OR ((#T1_ET02 OR #T1_ET03) AND #O_Vaciar AND NOT #Mx_FlujoPrin_S4) OR #T1_ET70 OR #T1_ET50) AND #EstadoZona.Marcha_CBx AND NOT #EstadoVI.Error_Mx AND NOT #EstadoZona.Manual_CBx;
END_REGION

REGION Network 56: #NXT_Descarga_Act_S3
   RUNG wire#powerrail
      Contact( #T1_ET50 )
      wire#w1
      Contact( #EstadoZona.Marcha_CBx )
      I_Contact( #EstadoVI.Error_Mx )
      I_Contact( #EstadoZona.Manual_CBx )
      Coil( #NXT_Descarga_Act_S3 )
   END_RUNG
   RUNG wire#powerrail
      Contact( #T1_ET70 )
   END_RUNG wire#w1
   // the same network as SCL:
   #NXT_Descarga_Act_S3 := (#T1_ET50 OR #T1_ET70) AND #EstadoZona.Marcha_CBx AND NOT #EstadoVI.Error_Mx AND NOT #EstadoZona.Manual_CBx;
END_REGION

REGION Network 57: #NXT_AVTF_S2
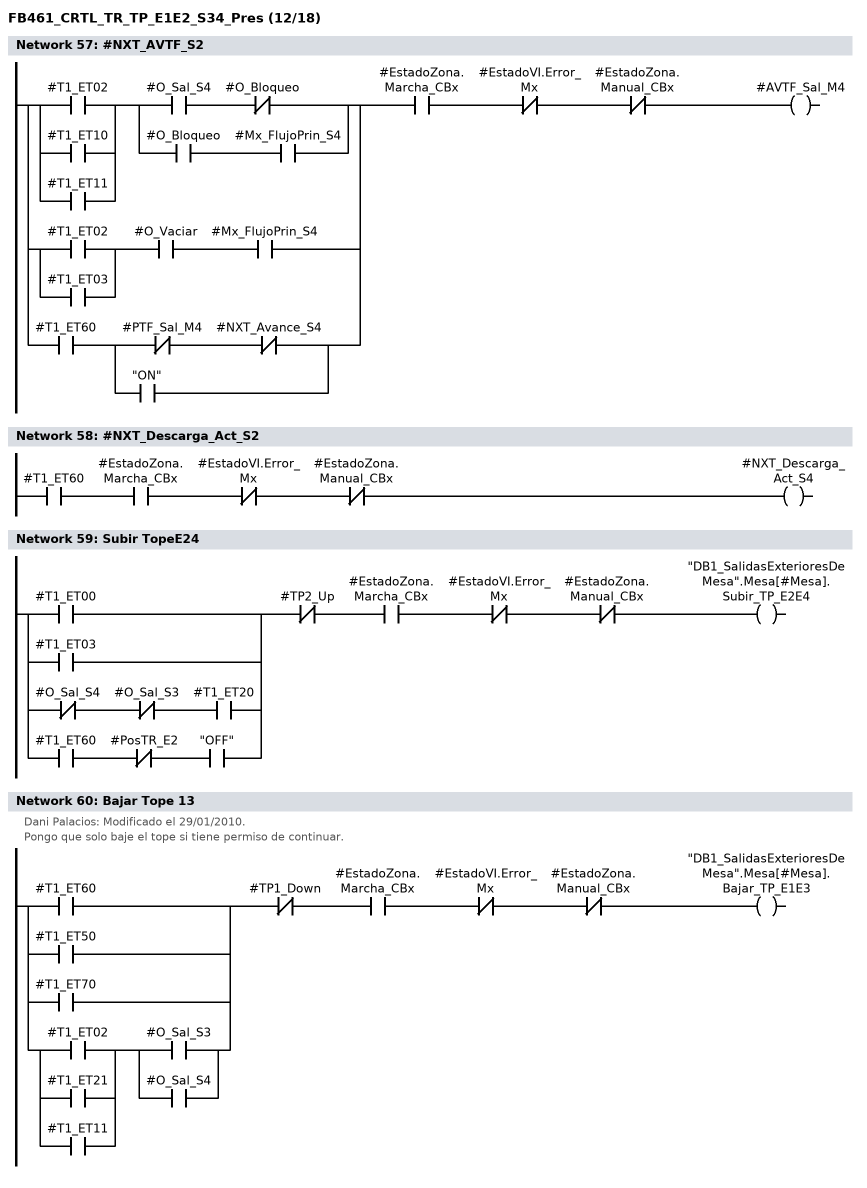
   RUNG wire#powerrail
      Contact( #T1_ET02 )
      wire#w1
      Contact( #O_Sal_S4 )
      I_Contact( #O_Bloqueo )
      wire#w2
      Contact( #EstadoZona.Marcha_CBx )
      I_Contact( #EstadoVI.Error_Mx )
      I_Contact( #EstadoZona.Manual_CBx )
      Coil( #AVTF_Sal_M4 )
   END_RUNG
   RUNG wire#powerrail
      Contact( #T1_ET10 )
   END_RUNG wire#w1
   RUNG wire#powerrail
      Contact( #T1_ET11 )
   END_RUNG wire#w1
   RUNG wire#w1
      Contact( #O_Bloqueo )
      Contact( #Mx_FlujoPrin_S4 )
   END_RUNG wire#w2
   RUNG wire#powerrail
      Contact( #T1_ET02 )
      wire#w3
      Contact( #O_Vaciar )
      Contact( #Mx_FlujoPrin_S4 )
   END_RUNG wire#w2
   RUNG wire#powerrail
      Contact( #T1_ET03 )
   END_RUNG wire#w3
   RUNG wire#powerrail
      Contact( #T1_ET60 )
      wire#w4
      I_Contact( #PTF_Sal_M4 )
      I_Contact( #NXT_Avance_S4 )
   END_RUNG wire#w2
   RUNG wire#w4
      Contact( "ON" )
   END_RUNG wire#w2
   // the same network as SCL:
   #AVTF_Sal_M4 := (((#T1_ET02 OR #T1_ET10 OR #T1_ET11) AND ((#O_Sal_S4 AND NOT #O_Bloqueo) OR (#O_Bloqueo AND #Mx_FlujoPrin_S4))) OR ((#T1_ET02 OR #T1_ET03) AND #O_Vaciar AND #Mx_FlujoPrin_S4) OR (#T1_ET60 AND ((NOT #PTF_Sal_M4 AND NOT #NXT_Avance_S4) OR "ON"))) AND #EstadoZona.Marcha_CBx AND NOT #EstadoVI.Error_Mx AND NOT #EstadoZona.Manual_CBx;
END_REGION

REGION Network 58: #NXT_Descarga_Act_S2
   RUNG wire#powerrail
      Contact( #T1_ET60 )
      Contact( #EstadoZona.Marcha_CBx )
      I_Contact( #EstadoVI.Error_Mx )
      I_Contact( #EstadoZona.Manual_CBx )
      Coil( #NXT_Descarga_Act_S4 )
   END_RUNG
   // the same network as SCL:
   #NXT_Descarga_Act_S4 := #T1_ET60 AND #EstadoZona.Marcha_CBx AND NOT #EstadoVI.Error_Mx AND NOT #EstadoZona.Manual_CBx;
END_REGION

REGION Network 59: Subir TopeE24
   RUNG wire#powerrail
      Contact( #T1_ET00 )
      wire#w1
      I_Contact( #TP2_Up )
      Contact( #EstadoZona.Marcha_CBx )
      I_Contact( #EstadoVI.Error_Mx )
      I_Contact( #EstadoZona.Manual_CBx )
      Coil( "DB1_SalidasExterioresDeMesa".Mesa[#Mesa].Subir_TP_E2E4 )
   END_RUNG
   RUNG wire#powerrail
      Contact( #T1_ET03 )
   END_RUNG wire#w1
   RUNG wire#powerrail
      I_Contact( #O_Sal_S4 )
      I_Contact( #O_Sal_S3 )
      Contact( #T1_ET20 )
   END_RUNG wire#w1
   RUNG wire#powerrail
      Contact( #T1_ET60 )
      I_Contact( #PosTR_E2 )
      Contact( "OFF" )
   END_RUNG wire#w1
   // the same network as SCL:
   "DB1_SalidasExterioresDeMesa".Mesa[#Mesa].Subir_TP_E2E4 := (#T1_ET00 OR #T1_ET03 OR (NOT #O_Sal_S4 AND NOT #O_Sal_S3 AND #T1_ET20) OR (#T1_ET60 AND NOT #PosTR_E2 AND "OFF")) AND NOT #TP2_Up AND #EstadoZona.Marcha_CBx AND NOT #EstadoVI.Error_Mx AND NOT #EstadoZona.Manual_CBx;
END_REGION

REGION Network 60: Bajar Tope 13
   // Dani Palacios: Modificado el 29/01/2010.
   // Pongo que solo baje el tope si tiene permiso de continuar.
   RUNG wire#powerrail
      Contact( #T1_ET60 )
      wire#w1
      I_Contact( #TP1_Down )
      Contact( #EstadoZona.Marcha_CBx )
      I_Contact( #EstadoVI.Error_Mx )
      I_Contact( #EstadoZona.Manual_CBx )
      Coil( "DB1_SalidasExterioresDeMesa".Mesa[#Mesa].Bajar_TP_E1E3 )
   END_RUNG
   RUNG wire#powerrail
      Contact( #T1_ET50 )
   END_RUNG wire#w1
   RUNG wire#powerrail
      Contact( #T1_ET70 )
   END_RUNG wire#w1
   RUNG wire#powerrail
      Contact( #T1_ET02 )
      wire#w2
      Contact( #O_Sal_S3 )
   END_RUNG wire#w1
   RUNG wire#powerrail
      Contact( #T1_ET21 )
   END_RUNG wire#w2
   RUNG wire#powerrail
      Contact( #T1_ET11 )
   END_RUNG wire#w2
   RUNG wire#w2
      Contact( #O_Sal_S4 )
   END_RUNG wire#w1
   // the same network as SCL:
   "DB1_SalidasExterioresDeMesa".Mesa[#Mesa].Bajar_TP_E1E3 := (#T1_ET60 OR #T1_ET50 OR #T1_ET70 OR ((#T1_ET02 OR #T1_ET21 OR #T1_ET11) AND (#O_Sal_S3 OR #O_Sal_S4))) AND NOT #TP1_Down AND #EstadoZona.Marcha_CBx AND NOT #EstadoVI.Error_Mx AND NOT #EstadoZona.Manual_CBx;
END_REGION

REGION Network 61: Bajar Tope 24
   // Dani Palacios: Modificado el 29/01/2010.
   // Pongo que solo baje el tope si tiene permiso de continuar.
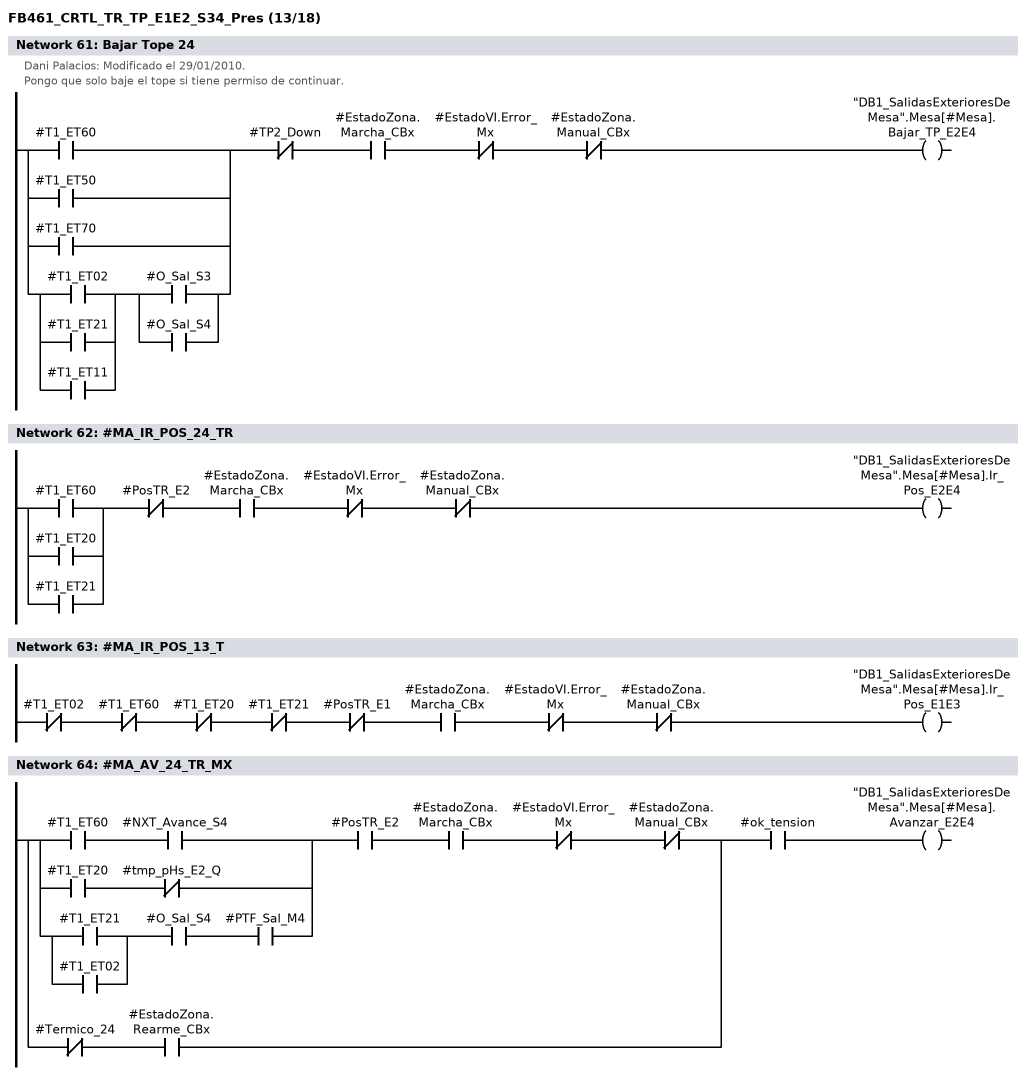
   RUNG wire#powerrail
      Contact( #T1_ET60 )
      wire#w1
      I_Contact( #TP2_Down )
      Contact( #EstadoZona.Marcha_CBx )
      I_Contact( #EstadoVI.Error_Mx )
      I_Contact( #EstadoZona.Manual_CBx )
      Coil( "DB1_SalidasExterioresDeMesa".Mesa[#Mesa].Bajar_TP_E2E4 )
   END_RUNG
   RUNG wire#powerrail
      Contact( #T1_ET50 )
   END_RUNG wire#w1
   RUNG wire#powerrail
      Contact( #T1_ET70 )
   END_RUNG wire#w1
   RUNG wire#powerrail
      Contact( #T1_ET02 )
      wire#w2
      Contact( #O_Sal_S3 )
   END_RUNG wire#w1
   RUNG wire#powerrail
      Contact( #T1_ET21 )
   END_RUNG wire#w2
   RUNG wire#powerrail
      Contact( #T1_ET11 )
   END_RUNG wire#w2
   RUNG wire#w2
      Contact( #O_Sal_S4 )
   END_RUNG wire#w1
   // the same network as SCL:
   "DB1_SalidasExterioresDeMesa".Mesa[#Mesa].Bajar_TP_E2E4 := (#T1_ET60 OR #T1_ET50 OR #T1_ET70 OR ((#T1_ET02 OR #T1_ET21 OR #T1_ET11) AND (#O_Sal_S3 OR #O_Sal_S4))) AND NOT #TP2_Down AND #EstadoZona.Marcha_CBx AND NOT #EstadoVI.Error_Mx AND NOT #EstadoZona.Manual_CBx;
END_REGION

REGION Network 62: #MA_IR_POS_24_TR
   RUNG wire#powerrail
      Contact( #T1_ET60 )
      wire#w1
      I_Contact( #PosTR_E2 )
      Contact( #EstadoZona.Marcha_CBx )
      I_Contact( #EstadoVI.Error_Mx )
      I_Contact( #EstadoZona.Manual_CBx )
      Coil( "DB1_SalidasExterioresDeMesa".Mesa[#Mesa].Ir_Pos_E2E4 )
   END_RUNG
   RUNG wire#powerrail
      Contact( #T1_ET20 )
   END_RUNG wire#w1
   RUNG wire#powerrail
      Contact( #T1_ET21 )
   END_RUNG wire#w1
   // the same network as SCL:
   "DB1_SalidasExterioresDeMesa".Mesa[#Mesa].Ir_Pos_E2E4 := (#T1_ET60 OR #T1_ET20 OR #T1_ET21) AND NOT #PosTR_E2 AND #EstadoZona.Marcha_CBx AND NOT #EstadoVI.Error_Mx AND NOT #EstadoZona.Manual_CBx;
END_REGION

REGION Network 63: #MA_IR_POS_13_T
   RUNG wire#powerrail
      I_Contact( #T1_ET02 )
      I_Contact( #T1_ET60 )
      I_Contact( #T1_ET20 )
      I_Contact( #T1_ET21 )
      I_Contact( #PosTR_E1 )
      Contact( #EstadoZona.Marcha_CBx )
      I_Contact( #EstadoVI.Error_Mx )
      I_Contact( #EstadoZona.Manual_CBx )
      Coil( "DB1_SalidasExterioresDeMesa".Mesa[#Mesa].Ir_Pos_E1E3 )
   END_RUNG
   // the same network as SCL:
   "DB1_SalidasExterioresDeMesa".Mesa[#Mesa].Ir_Pos_E1E3 := NOT #T1_ET02 AND NOT #T1_ET60 AND NOT #T1_ET20 AND NOT #T1_ET21 AND NOT #PosTR_E1 AND #EstadoZona.Marcha_CBx AND NOT #EstadoVI.Error_Mx AND NOT #EstadoZona.Manual_CBx;
END_REGION

REGION Network 64: #MA_AV_24_TR_MX
   RUNG wire#powerrail
      Contact( #T1_ET60 )
      Contact( #NXT_Avance_S4 )
      wire#w1
      Contact( #PosTR_E2 )
      Contact( #EstadoZona.Marcha_CBx )
      I_Contact( #EstadoVI.Error_Mx )
      I_Contact( #EstadoZona.Manual_CBx )
      wire#w3
      Contact( #ok_tension )
      Coil( "DB1_SalidasExterioresDeMesa".Mesa[#Mesa].Avanzar_E2E4 )
   END_RUNG
   RUNG wire#powerrail
      Contact( #T1_ET20 )
      I_Contact( #tmp_pHs_E2_Q )
   END_RUNG wire#w1
   RUNG wire#powerrail
      Contact( #T1_ET21 )
      wire#w2
      Contact( #O_Sal_S4 )
      Contact( #PTF_Sal_M4 )
   END_RUNG wire#w1
   RUNG wire#powerrail
      Contact( #T1_ET02 )
   END_RUNG wire#w2
   RUNG wire#powerrail
      I_Contact( #Termico_24 )
      Contact( #EstadoZona.Rearme_CBx )
   END_RUNG wire#w3
   // the same network as SCL:
   "DB1_SalidasExterioresDeMesa".Mesa[#Mesa].Avanzar_E2E4 := ((((#T1_ET60 AND #NXT_Avance_S4) OR (#T1_ET20 AND NOT #tmp_pHs_E2_Q) OR ((#T1_ET21 OR #T1_ET02) AND #O_Sal_S4 AND #PTF_Sal_M4)) AND #PosTR_E2 AND #EstadoZona.Marcha_CBx AND NOT #EstadoVI.Error_Mx AND NOT #EstadoZona.Manual_CBx) OR (NOT #Termico_24 AND #EstadoZona.Rearme_CBx)) AND #ok_tension;
END_REGION

REGION Network 65: #Parar_E1
   // Dani Palacios: Añadido el 21/07/2009 despues de hablar con Carlos.
   // Las entradas a las WS de Systeme U no tienen tope
   // 29/07/2009 HE METIDO LA CONDICION DE BLOQ ACTIVO PARA EVITAR QUE AVANCE NE LA 
   // ETAPA  2 SI NO TIENE PERMISO Y NO SE PUEDE DAR BLOQUEO
   // tambien meto la otra condicion para el o_vaciar*mx_flujo_prin_entrar
   // PUENTEO MX_FLUJO PRINCIPAL
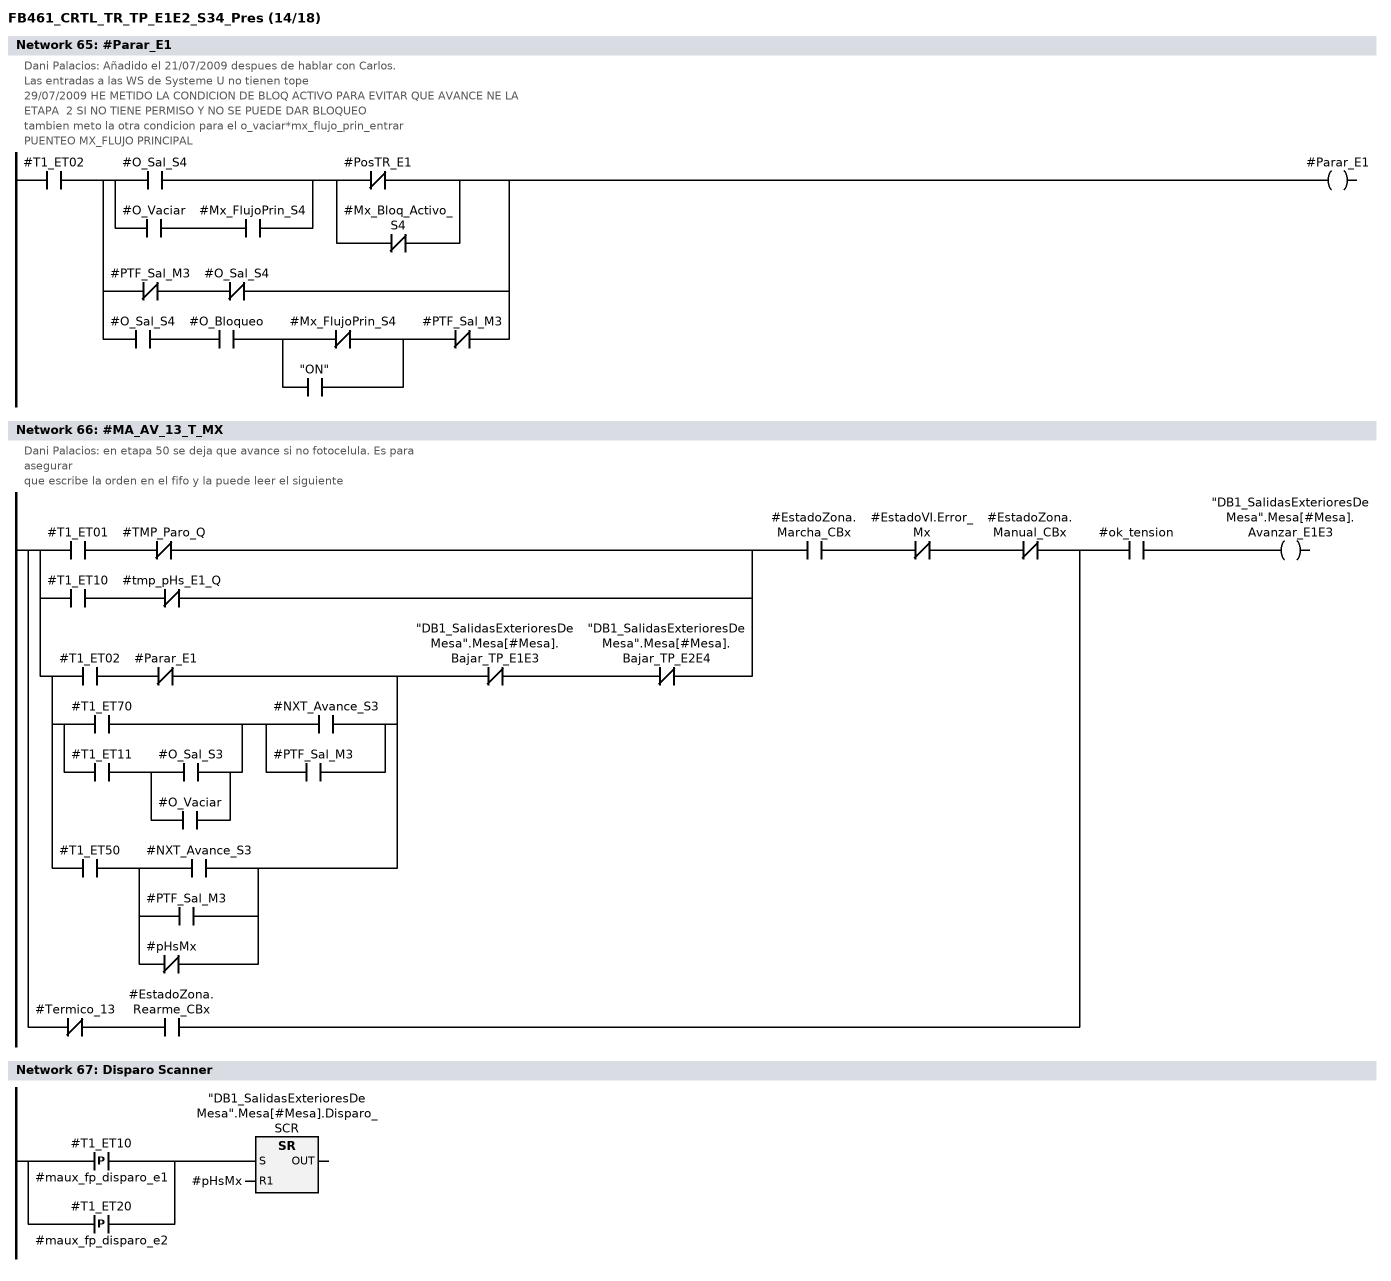
   RUNG wire#powerrail
      Contact( #T1_ET02 )
      wire#w1
      Contact( #O_Sal_S4 )
      wire#w2
      I_Contact( #PosTR_E1 )
      wire#w3
      Coil( #Parar_E1 )
   END_RUNG
   RUNG wire#w1
      Contact( #O_Vaciar )
      Contact( #Mx_FlujoPrin_S4 )
   END_RUNG wire#w2
   RUNG wire#w2
      I_Contact( #Mx_Bloq_Activo_S4 )
   END_RUNG wire#w3
   RUNG wire#w1
      I_Contact( #PTF_Sal_M3 )
      I_Contact( #O_Sal_S4 )
   END_RUNG wire#w3
   RUNG wire#w1
      Contact( #O_Sal_S4 )
      Contact( #O_Bloqueo )
      wire#w4
      I_Contact( #Mx_FlujoPrin_S4 )
      wire#w5
      I_Contact( #PTF_Sal_M3 )
   END_RUNG wire#w3
   RUNG wire#w4
      Contact( "ON" )
   END_RUNG wire#w5
   // the same network as SCL:
   #Parar_E1 := #T1_ET02 AND (((#O_Sal_S4 OR (#O_Vaciar AND #Mx_FlujoPrin_S4)) AND (NOT #PosTR_E1 OR NOT #Mx_Bloq_Activo_S4)) OR (NOT #PTF_Sal_M3 AND NOT #O_Sal_S4) OR (#O_Sal_S4 AND #O_Bloqueo AND (NOT #Mx_FlujoPrin_S4 OR "ON") AND NOT #PTF_Sal_M3));
END_REGION

REGION Network 66: #MA_AV_13_T_MX
   // Dani Palacios: en etapa 50 se deja que avance si no fotocelula. Es para 
   // asegurar 
   // que escribe la orden en el fifo y la puede leer el siguiente
   RUNG wire#powerrail
      Contact( #T1_ET01 )
      I_Contact( #TMP_Paro_Q )
      wire#w1
      Contact( #EstadoZona.Marcha_CBx )
      I_Contact( #EstadoVI.Error_Mx )
      I_Contact( #EstadoZona.Manual_CBx )
      wire#w6
      Contact( #ok_tension )
      Coil( "DB1_SalidasExterioresDeMesa".Mesa[#Mesa].Avanzar_E1E3 )
   END_RUNG
   RUNG wire#powerrail
      Contact( #T1_ET10 )
      I_Contact( #tmp_pHs_E1_Q )
   END_RUNG wire#w1
   RUNG wire#powerrail
      Contact( #T1_ET02 )
      I_Contact( #Parar_E1 )
      wire#w2
      I_Contact( "DB1_SalidasExterioresDeMesa".Mesa[#Mesa].Bajar_TP_E1E3 )
      I_Contact( "DB1_SalidasExterioresDeMesa".Mesa[#Mesa].Bajar_TP_E2E4 )
   END_RUNG wire#w1
   RUNG wire#powerrail
      Contact( #T1_ET70 )
      wire#w3
      Contact( #NXT_Avance_S3 )
   END_RUNG wire#w2
   RUNG wire#powerrail
      Contact( #T1_ET11 )
      wire#w4
      Contact( #O_Sal_S3 )
   END_RUNG wire#w3
   RUNG wire#w4
      Contact( #O_Vaciar )
   END_RUNG wire#w3
   RUNG wire#w3
      Contact( #PTF_Sal_M3 )
   END_RUNG wire#w2
   RUNG wire#powerrail
      Contact( #T1_ET50 )
      wire#w5
      Contact( #NXT_Avance_S3 )
   END_RUNG wire#w2
   RUNG wire#w5
      Contact( #PTF_Sal_M3 )
   END_RUNG wire#w2
   RUNG wire#w5
      I_Contact( #pHsMx )
   END_RUNG wire#w2
   RUNG wire#powerrail
      I_Contact( #Termico_13 )
      Contact( #EstadoZona.Rearme_CBx )
   END_RUNG wire#w6
   // the same network as SCL:
   "DB1_SalidasExterioresDeMesa".Mesa[#Mesa].Avanzar_E1E3 := ((((#T1_ET01 AND NOT #TMP_Paro_Q) OR (#T1_ET10 AND NOT #tmp_pHs_E1_Q) OR (((#T1_ET02 AND NOT #Parar_E1) OR ((#T1_ET70 OR (#T1_ET11 AND (#O_Sal_S3 OR #O_Vaciar))) AND (#NXT_Avance_S3 OR #PTF_Sal_M3)) OR (#T1_ET50 AND (#NXT_Avance_S3 OR #PTF_Sal_M3 OR NOT #pHsMx))) AND NOT "DB1_SalidasExterioresDeMesa".Mesa[#Mesa].Bajar_TP_E1E3 AND NOT "DB1_SalidasExterioresDeMesa".Mesa[#Mesa].Bajar_TP_E2E4)) AND #EstadoZona.Marcha_CBx AND NOT #EstadoVI.Error_Mx AND NOT #EstadoZona.Manual_CBx) OR (NOT #Termico_13 AND #EstadoZona.Rearme_CBx)) AND #ok_tension;
END_REGION

REGION Network 67: Disparo Scanner
   RUNG wire#powerrail
      P_Contact(operand := #T1_ET10, bit := #maux_fp_disparo_e1)
      wire#w1
      S_SR(operand := "DB1_SalidasExterioresDeMesa".Mesa[#Mesa].Disparo_SCR, r1 := #pHsMx)
   END_RUNG
   RUNG wire#powerrail
      P_Contact(operand := #T1_ET20, bit := #maux_fp_disparo_e2)
   END_RUNG wire#w1
   // the same network as SCL:
   #_w1 := #T1_ET10 AND NOT #maux_fp_disparo_e1;   // rising edge of #T1_ET10
   #maux_fp_disparo_e1 := #T1_ET10;
   #_w2 := #T1_ET20 AND NOT #maux_fp_disparo_e2;   // rising edge of #T1_ET20
   #maux_fp_disparo_e2 := #T1_ET20;
   IF #_w1 OR #_w2 THEN
       "DB1_SalidasExterioresDeMesa".Mesa[#Mesa].Disparo_SCR := TRUE;   // SR flip-flop
   END_IF;
   IF #pHsMx THEN "DB1_SalidasExterioresDeMesa".Mesa[#Mesa].Disparo_SCR := FALSE; END_IF;
END_REGION

